REGION Network 56: Paregg. Testa - [Sollevatore] - Movimento operazione a lavoro / a riposo
   // Sollevatore del Centraggio - Scende quando è in posizione e sta attendendo il pezzo
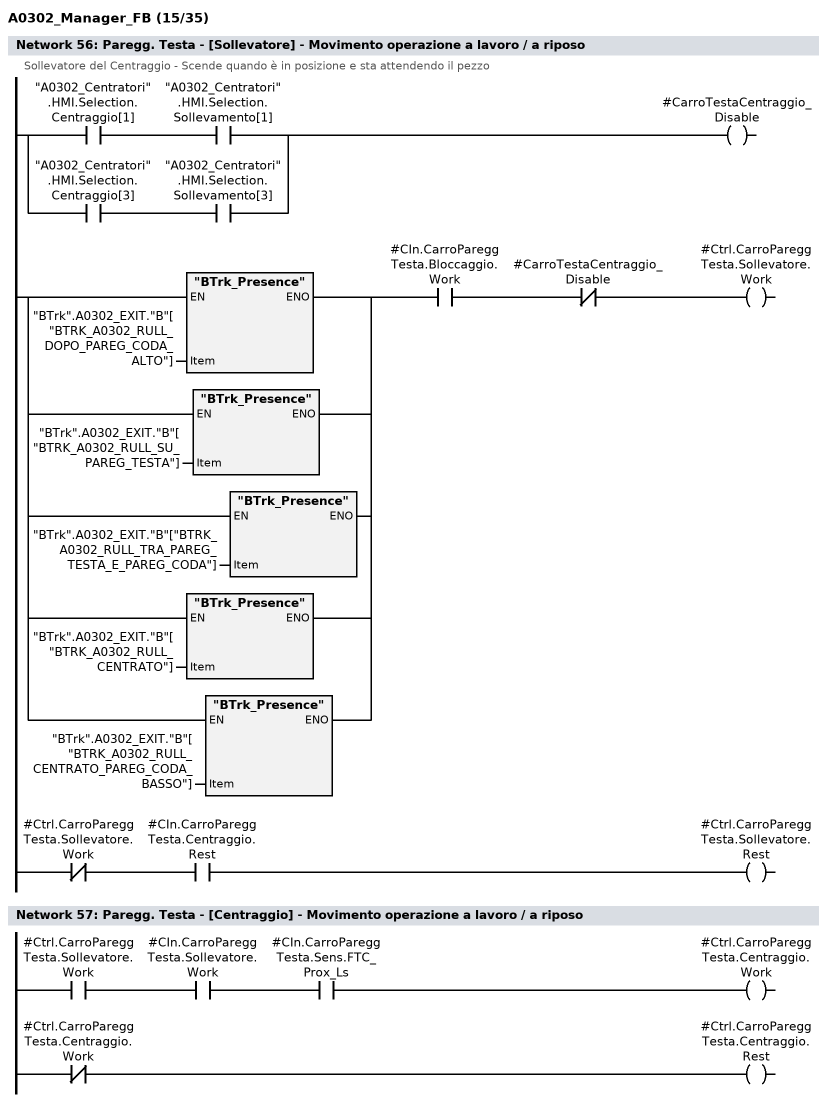
   RUNG wire#powerrail
      Contact( "A0302_Centratori".HMI.Selection.Centraggio[1] )
      Contact( "A0302_Centratori".HMI.Selection.Sollevamento[1] )
      wire#w1
      Coil( #CarroTestaCentraggio_Disable )
   END_RUNG
   RUNG wire#powerrail
      Contact( "A0302_Centratori".HMI.Selection.Centraggio[3] )
      Contact( "A0302_Centratori".HMI.Selection.Sollevamento[3] )
   END_RUNG wire#w1
   RUNG wire#powerrail
      "BTrk_Presence"(Item := "BTrk".A0302_EXIT."B"["BTRK_A0302_RULL_DOPO_PAREG_CODA_ALTO"])
      wire#w2
      Contact( #CIn.CarroPareggTesta.Bloccaggio.Work )
      I_Contact( #CarroTestaCentraggio_Disable )
      Coil( #Ctrl.CarroPareggTesta.Sollevatore.Work )
   END_RUNG
   RUNG wire#powerrail
      "BTrk_Presence"(Item := "BTrk".A0302_EXIT."B"["BTRK_A0302_RULL_SU_PAREG_TESTA"])
   END_RUNG wire#w2
   RUNG wire#powerrail
      "BTrk_Presence"(Item := "BTrk".A0302_EXIT."B"["BTRK_A0302_RULL_TRA_PAREG_TESTA_E_PAREG_CODA"])
   END_RUNG wire#w2
   RUNG wire#powerrail
      "BTrk_Presence"(Item := "BTrk".A0302_EXIT."B"["BTRK_A0302_RULL_CENTRATO"])
   END_RUNG wire#w2
   RUNG wire#powerrail
      "BTrk_Presence"(Item := "BTrk".A0302_EXIT."B"["BTRK_A0302_RULL_CENTRATO_PAREG_CODA_BASSO"])
   END_RUNG wire#w2
   RUNG wire#powerrail
      I_Contact( #Ctrl.CarroPareggTesta.Sollevatore.Work )
      Contact( #CIn.CarroPareggTesta.Centraggio.Rest )
      Coil( #Ctrl.CarroPareggTesta.Sollevatore.Rest )
   END_RUNG
   // the same network as SCL:
   #CarroTestaCentraggio_Disable := ("A0302_Centratori".HMI.Selection.Centraggio[1] AND "A0302_Centratori".HMI.Selection.Sollevamento[1]) OR ("A0302_Centratori".HMI.Selection.Centraggio[3] AND "A0302_Centratori".HMI.Selection.Sollevamento[3]);
   "BTrk_Presence"(Item := "BTrk".A0302_EXIT."B"["BTRK_A0302_RULL_DOPO_PAREG_CODA_ALTO"], ENO => #_w1);
   "BTrk_Presence"(Item := "BTrk".A0302_EXIT."B"["BTRK_A0302_RULL_SU_PAREG_TESTA"], ENO => #_w2);
   "BTrk_Presence"(Item := "BTrk".A0302_EXIT."B"["BTRK_A0302_RULL_TRA_PAREG_TESTA_E_PAREG_CODA"], ENO => #_w3);
   "BTrk_Presence"(Item := "BTrk".A0302_EXIT."B"["BTRK_A0302_RULL_CENTRATO"], ENO => #_w4);
   "BTrk_Presence"(Item := "BTrk".A0302_EXIT."B"["BTRK_A0302_RULL_CENTRATO_PAREG_CODA_BASSO"], ENO => #_w5);
   #Ctrl.CarroPareggTesta.Sollevatore.Work := (#_w1 OR #_w2 OR #_w3 OR #_w4 OR #_w5) AND #CIn.CarroPareggTesta.Bloccaggio.Work AND NOT #CarroTestaCentraggio_Disable;
   #Ctrl.CarroPareggTesta.Sollevatore.Rest := NOT #Ctrl.CarroPareggTesta.Sollevatore.Work AND #CIn.CarroPareggTesta.Centraggio.Rest;
END_REGION

REGION Network 57: Paregg. Testa - [Centraggio] - Movimento operazione a lavoro / a riposo
   RUNG wire#powerrail
      Contact( #Ctrl.CarroPareggTesta.Sollevatore.Work )
      Contact( #CIn.CarroPareggTesta.Sollevatore.Work )
      Contact( #CIn.CarroPareggTesta.Sens.FTC_Prox_Ls )
      Coil( #Ctrl.CarroPareggTesta.Centraggio.Work )
   END_RUNG
   RUNG wire#powerrail
      I_Contact( #Ctrl.CarroPareggTesta.Centraggio.Work )
      Coil( #Ctrl.CarroPareggTesta.Centraggio.Rest )
   END_RUNG
   // the same network as SCL:
   #Ctrl.CarroPareggTesta.Centraggio.Work := #Ctrl.CarroPareggTesta.Sollevatore.Work AND #CIn.CarroPareggTesta.Sollevatore.Work AND #CIn.CarroPareggTesta.Sens.FTC_Prox_Ls;
   #Ctrl.CarroPareggTesta.Centraggio.Rest := NOT #Ctrl.CarroPareggTesta.Centraggio.Work;
END_REGION

REGION Network 58: <+>
END_REGION

REGION Network 59: Paregg. Testa - [Ax - Sollevatore + Centraggio] - COut Manager
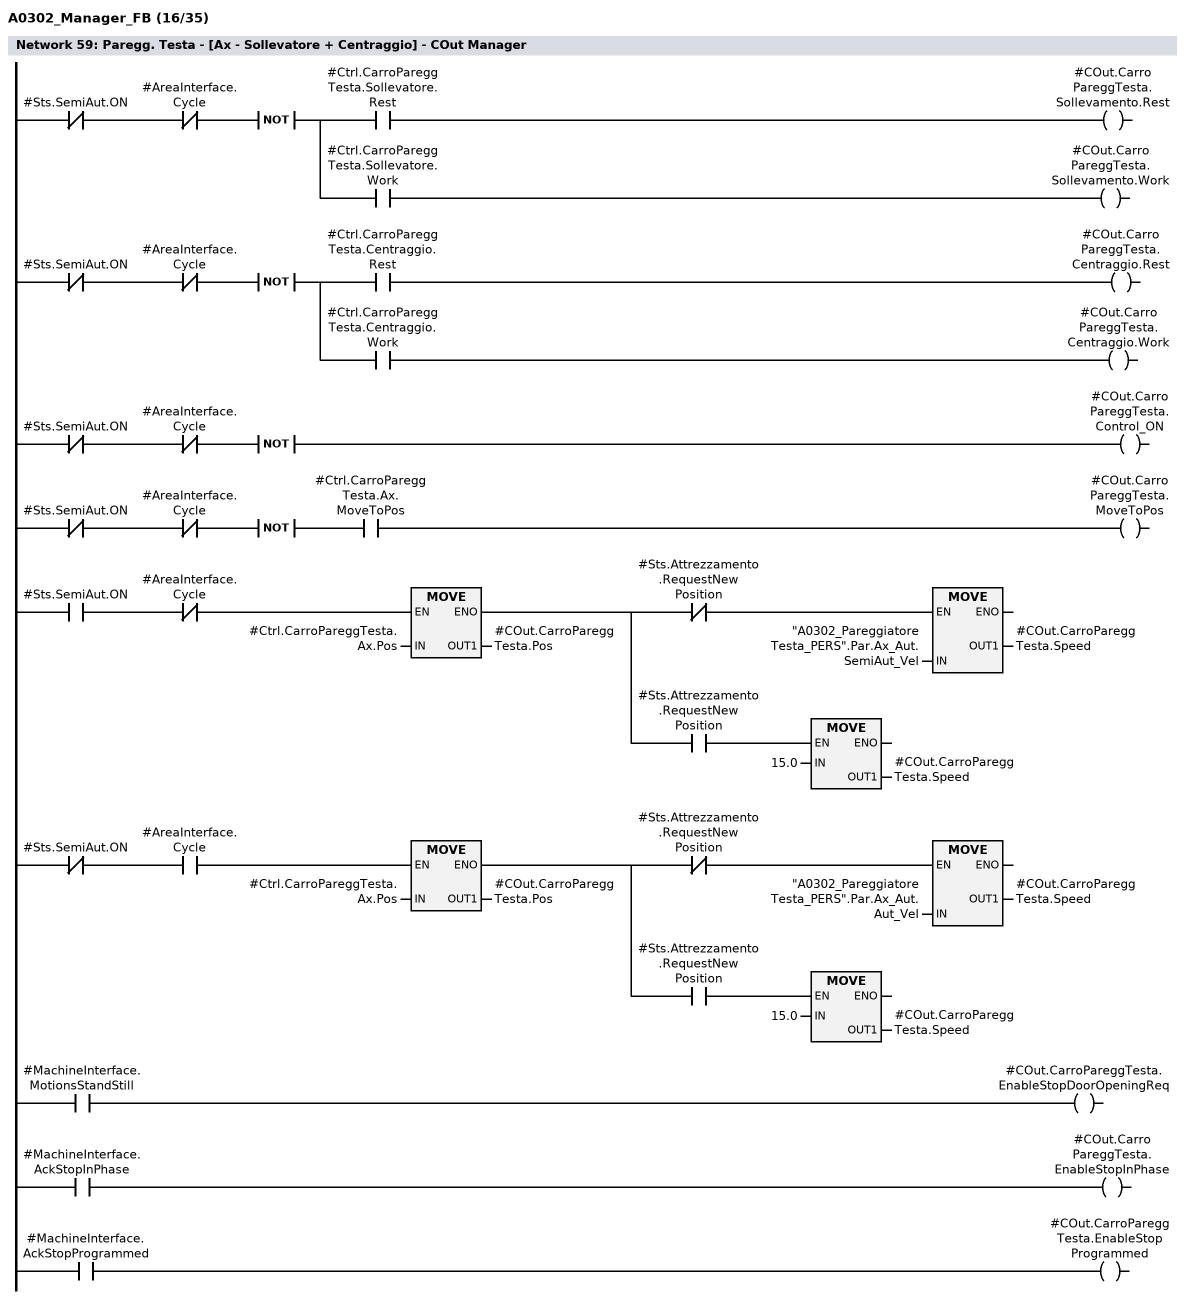
   RUNG wire#powerrail
      I_Contact( #Sts.SemiAut.ON )
      I_Contact( #AreaInterface.Cycle )
      Not()
      wire#w1
      Contact( #Ctrl.CarroPareggTesta.Sollevatore.Rest )
      Coil( #COut.CarroPareggTesta.Sollevamento.Rest )
   END_RUNG
   RUNG wire#w1
      Contact( #Ctrl.CarroPareggTesta.Sollevatore.Work )
      Coil( #COut.CarroPareggTesta.Sollevamento.Work )
   END_RUNG
   RUNG wire#powerrail
      I_Contact( #Sts.SemiAut.ON )
      I_Contact( #AreaInterface.Cycle )
      Not()
      wire#w2
      Contact( #Ctrl.CarroPareggTesta.Centraggio.Rest )
      Coil( #COut.CarroPareggTesta.Centraggio.Rest )
   END_RUNG
   RUNG wire#w2
      Contact( #Ctrl.CarroPareggTesta.Centraggio.Work )
      Coil( #COut.CarroPareggTesta.Centraggio.Work )
   END_RUNG
   RUNG wire#powerrail
      I_Contact( #Sts.SemiAut.ON )
      I_Contact( #AreaInterface.Cycle )
      Not()
      Coil( #COut.CarroPareggTesta.Control_ON )
   END_RUNG
   RUNG wire#powerrail
      I_Contact( #Sts.SemiAut.ON )
      I_Contact( #AreaInterface.Cycle )
      Not()
      Contact( #Ctrl.CarroPareggTesta.Ax.MoveToPos )
      Coil( #COut.CarroPareggTesta.MoveToPos )
   END_RUNG
   RUNG wire#powerrail
      Contact( #Sts.SemiAut.ON )
      I_Contact( #AreaInterface.Cycle )
      Move(in := #Ctrl.CarroPareggTesta.Ax.Pos, out1 => #COut.CarroPareggTesta.Pos)
      wire#w3
      I_Contact( #Sts.Attrezzamento.RequestNewPosition )
      Move(in := "A0302_PareggiatoreTesta_PERS".Par.Ax_Aut.SemiAut_Vel, out1 => #COut.CarroPareggTesta.Speed)
   END_RUNG
   RUNG wire#w3
      Contact( #Sts.Attrezzamento.RequestNewPosition )
      Move(in := 15.0, out1 => #COut.CarroPareggTesta.Speed)
   END_RUNG
   RUNG wire#powerrail
      I_Contact( #Sts.SemiAut.ON )
      Contact( #AreaInterface.Cycle )
      Move(in := #Ctrl.CarroPareggTesta.Ax.Pos, out1 => #COut.CarroPareggTesta.Pos)
      wire#w4
      I_Contact( #Sts.Attrezzamento.RequestNewPosition )
      Move(in := "A0302_PareggiatoreTesta_PERS".Par.Ax_Aut.Aut_Vel, out1 => #COut.CarroPareggTesta.Speed)
   END_RUNG
   RUNG wire#w4
      Contact( #Sts.Attrezzamento.RequestNewPosition )
      Move(in := 15.0, out1 => #COut.CarroPareggTesta.Speed)
   END_RUNG
   RUNG wire#powerrail
      Contact( #MachineInterface.MotionsStandStill )
      Coil( #COut.CarroPareggTesta.EnableStopDoorOpeningReq )
   END_RUNG
   RUNG wire#powerrail
      Contact( #MachineInterface.AckStopInPhase )
      Coil( #COut.CarroPareggTesta.EnableStopInPhase )
   END_RUNG
   RUNG wire#powerrail
      Contact( #MachineInterface.AckStopProgrammed )
      Coil( #COut.CarroPareggTesta.EnableStopProgrammed )
   END_RUNG
   // the same network as SCL:
   #_w1 := NOT (NOT #Sts.SemiAut.ON AND NOT #AreaInterface.Cycle);
   #COut.CarroPareggTesta.Sollevamento.Rest := #_w1 AND #Ctrl.CarroPareggTesta.Sollevatore.Rest;
   #COut.CarroPareggTesta.Sollevamento.Work := #_w1 AND #Ctrl.CarroPareggTesta.Sollevatore.Work;
   #_w2 := NOT (NOT #Sts.SemiAut.ON AND NOT #AreaInterface.Cycle);
   #COut.CarroPareggTesta.Centraggio.Rest := #_w2 AND #Ctrl.CarroPareggTesta.Centraggio.Rest;
   #COut.CarroPareggTesta.Centraggio.Work := #_w2 AND #Ctrl.CarroPareggTesta.Centraggio.Work;
   #COut.CarroPareggTesta.Control_ON := NOT (NOT #Sts.SemiAut.ON AND NOT #AreaInterface.Cycle);
   #COut.CarroPareggTesta.MoveToPos := NOT (NOT #Sts.SemiAut.ON AND NOT #AreaInterface.Cycle) AND #Ctrl.CarroPareggTesta.Ax.MoveToPos;
   #_w3 := #Sts.SemiAut.ON AND NOT #AreaInterface.Cycle;
   IF #_w3 THEN #COut.CarroPareggTesta.Pos := #Ctrl.CarroPareggTesta.Ax.Pos; END_IF;
   IF #_w3 AND NOT #Sts.Attrezzamento.RequestNewPosition THEN
       #COut.CarroPareggTesta.Speed := "A0302_PareggiatoreTesta_PERS".Par.Ax_Aut.SemiAut_Vel;
   END_IF;
   IF #_w3 AND #Sts.Attrezzamento.RequestNewPosition THEN #COut.CarroPareggTesta.Speed := 15.0; END_IF;
   #_w4 := NOT #Sts.SemiAut.ON AND #AreaInterface.Cycle;
   IF #_w4 THEN #COut.CarroPareggTesta.Pos := #Ctrl.CarroPareggTesta.Ax.Pos; END_IF;
   IF #_w4 AND NOT #Sts.Attrezzamento.RequestNewPosition THEN
       #COut.CarroPareggTesta.Speed := "A0302_PareggiatoreTesta_PERS".Par.Ax_Aut.Aut_Vel;
   END_IF;
   IF #_w4 AND #Sts.Attrezzamento.RequestNewPosition THEN #COut.CarroPareggTesta.Speed := 15.0; END_IF;
   #COut.CarroPareggTesta.EnableStopDoorOpeningReq := #MachineInterface.MotionsStandStill;
   #COut.CarroPareggTesta.EnableStopInPhase := #MachineInterface.AckStopInPhase;
   #COut.CarroPareggTesta.EnableStopProgrammed := #MachineInterface.AckStopProgrammed;
END_REGION

REGION Network 60: Paregg. Testa [Bloccaggio] - Movimento operazione a lavoro / a riposo
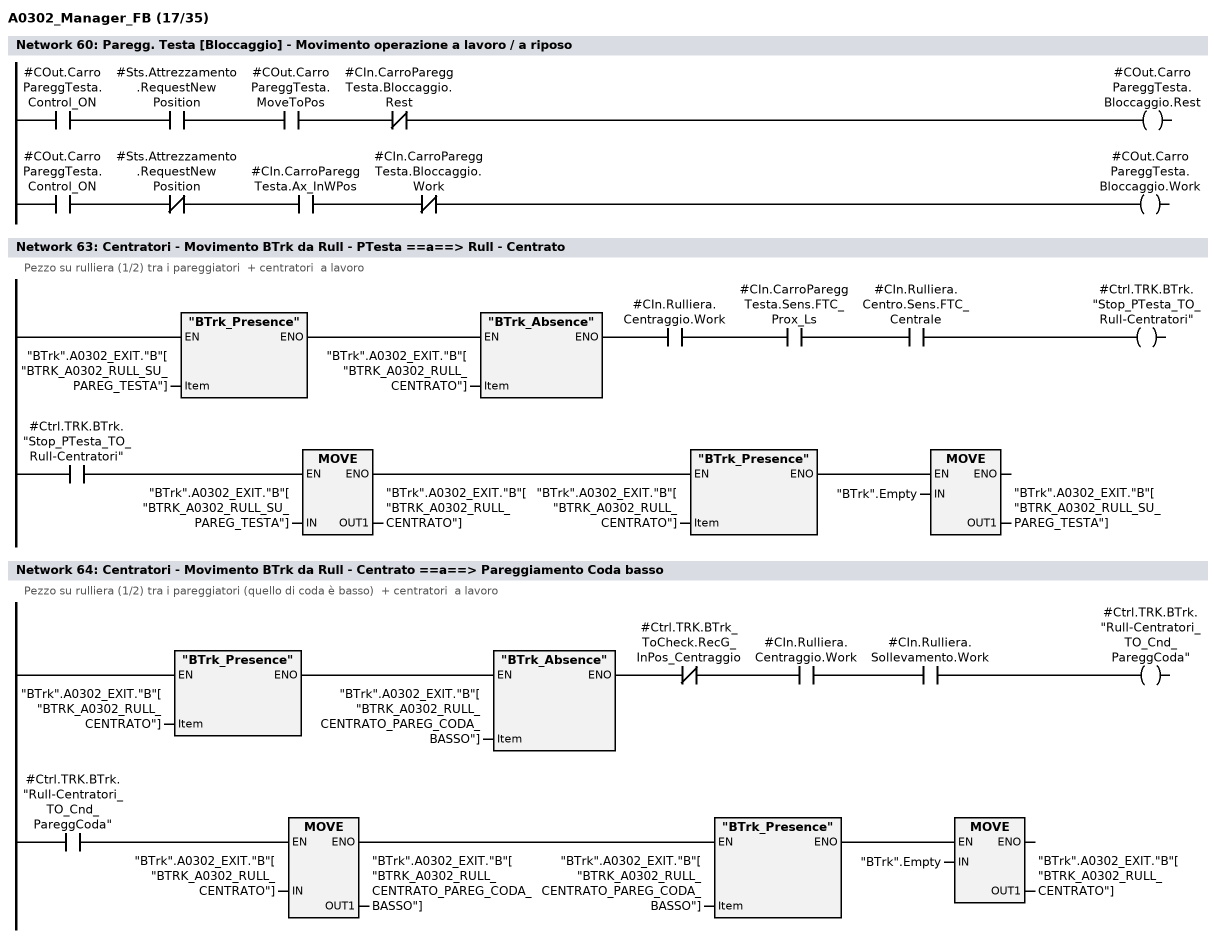
   RUNG wire#powerrail
      Contact( #COut.CarroPareggTesta.Control_ON )
      Contact( #Sts.Attrezzamento.RequestNewPosition )
      Contact( #COut.CarroPareggTesta.MoveToPos )
      I_Contact( #CIn.CarroPareggTesta.Bloccaggio.Rest )
      Coil( #COut.CarroPareggTesta.Bloccaggio.Rest )
   END_RUNG
   RUNG wire#powerrail
      Contact( #COut.CarroPareggTesta.Control_ON )
      I_Contact( #Sts.Attrezzamento.RequestNewPosition )
      Contact( #CIn.CarroPareggTesta.Ax_InWPos )
      I_Contact( #CIn.CarroPareggTesta.Bloccaggio.Work )
      Coil( #COut.CarroPareggTesta.Bloccaggio.Work )
   END_RUNG
   // the same network as SCL:
   #COut.CarroPareggTesta.Bloccaggio.Rest := #COut.CarroPareggTesta.Control_ON AND #Sts.Attrezzamento.RequestNewPosition AND #COut.CarroPareggTesta.MoveToPos AND NOT #CIn.CarroPareggTesta.Bloccaggio.Rest;
   #COut.CarroPareggTesta.Bloccaggio.Work := #COut.CarroPareggTesta.Control_ON AND NOT #Sts.Attrezzamento.RequestNewPosition AND #CIn.CarroPareggTesta.Ax_InWPos AND NOT #CIn.CarroPareggTesta.Bloccaggio.Work;
END_REGION

REGION Network 61: <<<< CENTRATORI >>>>
END_REGION

REGION Network 62: <+>
END_REGION

REGION Network 63: Centratori - Movimento BTrk da Rull - PTesta ==a==> Rull - Centrato
   // Pezzo su rulliera (1/2) tra i pareggiatori  + centratori  a lavoro
   RUNG wire#powerrail
      "BTrk_Presence"(Item := "BTrk".A0302_EXIT."B"["BTRK_A0302_RULL_SU_PAREG_TESTA"])
      "BTrk_Absence"(Item := "BTrk".A0302_EXIT."B"["BTRK_A0302_RULL_CENTRATO"])
      Contact( #CIn.Rulliera.Centraggio.Work )
      Contact( #CIn.CarroPareggTesta.Sens.FTC_Prox_Ls )
      Contact( #CIn.Rulliera.Centro.Sens.FTC_Centrale )
      Coil( #Ctrl.TRK.BTrk."Stop_PTesta_TO_Rull-Centratori" )
   END_RUNG
   RUNG wire#powerrail
      Contact( #Ctrl.TRK.BTrk."Stop_PTesta_TO_Rull-Centratori" )
      Move(in := "BTrk".A0302_EXIT."B"["BTRK_A0302_RULL_SU_PAREG_TESTA"], out1 => "BTrk".A0302_EXIT."B"["BTRK_A0302_RULL_CENTRATO"])
      "BTrk_Presence"(Item := "BTrk".A0302_EXIT."B"["BTRK_A0302_RULL_CENTRATO"])
      Move(in := "BTrk".Empty, out1 => "BTrk".A0302_EXIT."B"["BTRK_A0302_RULL_SU_PAREG_TESTA"])
   END_RUNG
   // the same network as SCL:
   "BTrk_Presence"(Item := "BTrk".A0302_EXIT."B"["BTRK_A0302_RULL_SU_PAREG_TESTA"], ENO => #_w1);
   "BTrk_Absence"(EN := #_w1, Item := "BTrk".A0302_EXIT."B"["BTRK_A0302_RULL_CENTRATO"], ENO => #_w2);
   #Ctrl.TRK.BTrk."Stop_PTesta_TO_Rull-Centratori" := #_w2 AND #CIn.Rulliera.Centraggio.Work AND #CIn.CarroPareggTesta.Sens.FTC_Prox_Ls AND #CIn.Rulliera.Centro.Sens.FTC_Centrale;
   IF #Ctrl.TRK.BTrk."Stop_PTesta_TO_Rull-Centratori" THEN
       "BTrk".A0302_EXIT."B"["BTRK_A0302_RULL_CENTRATO"] := "BTrk".A0302_EXIT."B"["BTRK_A0302_RULL_SU_PAREG_TESTA"];
   END_IF;
   "BTrk_Presence"(EN := #Ctrl.TRK.BTrk."Stop_PTesta_TO_Rull-Centratori",
                   Item := "BTrk".A0302_EXIT."B"["BTRK_A0302_RULL_CENTRATO"],
                   ENO => #_w3);
   IF #_w3 THEN "BTrk".A0302_EXIT."B"["BTRK_A0302_RULL_SU_PAREG_TESTA"] := "BTrk".Empty; END_IF;
END_REGION

REGION Network 64: Centratori - Movimento BTrk da Rull - Centrato ==a==> Pareggiamento Coda basso
   // Pezzo su rulliera (1/2) tra i pareggiatori (quello di coda è basso)  + centratori  a lavoro
   RUNG wire#powerrail
      "BTrk_Presence"(Item := "BTrk".A0302_EXIT."B"["BTRK_A0302_RULL_CENTRATO"])
      "BTrk_Absence"(Item := "BTrk".A0302_EXIT."B"["BTRK_A0302_RULL_CENTRATO_PAREG_CODA_BASSO"])
      I_Contact( #Ctrl.TRK.BTrk_ToCheck.RecG_InPos_Centraggio )
      Contact( #CIn.Rulliera.Centraggio.Work )
      Contact( #CIn.Rulliera.Sollevamento.Work )
      Coil( #Ctrl.TRK.BTrk."Rull-Centratori_TO_Cnd_PareggCoda" )
   END_RUNG
   RUNG wire#powerrail
      Contact( #Ctrl.TRK.BTrk."Rull-Centratori_TO_Cnd_PareggCoda" )
      Move(in := "BTrk".A0302_EXIT."B"["BTRK_A0302_RULL_CENTRATO"], out1 => "BTrk".A0302_EXIT."B"["BTRK_A0302_RULL_CENTRATO_PAREG_CODA_BASSO"])
      "BTrk_Presence"(Item := "BTrk".A0302_EXIT."B"["BTRK_A0302_RULL_CENTRATO_PAREG_CODA_BASSO"])
      Move(in := "BTrk".Empty, out1 => "BTrk".A0302_EXIT."B"["BTRK_A0302_RULL_CENTRATO"])
   END_RUNG
   // the same network as SCL:
   "BTrk_Presence"(Item := "BTrk".A0302_EXIT."B"["BTRK_A0302_RULL_CENTRATO"], ENO => #_w1);
   "BTrk_Absence"(EN := #_w1,
                  Item := "BTrk".A0302_EXIT."B"["BTRK_A0302_RULL_CENTRATO_PAREG_CODA_BASSO"],
                  ENO => #_w2);
   #Ctrl.TRK.BTrk."Rull-Centratori_TO_Cnd_PareggCoda" := #_w2 AND NOT #Ctrl.TRK.BTrk_ToCheck.RecG_InPos_Centraggio AND #CIn.Rulliera.Centraggio.Work AND #CIn.Rulliera.Sollevamento.Work;
   IF #Ctrl.TRK.BTrk."Rull-Centratori_TO_Cnd_PareggCoda" THEN
       "BTrk".A0302_EXIT."B"["BTRK_A0302_RULL_CENTRATO_PAREG_CODA_BASSO"] := "BTrk".A0302_EXIT."B"["BTRK_A0302_RULL_CENTRATO"];
   END_IF;
   "BTrk_Presence"(EN := #Ctrl.TRK.BTrk."Rull-Centratori_TO_Cnd_PareggCoda",
                   Item := "BTrk".A0302_EXIT."B"["BTRK_A0302_RULL_CENTRATO_PAREG_CODA_BASSO"],
                   ENO => #_w3);
   IF #_w3 THEN "BTrk".A0302_EXIT."B"["BTRK_A0302_RULL_CENTRATO"] := "BTrk".Empty; END_IF;
END_REGION

REGION Network 65: Centratori - Movimento BTrk da Pareggiamento Coda basso ==a==> Pareggiato
   // Pezzo su rulliera (1/2) tra i pareggiatori e paregiatura di coda eseguito lavoro cilindro idraulico (ora si sa la misura del pezzo, si può mettere utenze in attesa del prossimo pezzo)
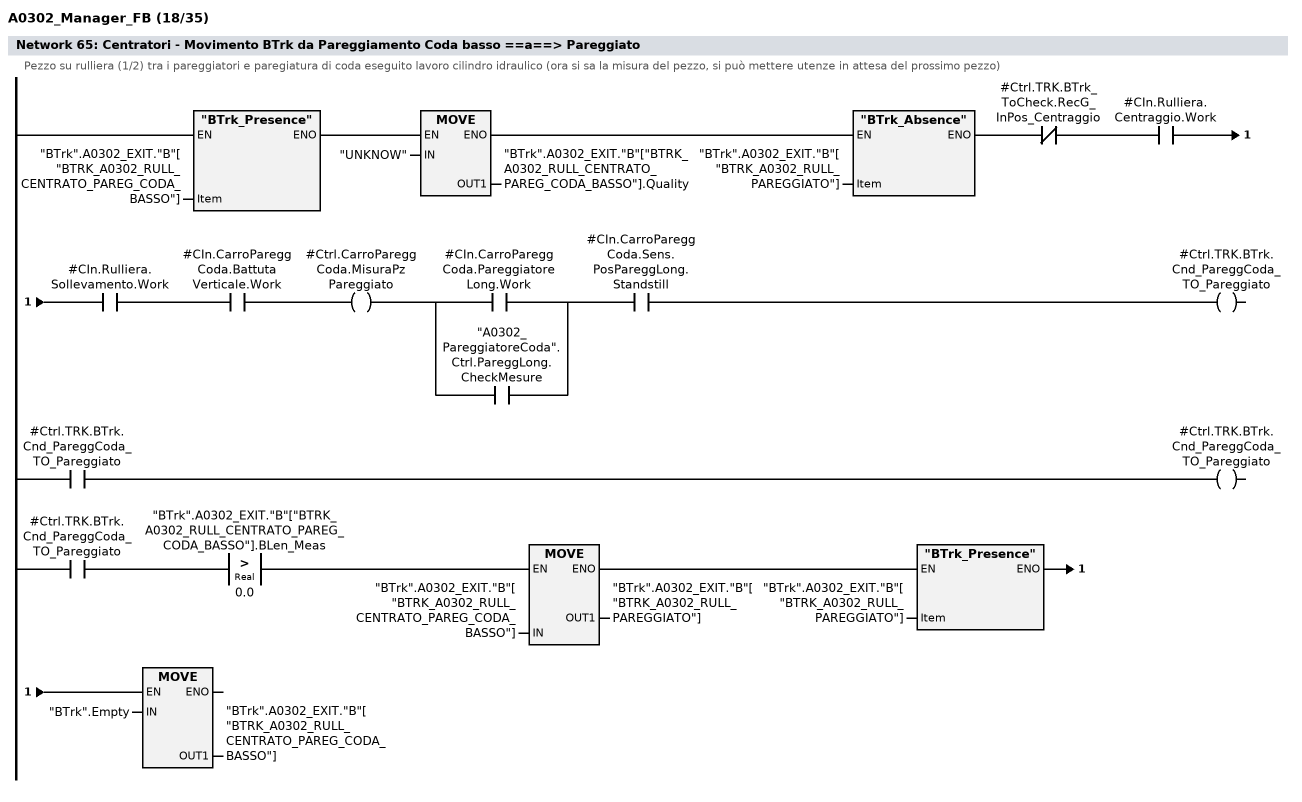
   RUNG wire#powerrail
      "BTrk_Presence"(Item := "BTrk".A0302_EXIT."B"["BTRK_A0302_RULL_CENTRATO_PAREG_CODA_BASSO"])
      Move(in := "UNKNOW", out1 => "BTrk".A0302_EXIT."B"["BTRK_A0302_RULL_CENTRATO_PAREG_CODA_BASSO"].Quality)
      "BTrk_Absence"(Item := "BTrk".A0302_EXIT."B"["BTRK_A0302_RULL_PAREGGIATO"])
      I_Contact( #Ctrl.TRK.BTrk_ToCheck.RecG_InPos_Centraggio )
      Contact( #CIn.Rulliera.Centraggio.Work )
      Contact( #CIn.Rulliera.Sollevamento.Work )
      Contact( #CIn.CarroPareggCoda.BattutaVerticale.Work )
      Coil( #Ctrl.CarroPareggCoda.MisuraPzPareggiato )
      wire#w1
      Contact( #CIn.CarroPareggCoda.PareggiatoreLong.Work )
      wire#w2
      Contact( #CIn.CarroPareggCoda.Sens.PosPareggLong.Standstill )
      Coil( #Ctrl.TRK.BTrk.Cnd_PareggCoda_TO_Pareggiato )
   END_RUNG
   RUNG wire#w1
      Contact( "A0302_PareggiatoreCoda".Ctrl.PareggLong.CheckMesure )
   END_RUNG wire#w2
   RUNG wire#powerrail
      Contact( #Ctrl.TRK.BTrk.Cnd_PareggCoda_TO_Pareggiato )
      Coil( #Ctrl.TRK.BTrk.Cnd_PareggCoda_TO_Pareggiato )
   END_RUNG
   RUNG wire#powerrail
      Contact( #Ctrl.TRK.BTrk.Cnd_PareggCoda_TO_Pareggiato )
      { S7_Templates := "SrcType := Real" } GT_Contact(in1 := "BTrk".A0302_EXIT."B"["BTRK_A0302_RULL_CENTRATO_PAREG_CODA_BASSO"].BLen_Meas, in2 := 0.0)
      Move(in := "BTrk".A0302_EXIT."B"["BTRK_A0302_RULL_CENTRATO_PAREG_CODA_BASSO"], out1 => "BTrk".A0302_EXIT."B"["BTRK_A0302_RULL_PAREGGIATO"])
      "BTrk_Presence"(Item := "BTrk".A0302_EXIT."B"["BTRK_A0302_RULL_PAREGGIATO"])
      Move(in := "BTrk".Empty, out1 => "BTrk".A0302_EXIT."B"["BTRK_A0302_RULL_CENTRATO_PAREG_CODA_BASSO"])
   END_RUNG
   // the same network as SCL:
   "BTrk_Presence"(Item := "BTrk".A0302_EXIT."B"["BTRK_A0302_RULL_CENTRATO_PAREG_CODA_BASSO"], ENO => #_w1);
   IF #_w1 THEN
       "BTrk".A0302_EXIT."B"["BTRK_A0302_RULL_CENTRATO_PAREG_CODA_BASSO"].Quality := "UNKNOW";
   END_IF;
   "BTrk_Absence"(EN := #_w1, Item := "BTrk".A0302_EXIT."B"["BTRK_A0302_RULL_PAREGGIATO"], ENO => #_w2);
   #Ctrl.CarroPareggCoda.MisuraPzPareggiato := #_w2 AND NOT #Ctrl.TRK.BTrk_ToCheck.RecG_InPos_Centraggio AND #CIn.Rulliera.Centraggio.Work AND #CIn.Rulliera.Sollevamento.Work AND #CIn.CarroPareggCoda.BattutaVerticale.Work;
   #Ctrl.TRK.BTrk.Cnd_PareggCoda_TO_Pareggiato := #Ctrl.CarroPareggCoda.MisuraPzPareggiato AND (#CIn.CarroPareggCoda.PareggiatoreLong.Work OR "A0302_PareggiatoreCoda".Ctrl.PareggLong.CheckMesure) AND #CIn.CarroPareggCoda.Sens.PosPareggLong.Standstill;
   #Ctrl.TRK.BTrk.Cnd_PareggCoda_TO_Pareggiato := #Ctrl.TRK.BTrk.Cnd_PareggCoda_TO_Pareggiato;
   #_w3 := #Ctrl.TRK.BTrk.Cnd_PareggCoda_TO_Pareggiato AND ("BTrk".A0302_EXIT."B"["BTRK_A0302_RULL_CENTRATO_PAREG_CODA_BASSO"].BLen_Meas > 0.0);
   IF #_w3 THEN
       "BTrk".A0302_EXIT."B"["BTRK_A0302_RULL_PAREGGIATO"] := "BTrk".A0302_EXIT."B"["BTRK_A0302_RULL_CENTRATO_PAREG_CODA_BASSO"];
   END_IF;
   "BTrk_Presence"(EN := #_w3, Item := "BTrk".A0302_EXIT."B"["BTRK_A0302_RULL_PAREGGIATO"], ENO => #_w4);
   IF #_w4 THEN "BTrk".A0302_EXIT."B"["BTRK_A0302_RULL_CENTRATO_PAREG_CODA_BASSO"] := "BTrk".Empty; END_IF;
END_REGION

REGION Network 66: <+>
END_REGION

REGION Network 67: [Sollevamento] - Rulliera - Movimento operazione a lavoro / a riposo
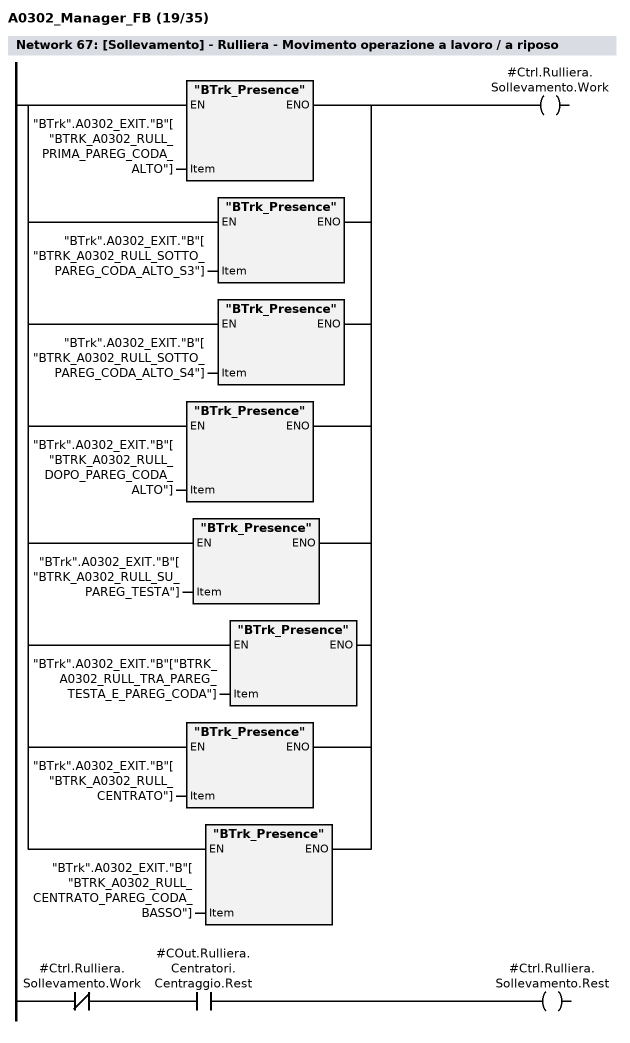
   RUNG wire#powerrail
      "BTrk_Presence"(Item := "BTrk".A0302_EXIT."B"["BTRK_A0302_RULL_PRIMA_PAREG_CODA_ALTO"])
      wire#w1
      Coil( #Ctrl.Rulliera.Sollevamento.Work )
   END_RUNG
   RUNG wire#powerrail
      "BTrk_Presence"(Item := "BTrk".A0302_EXIT."B"["BTRK_A0302_RULL_SOTTO_PAREG_CODA_ALTO_S3"])
   END_RUNG wire#w1
   RUNG wire#powerrail
      "BTrk_Presence"(Item := "BTrk".A0302_EXIT."B"["BTRK_A0302_RULL_SOTTO_PAREG_CODA_ALTO_S4"])
   END_RUNG wire#w1
   RUNG wire#powerrail
      "BTrk_Presence"(Item := "BTrk".A0302_EXIT."B"["BTRK_A0302_RULL_DOPO_PAREG_CODA_ALTO"])
   END_RUNG wire#w1
   RUNG wire#powerrail
      "BTrk_Presence"(Item := "BTrk".A0302_EXIT."B"["BTRK_A0302_RULL_SU_PAREG_TESTA"])
   END_RUNG wire#w1
   RUNG wire#powerrail
      "BTrk_Presence"(Item := "BTrk".A0302_EXIT."B"["BTRK_A0302_RULL_TRA_PAREG_TESTA_E_PAREG_CODA"])
   END_RUNG wire#w1
   RUNG wire#powerrail
      "BTrk_Presence"(Item := "BTrk".A0302_EXIT."B"["BTRK_A0302_RULL_CENTRATO"])
   END_RUNG wire#w1
   RUNG wire#powerrail
      "BTrk_Presence"(Item := "BTrk".A0302_EXIT."B"["BTRK_A0302_RULL_CENTRATO_PAREG_CODA_BASSO"])
   END_RUNG wire#w1
   RUNG wire#powerrail
      I_Contact( #Ctrl.Rulliera.Sollevamento.Work )
      Contact( #COut.Rulliera.Centratori.Centraggio.Rest )
      Coil( #Ctrl.Rulliera.Sollevamento.Rest )
   END_RUNG
   // the same network as SCL:
   "BTrk_Presence"(Item := "BTrk".A0302_EXIT."B"["BTRK_A0302_RULL_PRIMA_PAREG_CODA_ALTO"], ENO => #_w1);
   "BTrk_Presence"(Item := "BTrk".A0302_EXIT."B"["BTRK_A0302_RULL_SOTTO_PAREG_CODA_ALTO_S3"], ENO => #_w2);
   "BTrk_Presence"(Item := "BTrk".A0302_EXIT."B"["BTRK_A0302_RULL_SOTTO_PAREG_CODA_ALTO_S4"], ENO => #_w3);
   "BTrk_Presence"(Item := "BTrk".A0302_EXIT."B"["BTRK_A0302_RULL_DOPO_PAREG_CODA_ALTO"], ENO => #_w4);
   "BTrk_Presence"(Item := "BTrk".A0302_EXIT."B"["BTRK_A0302_RULL_SU_PAREG_TESTA"], ENO => #_w5);
   "BTrk_Presence"(Item := "BTrk".A0302_EXIT."B"["BTRK_A0302_RULL_TRA_PAREG_TESTA_E_PAREG_CODA"], ENO => #_w6);
   "BTrk_Presence"(Item := "BTrk".A0302_EXIT."B"["BTRK_A0302_RULL_CENTRATO"], ENO => #_w7);
   "BTrk_Presence"(Item := "BTrk".A0302_EXIT."B"["BTRK_A0302_RULL_CENTRATO_PAREG_CODA_BASSO"], ENO => #_w8);
   #Ctrl.Rulliera.Sollevamento.Work := #_w1 OR #_w2 OR #_w3 OR #_w4 OR #_w5 OR #_w6 OR #_w7 OR #_w8;
   #Ctrl.Rulliera.Sollevamento.Rest := NOT #Ctrl.Rulliera.Sollevamento.Work AND #COut.Rulliera.Centratori.Centraggio.Rest;
END_REGION

REGION Network 68: [Centraggio] - Rulliera - Movimento operazione a lavoro / a riposo
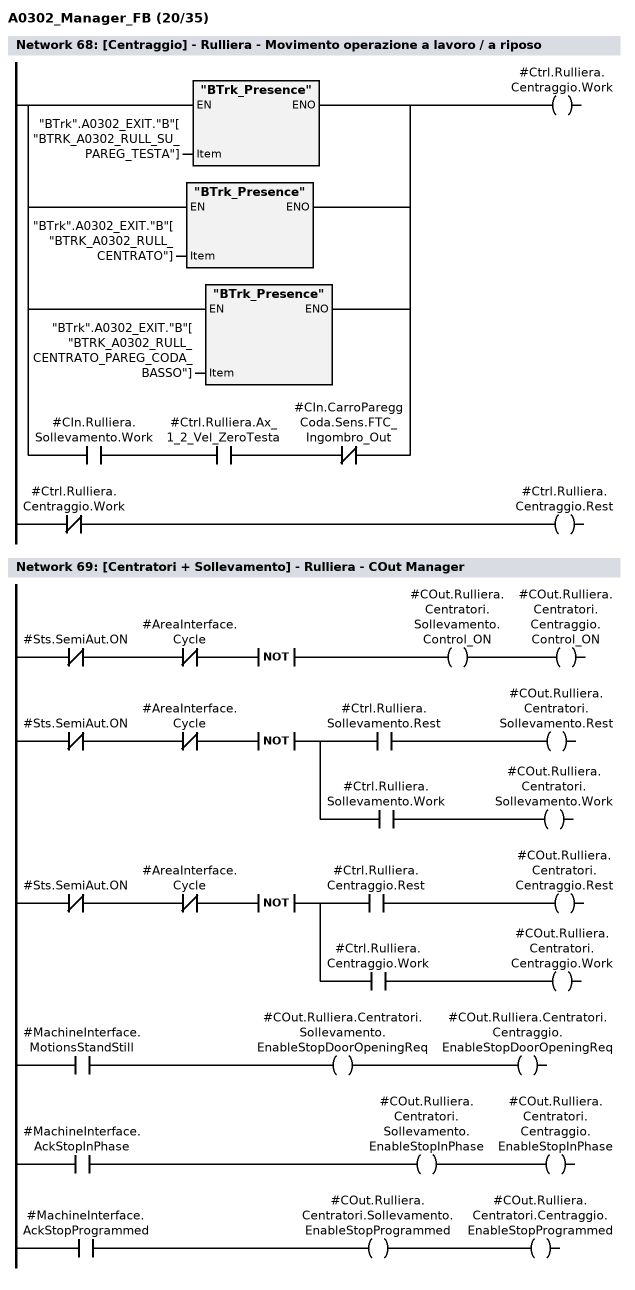
   RUNG wire#powerrail
      "BTrk_Presence"(Item := "BTrk".A0302_EXIT."B"["BTRK_A0302_RULL_SU_PAREG_TESTA"])
      wire#w1
      Coil( #Ctrl.Rulliera.Centraggio.Work )
   END_RUNG
   RUNG wire#powerrail
      "BTrk_Presence"(Item := "BTrk".A0302_EXIT."B"["BTRK_A0302_RULL_CENTRATO"])
   END_RUNG wire#w1
   RUNG wire#powerrail
      "BTrk_Presence"(Item := "BTrk".A0302_EXIT."B"["BTRK_A0302_RULL_CENTRATO_PAREG_CODA_BASSO"])
   END_RUNG wire#w1
   RUNG wire#powerrail
      Contact( #CIn.Rulliera.Sollevamento.Work )
      Contact( #Ctrl.Rulliera.Ax_1_2_Vel_ZeroTesta )
      I_Contact( #CIn.CarroPareggCoda.Sens.FTC_Ingombro_Out )
   END_RUNG wire#w1
   RUNG wire#powerrail
      I_Contact( #Ctrl.Rulliera.Centraggio.Work )
      Coil( #Ctrl.Rulliera.Centraggio.Rest )
   END_RUNG
   // the same network as SCL:
   "BTrk_Presence"(Item := "BTrk".A0302_EXIT."B"["BTRK_A0302_RULL_SU_PAREG_TESTA"], ENO => #_w1);
   "BTrk_Presence"(Item := "BTrk".A0302_EXIT."B"["BTRK_A0302_RULL_CENTRATO"], ENO => #_w2);
   "BTrk_Presence"(Item := "BTrk".A0302_EXIT."B"["BTRK_A0302_RULL_CENTRATO_PAREG_CODA_BASSO"], ENO => #_w3);
   #Ctrl.Rulliera.Centraggio.Work := #_w1 OR #_w2 OR #_w3 OR (#CIn.Rulliera.Sollevamento.Work AND #Ctrl.Rulliera.Ax_1_2_Vel_ZeroTesta AND NOT #CIn.CarroPareggCoda.Sens.FTC_Ingombro_Out);
   #Ctrl.Rulliera.Centraggio.Rest := NOT #Ctrl.Rulliera.Centraggio.Work;
END_REGION

REGION Network 69: [Centratori + Sollevamento] - Rulliera - COut Manager
   RUNG wire#powerrail
      I_Contact( #Sts.SemiAut.ON )
      I_Contact( #AreaInterface.Cycle )
      Not()
      Coil( #COut.Rulliera.Centratori.Sollevamento.Control_ON )
      Coil( #COut.Rulliera.Centratori.Centraggio.Control_ON )
   END_RUNG
   RUNG wire#powerrail
      I_Contact( #Sts.SemiAut.ON )
      I_Contact( #AreaInterface.Cycle )
      Not()
      wire#w1
      Contact( #Ctrl.Rulliera.Sollevamento.Rest )
      Coil( #COut.Rulliera.Centratori.Sollevamento.Rest )
   END_RUNG
   RUNG wire#w1
      Contact( #Ctrl.Rulliera.Sollevamento.Work )
      Coil( #COut.Rulliera.Centratori.Sollevamento.Work )
   END_RUNG
   RUNG wire#powerrail
      I_Contact( #Sts.SemiAut.ON )
      I_Contact( #AreaInterface.Cycle )
      Not()
      wire#w2
      Contact( #Ctrl.Rulliera.Centraggio.Rest )
      Coil( #COut.Rulliera.Centratori.Centraggio.Rest )
   END_RUNG
   RUNG wire#w2
      Contact( #Ctrl.Rulliera.Centraggio.Work )
      Coil( #COut.Rulliera.Centratori.Centraggio.Work )
   END_RUNG
   RUNG wire#powerrail
      Contact( #MachineInterface.MotionsStandStill )
      Coil( #COut.Rulliera.Centratori.Sollevamento.EnableStopDoorOpeningReq )
      Coil( #COut.Rulliera.Centratori.Centraggio.EnableStopDoorOpeningReq )
   END_RUNG
   RUNG wire#powerrail
      Contact( #MachineInterface.AckStopInPhase )
      Coil( #COut.Rulliera.Centratori.Sollevamento.EnableStopInPhase )
      Coil( #COut.Rulliera.Centratori.Centraggio.EnableStopInPhase )
   END_RUNG
   RUNG wire#powerrail
      Contact( #MachineInterface.AckStopProgrammed )
      Coil( #COut.Rulliera.Centratori.Sollevamento.EnableStopProgrammed )
      Coil( #COut.Rulliera.Centratori.Centraggio.EnableStopProgrammed )
   END_RUNG
   // the same network as SCL:
   #COut.Rulliera.Centratori.Sollevamento.Control_ON := NOT (NOT #Sts.SemiAut.ON AND NOT #AreaInterface.Cycle);
   #COut.Rulliera.Centratori.Centraggio.Control_ON := #COut.Rulliera.Centratori.Sollevamento.Control_ON;
   #_w1 := NOT (NOT #Sts.SemiAut.ON AND NOT #AreaInterface.Cycle);
   #COut.Rulliera.Centratori.Sollevamento.Rest := #_w1 AND #Ctrl.Rulliera.Sollevamento.Rest;
   #COut.Rulliera.Centratori.Sollevamento.Work := #_w1 AND #Ctrl.Rulliera.Sollevamento.Work;
   #_w2 := NOT (NOT #Sts.SemiAut.ON AND NOT #AreaInterface.Cycle);
   #COut.Rulliera.Centratori.Centraggio.Rest := #_w2 AND #Ctrl.Rulliera.Centraggio.Rest;
   #COut.Rulliera.Centratori.Centraggio.Work := #_w2 AND #Ctrl.Rulliera.Centraggio.Work;
   #COut.Rulliera.Centratori.Sollevamento.EnableStopDoorOpeningReq := #MachineInterface.MotionsStandStill;
   #COut.Rulliera.Centratori.Centraggio.EnableStopDoorOpeningReq := #MachineInterface.MotionsStandStill;
   #COut.Rulliera.Centratori.Sollevamento.EnableStopInPhase := #MachineInterface.AckStopInPhase;
   #COut.Rulliera.Centratori.Centraggio.EnableStopInPhase := #MachineInterface.AckStopInPhase;
   #COut.Rulliera.Centratori.Sollevamento.EnableStopProgrammed := #MachineInterface.AckStopProgrammed;
   #COut.Rulliera.Centratori.Centraggio.EnableStopProgrammed := #MachineInterface.AckStopProgrammed;
END_REGION

REGION Network 72: ************************************************************************************
END_REGION

REGION Network 73: <<<< PAREGGIATORE CODA >>>>
END_REGION

REGION Network 74: <+>
END_REGION

REGION Network 75: Paregg. Coda - Movimento BTrk da STOP Rull Paregg Coda Basso ==a==> Paregg Coda Alto
   // Pezzo su rulliera (1) + pareggiatore coda alto quindi può muoversi liberamente
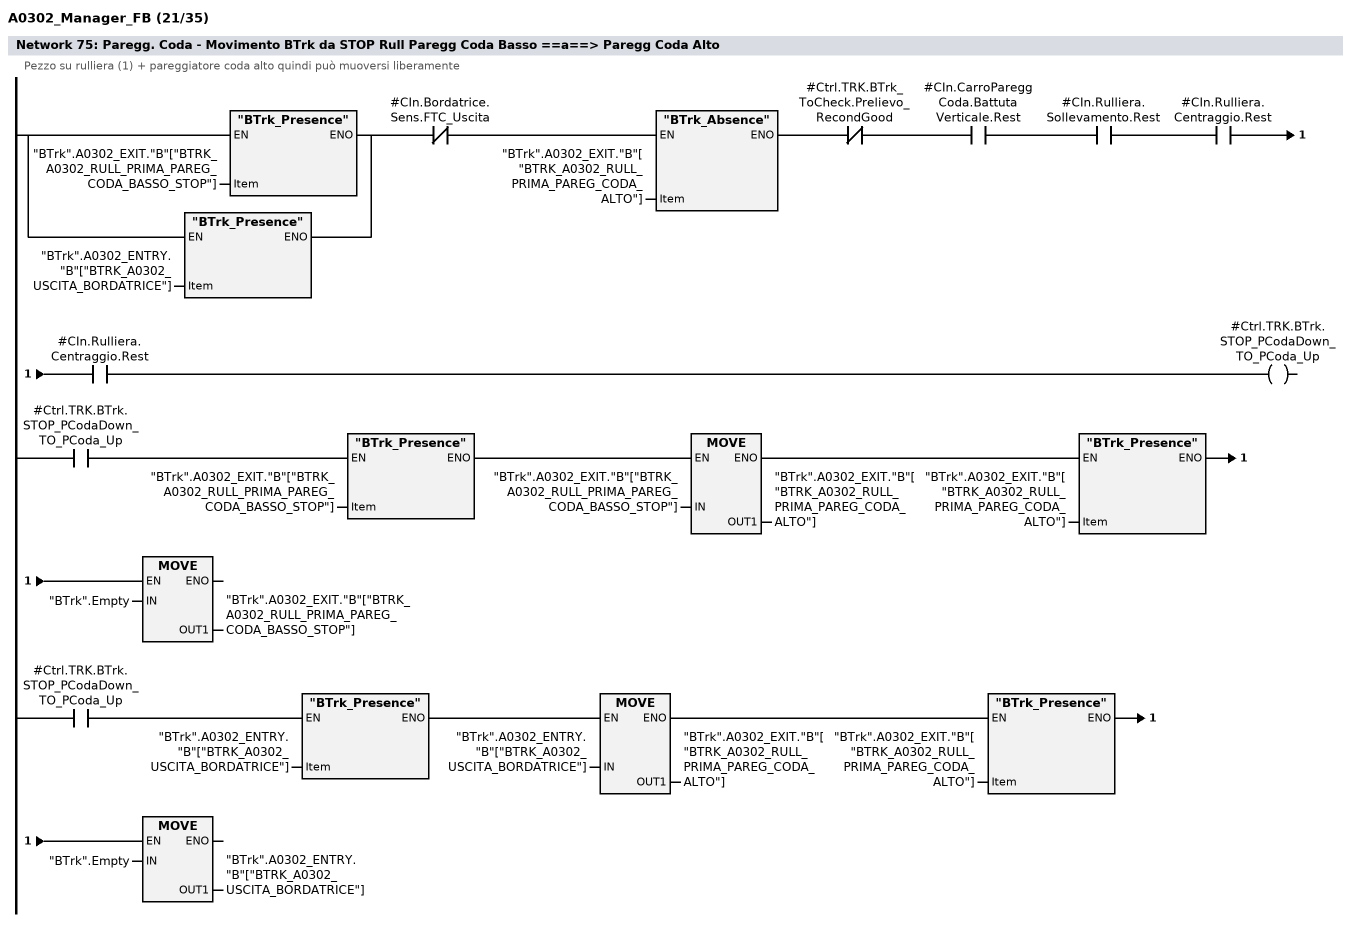
   RUNG wire#powerrail
      "BTrk_Presence"(Item := "BTrk".A0302_EXIT."B"["BTRK_A0302_RULL_PRIMA_PAREG_CODA_BASSO_STOP"])
      wire#w1
      I_Contact( #CIn.Bordatrice.Sens.FTC_Uscita )
      "BTrk_Absence"(Item := "BTrk".A0302_EXIT."B"["BTRK_A0302_RULL_PRIMA_PAREG_CODA_ALTO"])
      I_Contact( #Ctrl.TRK.BTrk_ToCheck.Prelievo_RecondGood )
      Contact( #CIn.CarroPareggCoda.BattutaVerticale.Rest )
      Contact( #CIn.Rulliera.Sollevamento.Rest )
      Contact( #CIn.Rulliera.Centraggio.Rest )
      Contact( #CIn.Rulliera.Centraggio.Rest )
      Coil( #Ctrl.TRK.BTrk.STOP_PCodaDown_TO_PCoda_Up )
   END_RUNG
   RUNG wire#powerrail
      "BTrk_Presence"(Item := "BTrk".A0302_ENTRY."B"["BTRK_A0302_USCITA_BORDATRICE"])
   END_RUNG wire#w1
   RUNG wire#powerrail
      Contact( #Ctrl.TRK.BTrk.STOP_PCodaDown_TO_PCoda_Up )
      "BTrk_Presence"(Item := "BTrk".A0302_EXIT."B"["BTRK_A0302_RULL_PRIMA_PAREG_CODA_BASSO_STOP"])
      Move(in := "BTrk".A0302_EXIT."B"["BTRK_A0302_RULL_PRIMA_PAREG_CODA_BASSO_STOP"], out1 => "BTrk".A0302_EXIT."B"["BTRK_A0302_RULL_PRIMA_PAREG_CODA_ALTO"])
      "BTrk_Presence"(Item := "BTrk".A0302_EXIT."B"["BTRK_A0302_RULL_PRIMA_PAREG_CODA_ALTO"])
      Move(in := "BTrk".Empty, out1 => "BTrk".A0302_EXIT."B"["BTRK_A0302_RULL_PRIMA_PAREG_CODA_BASSO_STOP"])
   END_RUNG
   RUNG wire#powerrail
      Contact( #Ctrl.TRK.BTrk.STOP_PCodaDown_TO_PCoda_Up )
      "BTrk_Presence"(Item := "BTrk".A0302_ENTRY."B"["BTRK_A0302_USCITA_BORDATRICE"])
      Move(in := "BTrk".A0302_ENTRY."B"["BTRK_A0302_USCITA_BORDATRICE"], out1 => "BTrk".A0302_EXIT."B"["BTRK_A0302_RULL_PRIMA_PAREG_CODA_ALTO"])
      "BTrk_Presence"(Item := "BTrk".A0302_EXIT."B"["BTRK_A0302_RULL_PRIMA_PAREG_CODA_ALTO"])
      Move(in := "BTrk".Empty, out1 => "BTrk".A0302_ENTRY."B"["BTRK_A0302_USCITA_BORDATRICE"])
   END_RUNG
   // the same network as SCL:
   "BTrk_Presence"(Item := "BTrk".A0302_EXIT."B"["BTRK_A0302_RULL_PRIMA_PAREG_CODA_BASSO_STOP"], ENO => #_w1);
   "BTrk_Presence"(Item := "BTrk".A0302_ENTRY."B"["BTRK_A0302_USCITA_BORDATRICE"], ENO => #_w2);
   "BTrk_Absence"(EN := (#_w1 OR #_w2) AND NOT #CIn.Bordatrice.Sens.FTC_Uscita,
                  Item := "BTrk".A0302_EXIT."B"["BTRK_A0302_RULL_PRIMA_PAREG_CODA_ALTO"],
                  ENO => #_w3);
   #Ctrl.TRK.BTrk.STOP_PCodaDown_TO_PCoda_Up := #_w3 AND NOT #Ctrl.TRK.BTrk_ToCheck.Prelievo_RecondGood AND #CIn.CarroPareggCoda.BattutaVerticale.Rest AND #CIn.Rulliera.Sollevamento.Rest AND #CIn.Rulliera.Centraggio.Rest AND #CIn.Rulliera.Centraggio.Rest;
   "BTrk_Presence"(EN := #Ctrl.TRK.BTrk.STOP_PCodaDown_TO_PCoda_Up,
                   Item := "BTrk".A0302_EXIT."B"["BTRK_A0302_RULL_PRIMA_PAREG_CODA_BASSO_STOP"],
                   ENO => #_w4);
   IF #_w4 THEN
       "BTrk".A0302_EXIT."B"["BTRK_A0302_RULL_PRIMA_PAREG_CODA_ALTO"] := "BTrk".A0302_EXIT."B"["BTRK_A0302_RULL_PRIMA_PAREG_CODA_BASSO_STOP"];
   END_IF;
   "BTrk_Presence"(EN := #_w4,
                   Item := "BTrk".A0302_EXIT."B"["BTRK_A0302_RULL_PRIMA_PAREG_CODA_ALTO"],
                   ENO => #_w5);
   IF #_w5 THEN "BTrk".A0302_EXIT."B"["BTRK_A0302_RULL_PRIMA_PAREG_CODA_BASSO_STOP"] := "BTrk".Empty; END_IF;
   "BTrk_Presence"(EN := #Ctrl.TRK.BTrk.STOP_PCodaDown_TO_PCoda_Up,
                   Item := "BTrk".A0302_ENTRY."B"["BTRK_A0302_USCITA_BORDATRICE"],
                   ENO => #_w6);
   IF #_w6 THEN
       "BTrk".A0302_EXIT."B"["BTRK_A0302_RULL_PRIMA_PAREG_CODA_ALTO"] := "BTrk".A0302_ENTRY."B"["BTRK_A0302_USCITA_BORDATRICE"];
   END_IF;
   "BTrk_Presence"(EN := #_w6,
                   Item := "BTrk".A0302_EXIT."B"["BTRK_A0302_RULL_PRIMA_PAREG_CODA_ALTO"],
                   ENO => #_w7);
   IF #_w7 THEN "BTrk".A0302_ENTRY."B"["BTRK_A0302_USCITA_BORDATRICE"] := "BTrk".Empty; END_IF;
END_REGION

REGION Network 76: Paregg. Coda - Movimento BTrk Rull prima P Coda Alto ==a==> Paregg Coda Alto e Beams in Sens S3
   // Pezzo su rulliera (1) + pareggiatore coda alto ed ha incontrato il sensore 3 (in ingresso al pareg.)
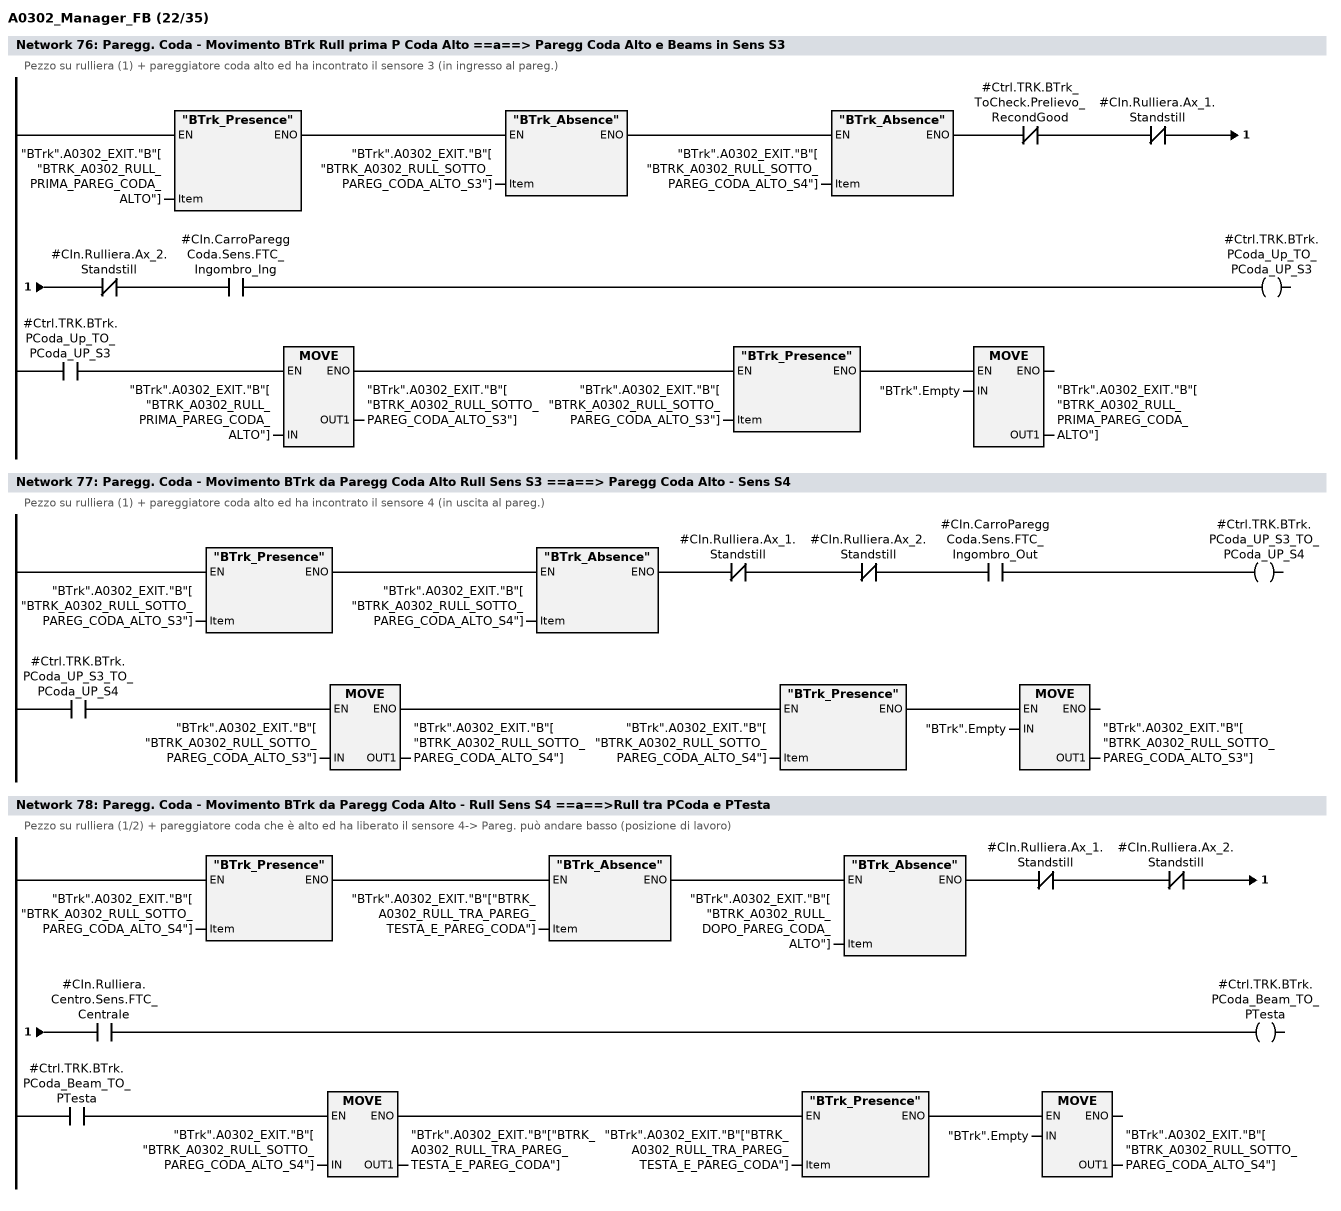
   RUNG wire#powerrail
      "BTrk_Presence"(Item := "BTrk".A0302_EXIT."B"["BTRK_A0302_RULL_PRIMA_PAREG_CODA_ALTO"])
      "BTrk_Absence"(Item := "BTrk".A0302_EXIT."B"["BTRK_A0302_RULL_SOTTO_PAREG_CODA_ALTO_S3"])
      "BTrk_Absence"(Item := "BTrk".A0302_EXIT."B"["BTRK_A0302_RULL_SOTTO_PAREG_CODA_ALTO_S4"])
      I_Contact( #Ctrl.TRK.BTrk_ToCheck.Prelievo_RecondGood )
      I_Contact( #CIn.Rulliera.Ax_1.Standstill )
      I_Contact( #CIn.Rulliera.Ax_2.Standstill )
      Contact( #CIn.CarroPareggCoda.Sens.FTC_Ingombro_Ing )
      Coil( #Ctrl.TRK.BTrk.PCoda_Up_TO_PCoda_UP_S3 )
   END_RUNG
   RUNG wire#powerrail
      Contact( #Ctrl.TRK.BTrk.PCoda_Up_TO_PCoda_UP_S3 )
      Move(in := "BTrk".A0302_EXIT."B"["BTRK_A0302_RULL_PRIMA_PAREG_CODA_ALTO"], out1 => "BTrk".A0302_EXIT."B"["BTRK_A0302_RULL_SOTTO_PAREG_CODA_ALTO_S3"])
      "BTrk_Presence"(Item := "BTrk".A0302_EXIT."B"["BTRK_A0302_RULL_SOTTO_PAREG_CODA_ALTO_S3"])
      Move(in := "BTrk".Empty, out1 => "BTrk".A0302_EXIT."B"["BTRK_A0302_RULL_PRIMA_PAREG_CODA_ALTO"])
   END_RUNG
   // the same network as SCL:
   "BTrk_Presence"(Item := "BTrk".A0302_EXIT."B"["BTRK_A0302_RULL_PRIMA_PAREG_CODA_ALTO"], ENO => #_w1);
   "BTrk_Absence"(EN := #_w1,
                  Item := "BTrk".A0302_EXIT."B"["BTRK_A0302_RULL_SOTTO_PAREG_CODA_ALTO_S3"],
                  ENO => #_w2);
   "BTrk_Absence"(EN := #_w2,
                  Item := "BTrk".A0302_EXIT."B"["BTRK_A0302_RULL_SOTTO_PAREG_CODA_ALTO_S4"],
                  ENO => #_w3);
   #Ctrl.TRK.BTrk.PCoda_Up_TO_PCoda_UP_S3 := #_w3 AND NOT #Ctrl.TRK.BTrk_ToCheck.Prelievo_RecondGood AND NOT #CIn.Rulliera.Ax_1.Standstill AND NOT #CIn.Rulliera.Ax_2.Standstill AND #CIn.CarroPareggCoda.Sens.FTC_Ingombro_Ing;
   IF #Ctrl.TRK.BTrk.PCoda_Up_TO_PCoda_UP_S3 THEN
       "BTrk".A0302_EXIT."B"["BTRK_A0302_RULL_SOTTO_PAREG_CODA_ALTO_S3"] := "BTrk".A0302_EXIT."B"["BTRK_A0302_RULL_PRIMA_PAREG_CODA_ALTO"];
   END_IF;
   "BTrk_Presence"(EN := #Ctrl.TRK.BTrk.PCoda_Up_TO_PCoda_UP_S3,
                   Item := "BTrk".A0302_EXIT."B"["BTRK_A0302_RULL_SOTTO_PAREG_CODA_ALTO_S3"],
                   ENO => #_w4);
   IF #_w4 THEN "BTrk".A0302_EXIT."B"["BTRK_A0302_RULL_PRIMA_PAREG_CODA_ALTO"] := "BTrk".Empty; END_IF;
END_REGION

REGION Network 77: Paregg. Coda - Movimento BTrk da Paregg Coda Alto Rull Sens S3 ==a==> Paregg Coda Alto - Sens S4
   // Pezzo su rulliera (1) + pareggiatore coda alto ed ha incontrato il sensore 4 (in uscita al pareg.)
   RUNG wire#powerrail
      "BTrk_Presence"(Item := "BTrk".A0302_EXIT."B"["BTRK_A0302_RULL_SOTTO_PAREG_CODA_ALTO_S3"])
      "BTrk_Absence"(Item := "BTrk".A0302_EXIT."B"["BTRK_A0302_RULL_SOTTO_PAREG_CODA_ALTO_S4"])
      I_Contact( #CIn.Rulliera.Ax_1.Standstill )
      I_Contact( #CIn.Rulliera.Ax_2.Standstill )
      Contact( #CIn.CarroPareggCoda.Sens.FTC_Ingombro_Out )
      Coil( #Ctrl.TRK.BTrk.PCoda_UP_S3_TO_PCoda_UP_S4 )
   END_RUNG
   RUNG wire#powerrail
      Contact( #Ctrl.TRK.BTrk.PCoda_UP_S3_TO_PCoda_UP_S4 )
      Move(in := "BTrk".A0302_EXIT."B"["BTRK_A0302_RULL_SOTTO_PAREG_CODA_ALTO_S3"], out1 => "BTrk".A0302_EXIT."B"["BTRK_A0302_RULL_SOTTO_PAREG_CODA_ALTO_S4"])
      "BTrk_Presence"(Item := "BTrk".A0302_EXIT."B"["BTRK_A0302_RULL_SOTTO_PAREG_CODA_ALTO_S4"])
      Move(in := "BTrk".Empty, out1 => "BTrk".A0302_EXIT."B"["BTRK_A0302_RULL_SOTTO_PAREG_CODA_ALTO_S3"])
   END_RUNG
   // the same network as SCL:
   "BTrk_Presence"(Item := "BTrk".A0302_EXIT."B"["BTRK_A0302_RULL_SOTTO_PAREG_CODA_ALTO_S3"], ENO => #_w1);
   "BTrk_Absence"(EN := #_w1,
                  Item := "BTrk".A0302_EXIT."B"["BTRK_A0302_RULL_SOTTO_PAREG_CODA_ALTO_S4"],
                  ENO => #_w2);
   #Ctrl.TRK.BTrk.PCoda_UP_S3_TO_PCoda_UP_S4 := #_w2 AND NOT #CIn.Rulliera.Ax_1.Standstill AND NOT #CIn.Rulliera.Ax_2.Standstill AND #CIn.CarroPareggCoda.Sens.FTC_Ingombro_Out;
   IF #Ctrl.TRK.BTrk.PCoda_UP_S3_TO_PCoda_UP_S4 THEN
       "BTrk".A0302_EXIT."B"["BTRK_A0302_RULL_SOTTO_PAREG_CODA_ALTO_S4"] := "BTrk".A0302_EXIT."B"["BTRK_A0302_RULL_SOTTO_PAREG_CODA_ALTO_S3"];
   END_IF;
   "BTrk_Presence"(EN := #Ctrl.TRK.BTrk.PCoda_UP_S3_TO_PCoda_UP_S4,
                   Item := "BTrk".A0302_EXIT."B"["BTRK_A0302_RULL_SOTTO_PAREG_CODA_ALTO_S4"],
                   ENO => #_w3);
   IF #_w3 THEN "BTrk".A0302_EXIT."B"["BTRK_A0302_RULL_SOTTO_PAREG_CODA_ALTO_S3"] := "BTrk".Empty; END_IF;
END_REGION

REGION Network 78: Paregg. Coda - Movimento BTrk da Paregg Coda Alto - Rull Sens S4 ==a==>Rull tra PCoda e PTesta
   // Pezzo su rulliera (1/2) + pareggiatore coda che è alto ed ha liberato il sensore 4-> Pareg. può andare basso (posizione di lavoro)
   RUNG wire#powerrail
      "BTrk_Presence"(Item := "BTrk".A0302_EXIT."B"["BTRK_A0302_RULL_SOTTO_PAREG_CODA_ALTO_S4"])
      "BTrk_Absence"(Item := "BTrk".A0302_EXIT."B"["BTRK_A0302_RULL_TRA_PAREG_TESTA_E_PAREG_CODA"])
      "BTrk_Absence"(Item := "BTrk".A0302_EXIT."B"["BTRK_A0302_RULL_DOPO_PAREG_CODA_ALTO"])
      I_Contact( #CIn.Rulliera.Ax_1.Standstill )
      I_Contact( #CIn.Rulliera.Ax_2.Standstill )
      Contact( #CIn.Rulliera.Centro.Sens.FTC_Centrale )
      Coil( #Ctrl.TRK.BTrk.PCoda_Beam_TO_PTesta )
   END_RUNG
   RUNG wire#powerrail
      Contact( #Ctrl.TRK.BTrk.PCoda_Beam_TO_PTesta )
      Move(in := "BTrk".A0302_EXIT."B"["BTRK_A0302_RULL_SOTTO_PAREG_CODA_ALTO_S4"], out1 => "BTrk".A0302_EXIT."B"["BTRK_A0302_RULL_TRA_PAREG_TESTA_E_PAREG_CODA"])
      "BTrk_Presence"(Item := "BTrk".A0302_EXIT."B"["BTRK_A0302_RULL_TRA_PAREG_TESTA_E_PAREG_CODA"])
      Move(in := "BTrk".Empty, out1 => "BTrk".A0302_EXIT."B"["BTRK_A0302_RULL_SOTTO_PAREG_CODA_ALTO_S4"])
   END_RUNG
   // the same network as SCL:
   "BTrk_Presence"(Item := "BTrk".A0302_EXIT."B"["BTRK_A0302_RULL_SOTTO_PAREG_CODA_ALTO_S4"], ENO => #_w1);
   "BTrk_Absence"(EN := #_w1,
                  Item := "BTrk".A0302_EXIT."B"["BTRK_A0302_RULL_TRA_PAREG_TESTA_E_PAREG_CODA"],
                  ENO => #_w2);
   "BTrk_Absence"(EN := #_w2,
                  Item := "BTrk".A0302_EXIT."B"["BTRK_A0302_RULL_DOPO_PAREG_CODA_ALTO"],
                  ENO => #_w3);
   #Ctrl.TRK.BTrk.PCoda_Beam_TO_PTesta := #_w3 AND NOT #CIn.Rulliera.Ax_1.Standstill AND NOT #CIn.Rulliera.Ax_2.Standstill AND #CIn.Rulliera.Centro.Sens.FTC_Centrale;
   IF #Ctrl.TRK.BTrk.PCoda_Beam_TO_PTesta THEN
       "BTrk".A0302_EXIT."B"["BTRK_A0302_RULL_TRA_PAREG_TESTA_E_PAREG_CODA"] := "BTrk".A0302_EXIT."B"["BTRK_A0302_RULL_SOTTO_PAREG_CODA_ALTO_S4"];
   END_IF;
   "BTrk_Presence"(EN := #Ctrl.TRK.BTrk.PCoda_Beam_TO_PTesta,
                   Item := "BTrk".A0302_EXIT."B"["BTRK_A0302_RULL_TRA_PAREG_TESTA_E_PAREG_CODA"],
                   ENO => #_w4);
   IF #_w4 THEN "BTrk".A0302_EXIT."B"["BTRK_A0302_RULL_SOTTO_PAREG_CODA_ALTO_S4"] := "BTrk".Empty; END_IF;
END_REGION

REGION Network 79: Paregg. Coda - Movimento BTrk tra Rull PCoda e PTesta => Rull dopo PCoda alto
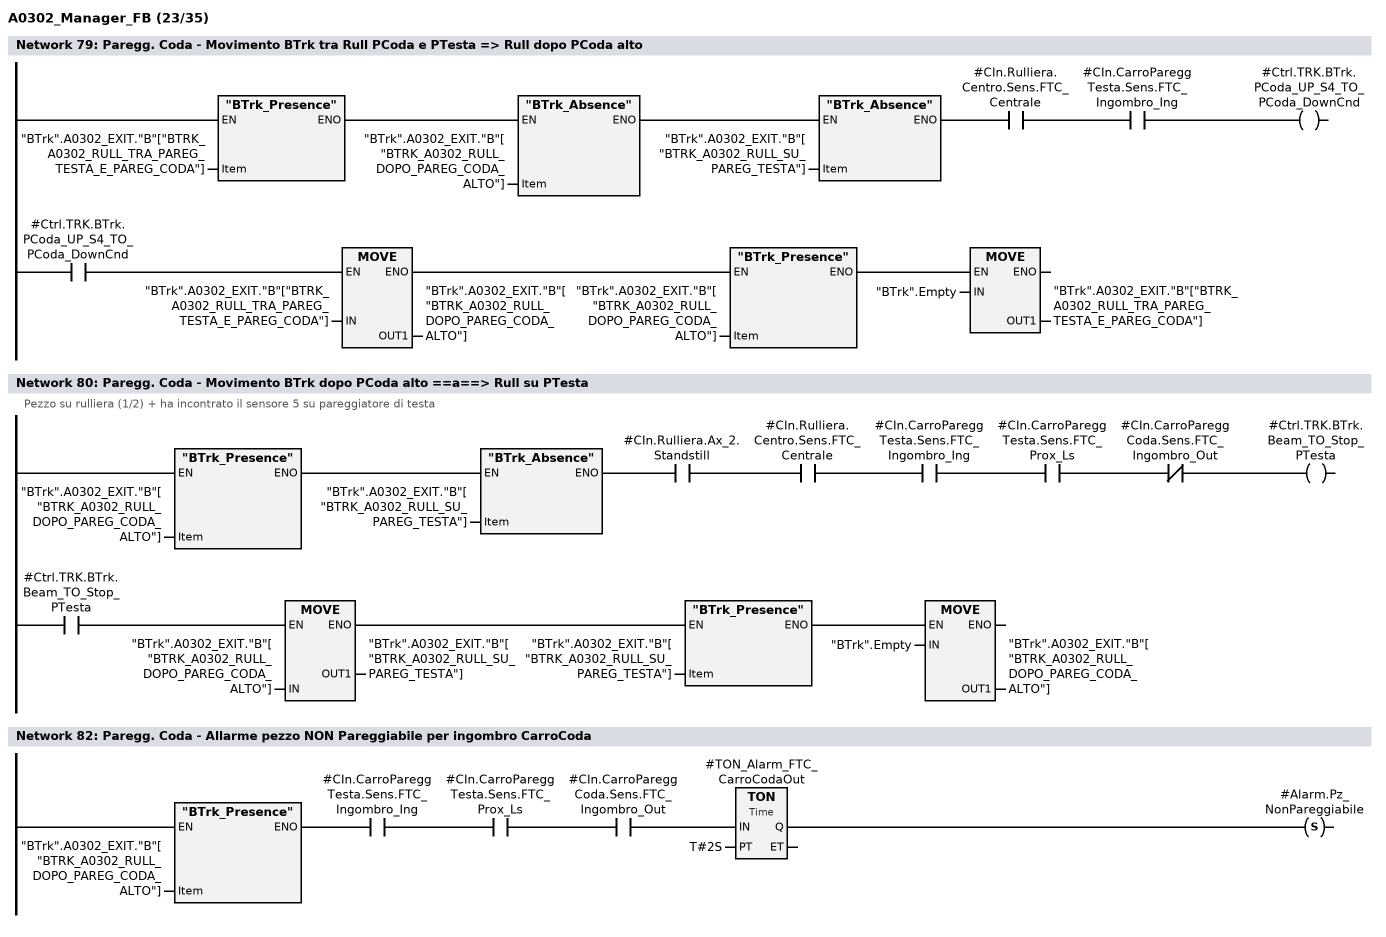
   RUNG wire#powerrail
      "BTrk_Presence"(Item := "BTrk".A0302_EXIT."B"["BTRK_A0302_RULL_TRA_PAREG_TESTA_E_PAREG_CODA"])
      "BTrk_Absence"(Item := "BTrk".A0302_EXIT."B"["BTRK_A0302_RULL_DOPO_PAREG_CODA_ALTO"])
      "BTrk_Absence"(Item := "BTrk".A0302_EXIT."B"["BTRK_A0302_RULL_SU_PAREG_TESTA"])
      Contact( #CIn.Rulliera.Centro.Sens.FTC_Centrale )
      Contact( #CIn.CarroPareggTesta.Sens.FTC_Ingombro_Ing )
      Coil( #Ctrl.TRK.BTrk.PCoda_UP_S4_TO_PCoda_DownCnd )
   END_RUNG
   RUNG wire#powerrail
      Contact( #Ctrl.TRK.BTrk.PCoda_UP_S4_TO_PCoda_DownCnd )
      Move(in := "BTrk".A0302_EXIT."B"["BTRK_A0302_RULL_TRA_PAREG_TESTA_E_PAREG_CODA"], out1 => "BTrk".A0302_EXIT."B"["BTRK_A0302_RULL_DOPO_PAREG_CODA_ALTO"])
      "BTrk_Presence"(Item := "BTrk".A0302_EXIT."B"["BTRK_A0302_RULL_DOPO_PAREG_CODA_ALTO"])
      Move(in := "BTrk".Empty, out1 => "BTrk".A0302_EXIT."B"["BTRK_A0302_RULL_TRA_PAREG_TESTA_E_PAREG_CODA"])
   END_RUNG
   // the same network as SCL:
   "BTrk_Presence"(Item := "BTrk".A0302_EXIT."B"["BTRK_A0302_RULL_TRA_PAREG_TESTA_E_PAREG_CODA"], ENO => #_w1);
   "BTrk_Absence"(EN := #_w1,
                  Item := "BTrk".A0302_EXIT."B"["BTRK_A0302_RULL_DOPO_PAREG_CODA_ALTO"],
                  ENO => #_w2);
   "BTrk_Absence"(EN := #_w2, Item := "BTrk".A0302_EXIT."B"["BTRK_A0302_RULL_SU_PAREG_TESTA"], ENO => #_w3);
   #Ctrl.TRK.BTrk.PCoda_UP_S4_TO_PCoda_DownCnd := #_w3 AND #CIn.Rulliera.Centro.Sens.FTC_Centrale AND #CIn.CarroPareggTesta.Sens.FTC_Ingombro_Ing;
   IF #Ctrl.TRK.BTrk.PCoda_UP_S4_TO_PCoda_DownCnd THEN
       "BTrk".A0302_EXIT."B"["BTRK_A0302_RULL_DOPO_PAREG_CODA_ALTO"] := "BTrk".A0302_EXIT."B"["BTRK_A0302_RULL_TRA_PAREG_TESTA_E_PAREG_CODA"];
   END_IF;
   "BTrk_Presence"(EN := #Ctrl.TRK.BTrk.PCoda_UP_S4_TO_PCoda_DownCnd,
                   Item := "BTrk".A0302_EXIT."B"["BTRK_A0302_RULL_DOPO_PAREG_CODA_ALTO"],
                   ENO => #_w4);
   IF #_w4 THEN
       "BTrk".A0302_EXIT."B"["BTRK_A0302_RULL_TRA_PAREG_TESTA_E_PAREG_CODA"] := "BTrk".Empty;
   END_IF;
END_REGION

REGION Network 80: Paregg. Coda - Movimento BTrk dopo PCoda alto ==a==> Rull su PTesta
   // Pezzo su rulliera (1/2) + ha incontrato il sensore 5 su pareggiatore di testa
   RUNG wire#powerrail
      "BTrk_Presence"(Item := "BTrk".A0302_EXIT."B"["BTRK_A0302_RULL_DOPO_PAREG_CODA_ALTO"])
      "BTrk_Absence"(Item := "BTrk".A0302_EXIT."B"["BTRK_A0302_RULL_SU_PAREG_TESTA"])
      Contact( #CIn.Rulliera.Ax_2.Standstill )
      Contact( #CIn.Rulliera.Centro.Sens.FTC_Centrale )
      Contact( #CIn.CarroPareggTesta.Sens.FTC_Ingombro_Ing )
      Contact( #CIn.CarroPareggTesta.Sens.FTC_Prox_Ls )
      I_Contact( #CIn.CarroPareggCoda.Sens.FTC_Ingombro_Out )
      Coil( #Ctrl.TRK.BTrk.Beam_TO_Stop_PTesta )
   END_RUNG
   RUNG wire#powerrail
      Contact( #Ctrl.TRK.BTrk.Beam_TO_Stop_PTesta )
      Move(in := "BTrk".A0302_EXIT."B"["BTRK_A0302_RULL_DOPO_PAREG_CODA_ALTO"], out1 => "BTrk".A0302_EXIT."B"["BTRK_A0302_RULL_SU_PAREG_TESTA"])
      "BTrk_Presence"(Item := "BTrk".A0302_EXIT."B"["BTRK_A0302_RULL_SU_PAREG_TESTA"])
      Move(in := "BTrk".Empty, out1 => "BTrk".A0302_EXIT."B"["BTRK_A0302_RULL_DOPO_PAREG_CODA_ALTO"])
   END_RUNG
   // the same network as SCL:
   "BTrk_Presence"(Item := "BTrk".A0302_EXIT."B"["BTRK_A0302_RULL_DOPO_PAREG_CODA_ALTO"], ENO => #_w1);
   "BTrk_Absence"(EN := #_w1, Item := "BTrk".A0302_EXIT."B"["BTRK_A0302_RULL_SU_PAREG_TESTA"], ENO => #_w2);
   #Ctrl.TRK.BTrk.Beam_TO_Stop_PTesta := #_w2 AND #CIn.Rulliera.Ax_2.Standstill AND #CIn.Rulliera.Centro.Sens.FTC_Centrale AND #CIn.CarroPareggTesta.Sens.FTC_Ingombro_Ing AND #CIn.CarroPareggTesta.Sens.FTC_Prox_Ls AND NOT #CIn.CarroPareggCoda.Sens.FTC_Ingombro_Out;
   IF #Ctrl.TRK.BTrk.Beam_TO_Stop_PTesta THEN
       "BTrk".A0302_EXIT."B"["BTRK_A0302_RULL_SU_PAREG_TESTA"] := "BTrk".A0302_EXIT."B"["BTRK_A0302_RULL_DOPO_PAREG_CODA_ALTO"];
   END_IF;
   "BTrk_Presence"(EN := #Ctrl.TRK.BTrk.Beam_TO_Stop_PTesta,
                   Item := "BTrk".A0302_EXIT."B"["BTRK_A0302_RULL_SU_PAREG_TESTA"],
                   ENO => #_w3);
   IF #_w3 THEN "BTrk".A0302_EXIT."B"["BTRK_A0302_RULL_DOPO_PAREG_CODA_ALTO"] := "BTrk".Empty; END_IF;
END_REGION

REGION Network 81: <+>
END_REGION

REGION Network 82: Paregg. Coda - Allarme pezzo NON Pareggiabile per ingombro CarroCoda
   RUNG wire#powerrail
      "BTrk_Presence"(Item := "BTrk".A0302_EXIT."B"["BTRK_A0302_RULL_DOPO_PAREG_CODA_ALTO"])
      Contact( #CIn.CarroPareggTesta.Sens.FTC_Ingombro_Ing )
      Contact( #CIn.CarroPareggTesta.Sens.FTC_Prox_Ls )
      Contact( #CIn.CarroPareggCoda.Sens.FTC_Ingombro_Out )
      { S7_Templates := "time_type := Time" } #TON_Alarm_FTC_CarroCodaOut.TON(pt := T#2S, et =>)
      S_Coil( #Alarm.Pz_NonPareggiabile )
   END_RUNG
   // the same network as SCL:
   "BTrk_Presence"(Item := "BTrk".A0302_EXIT."B"["BTRK_A0302_RULL_DOPO_PAREG_CODA_ALTO"], ENO => #_w1);
   #TON_Alarm_FTC_CarroCodaOut.TON(IN := #_w1 AND #CIn.CarroPareggTesta.Sens.FTC_Ingombro_Ing AND #CIn.CarroPareggTesta.Sens.FTC_Prox_Ls AND #CIn.CarroPareggCoda.Sens.FTC_Ingombro_Out,
                           PT := T#2S);
   IF #TON_Alarm_FTC_CarroCodaOut.Q THEN #Alarm.Pz_NonPareggiabile := TRUE; END_IF;
END_REGION

REGION Network 83: <+>
END_REGION

REGION Network 84: Paregg. Coda [Battuta Vrt] - Movimento operazione a lavoro / a riposo
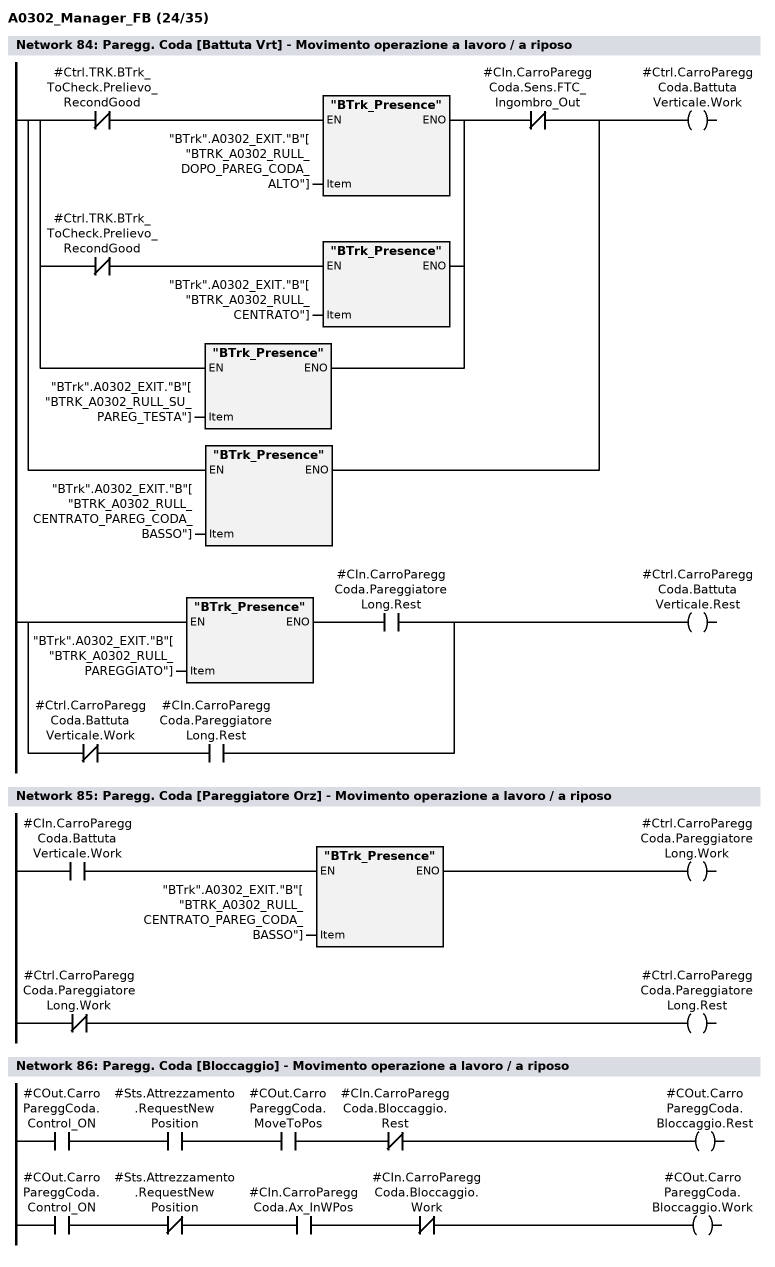
   RUNG wire#powerrail
      I_Contact( #Ctrl.TRK.BTrk_ToCheck.Prelievo_RecondGood )
      "BTrk_Presence"(Item := "BTrk".A0302_EXIT."B"["BTRK_A0302_RULL_DOPO_PAREG_CODA_ALTO"])
      wire#w1
      I_Contact( #CIn.CarroPareggCoda.Sens.FTC_Ingombro_Out )
      wire#w2
      Coil( #Ctrl.CarroPareggCoda.BattutaVerticale.Work )
   END_RUNG
   RUNG wire#powerrail
      I_Contact( #Ctrl.TRK.BTrk_ToCheck.Prelievo_RecondGood )
      "BTrk_Presence"(Item := "BTrk".A0302_EXIT."B"["BTRK_A0302_RULL_CENTRATO"])
   END_RUNG wire#w1
   RUNG wire#powerrail
      "BTrk_Presence"(Item := "BTrk".A0302_EXIT."B"["BTRK_A0302_RULL_SU_PAREG_TESTA"])
   END_RUNG wire#w1
   RUNG wire#powerrail
      "BTrk_Presence"(Item := "BTrk".A0302_EXIT."B"["BTRK_A0302_RULL_CENTRATO_PAREG_CODA_BASSO"])
   END_RUNG wire#w2
   RUNG wire#powerrail
      "BTrk_Presence"(Item := "BTrk".A0302_EXIT."B"["BTRK_A0302_RULL_PAREGGIATO"])
      Contact( #CIn.CarroPareggCoda.PareggiatoreLong.Rest )
      wire#w3
      Coil( #Ctrl.CarroPareggCoda.BattutaVerticale.Rest )
   END_RUNG
   RUNG wire#powerrail
      I_Contact( #Ctrl.CarroPareggCoda.BattutaVerticale.Work )
      Contact( #CIn.CarroPareggCoda.PareggiatoreLong.Rest )
   END_RUNG wire#w3
   // the same network as SCL:
   "BTrk_Presence"(EN := NOT #Ctrl.TRK.BTrk_ToCheck.Prelievo_RecondGood,
                   Item := "BTrk".A0302_EXIT."B"["BTRK_A0302_RULL_DOPO_PAREG_CODA_ALTO"],
                   ENO => #_w1);
   "BTrk_Presence"(EN := NOT #Ctrl.TRK.BTrk_ToCheck.Prelievo_RecondGood,
                   Item := "BTrk".A0302_EXIT."B"["BTRK_A0302_RULL_CENTRATO"],
                   ENO => #_w2);
   "BTrk_Presence"(Item := "BTrk".A0302_EXIT."B"["BTRK_A0302_RULL_SU_PAREG_TESTA"], ENO => #_w3);
   "BTrk_Presence"(Item := "BTrk".A0302_EXIT."B"["BTRK_A0302_RULL_CENTRATO_PAREG_CODA_BASSO"], ENO => #_w4);
   #Ctrl.CarroPareggCoda.BattutaVerticale.Work := ((#_w1 OR #_w2 OR #_w3) AND NOT #CIn.CarroPareggCoda.Sens.FTC_Ingombro_Out) OR #_w4;
   "BTrk_Presence"(Item := "BTrk".A0302_EXIT."B"["BTRK_A0302_RULL_PAREGGIATO"], ENO => #_w5);
   #Ctrl.CarroPareggCoda.BattutaVerticale.Rest := (#_w5 AND #CIn.CarroPareggCoda.PareggiatoreLong.Rest) OR (NOT #Ctrl.CarroPareggCoda.BattutaVerticale.Work AND #CIn.CarroPareggCoda.PareggiatoreLong.Rest);
END_REGION

REGION Network 85: Paregg. Coda [Pareggiatore Orz] - Movimento operazione a lavoro / a riposo
   RUNG wire#powerrail
      Contact( #CIn.CarroPareggCoda.BattutaVerticale.Work )
      "BTrk_Presence"(Item := "BTrk".A0302_EXIT."B"["BTRK_A0302_RULL_CENTRATO_PAREG_CODA_BASSO"])
      Coil( #Ctrl.CarroPareggCoda.PareggiatoreLong.Work )
   END_RUNG
   RUNG wire#powerrail
      I_Contact( #Ctrl.CarroPareggCoda.PareggiatoreLong.Work )
      Coil( #Ctrl.CarroPareggCoda.PareggiatoreLong.Rest )
   END_RUNG
   // the same network as SCL:
   "BTrk_Presence"(EN := #CIn.CarroPareggCoda.BattutaVerticale.Work,
                   Item := "BTrk".A0302_EXIT."B"["BTRK_A0302_RULL_CENTRATO_PAREG_CODA_BASSO"],
                   ENO => #_w1);
   #Ctrl.CarroPareggCoda.PareggiatoreLong.Work := #_w1;
   #Ctrl.CarroPareggCoda.PareggiatoreLong.Rest := NOT #Ctrl.CarroPareggCoda.PareggiatoreLong.Work;
END_REGION

REGION Network 86: Paregg. Coda [Bloccaggio] - Movimento operazione a lavoro / a riposo
   RUNG wire#powerrail
      Contact( #COut.CarroPareggCoda.Control_ON )
      Contact( #Sts.Attrezzamento.RequestNewPosition )
      Contact( #COut.CarroPareggCoda.MoveToPos )
      I_Contact( #CIn.CarroPareggCoda.Bloccaggio.Rest )
      Coil( #COut.CarroPareggCoda.Bloccaggio.Rest )
   END_RUNG
   RUNG wire#powerrail
      Contact( #COut.CarroPareggCoda.Control_ON )
      I_Contact( #Sts.Attrezzamento.RequestNewPosition )
      Contact( #CIn.CarroPareggCoda.Ax_InWPos )
      I_Contact( #CIn.CarroPareggCoda.Bloccaggio.Work )
      Coil( #COut.CarroPareggCoda.Bloccaggio.Work )
   END_RUNG
   // the same network as SCL:
   #COut.CarroPareggCoda.Bloccaggio.Rest := #COut.CarroPareggCoda.Control_ON AND #Sts.Attrezzamento.RequestNewPosition AND #COut.CarroPareggCoda.MoveToPos AND NOT #CIn.CarroPareggCoda.Bloccaggio.Rest;
   #COut.CarroPareggCoda.Bloccaggio.Work := #COut.CarroPareggCoda.Control_ON AND NOT #Sts.Attrezzamento.RequestNewPosition AND #CIn.CarroPareggCoda.Ax_InWPos AND NOT #CIn.CarroPareggCoda.Bloccaggio.Work;
END_REGION

REGION Network 87: <+>
END_REGION

REGION Network 88: Carro Pareggiatore Coda - COut Manager
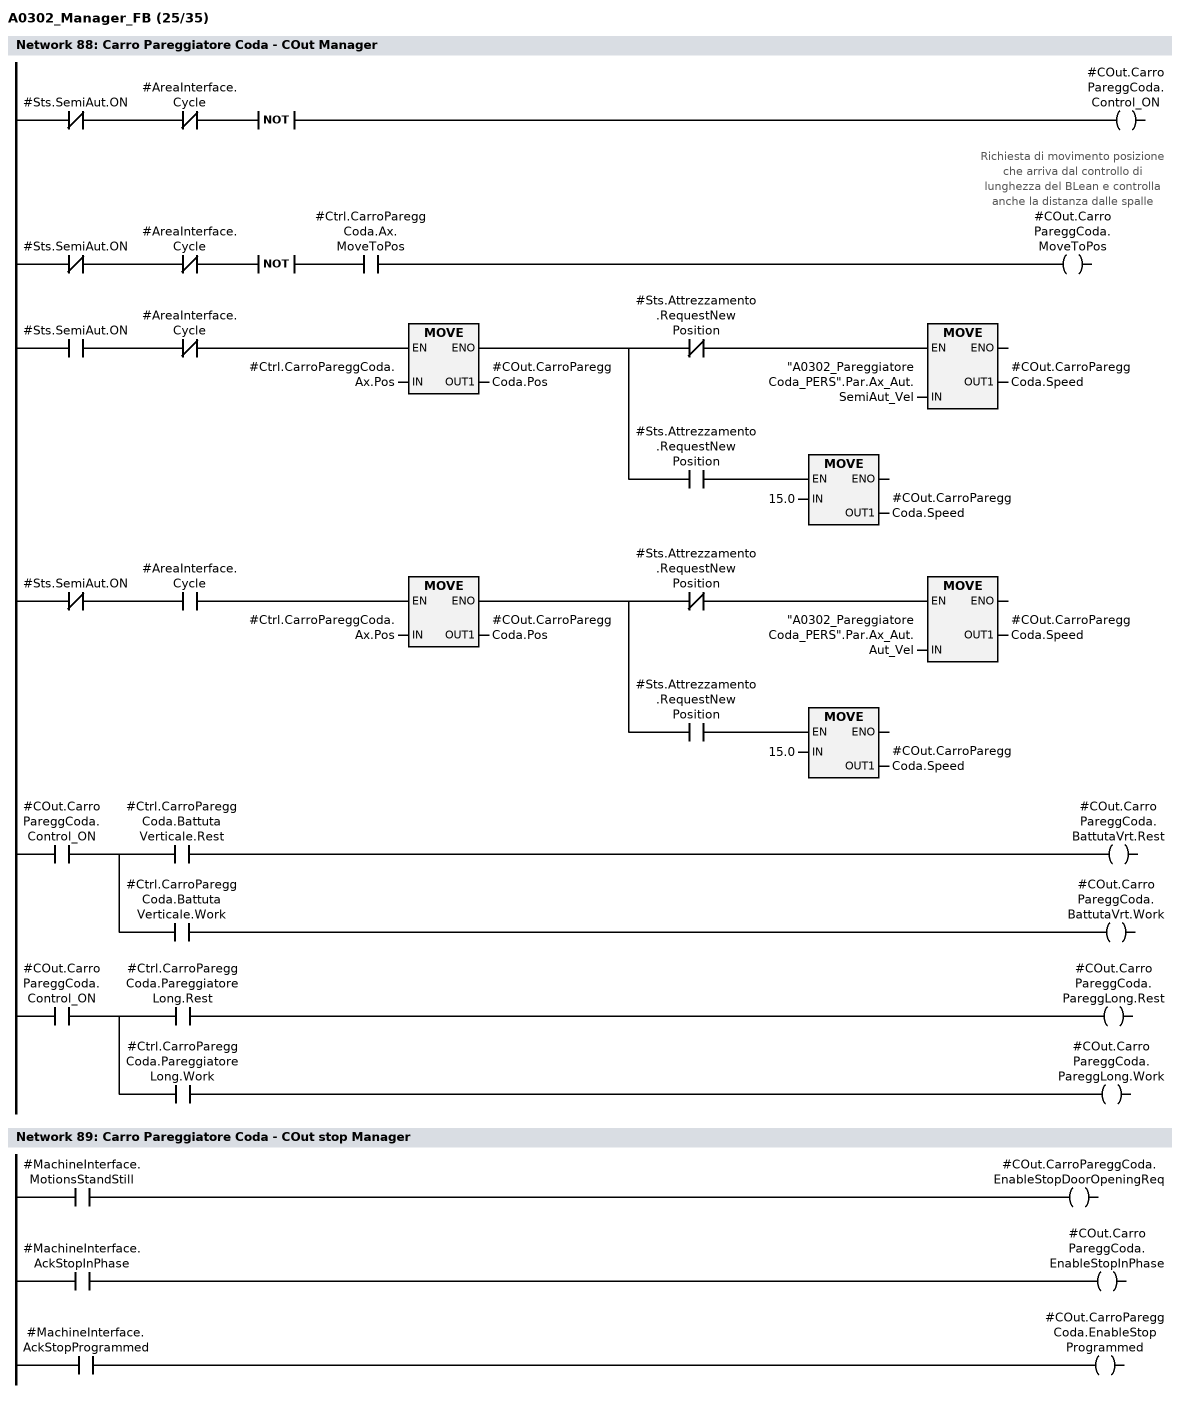
   RUNG wire#powerrail
      I_Contact( #Sts.SemiAut.ON )
      I_Contact( #AreaInterface.Cycle )
      Not()
      Coil( #COut.CarroPareggCoda.Control_ON )
   END_RUNG
   RUNG wire#powerrail
      I_Contact( #Sts.SemiAut.ON )
      I_Contact( #AreaInterface.Cycle )
      Not()
      Contact( #Ctrl.CarroPareggCoda.Ax.MoveToPos )
      Coil( #COut.CarroPareggCoda.MoveToPos )   // Richiesta di movimento posizione che arriva dal controllo di lunghezza del BLean e controlla anche la distanza dalle spalle
   END_RUNG
   RUNG wire#powerrail
      Contact( #Sts.SemiAut.ON )
      I_Contact( #AreaInterface.Cycle )
      Move(in := #Ctrl.CarroPareggCoda.Ax.Pos, out1 => #COut.CarroPareggCoda.Pos)
      wire#w1
      I_Contact( #Sts.Attrezzamento.RequestNewPosition )
      Move(in := "A0302_PareggiatoreCoda_PERS".Par.Ax_Aut.SemiAut_Vel, out1 => #COut.CarroPareggCoda.Speed)
   END_RUNG
   RUNG wire#w1
      Contact( #Sts.Attrezzamento.RequestNewPosition )
      Move(in := 15.0, out1 => #COut.CarroPareggCoda.Speed)
   END_RUNG
   RUNG wire#powerrail
      I_Contact( #Sts.SemiAut.ON )
      Contact( #AreaInterface.Cycle )
      Move(in := #Ctrl.CarroPareggCoda.Ax.Pos, out1 => #COut.CarroPareggCoda.Pos)
      wire#w2
      I_Contact( #Sts.Attrezzamento.RequestNewPosition )
      Move(in := "A0302_PareggiatoreCoda_PERS".Par.Ax_Aut.Aut_Vel, out1 => #COut.CarroPareggCoda.Speed)
   END_RUNG
   RUNG wire#w2
      Contact( #Sts.Attrezzamento.RequestNewPosition )
      Move(in := 15.0, out1 => #COut.CarroPareggCoda.Speed)
   END_RUNG
   RUNG wire#powerrail
      Contact( #COut.CarroPareggCoda.Control_ON )
      wire#w3
      Contact( #Ctrl.CarroPareggCoda.BattutaVerticale.Rest )
      Coil( #COut.CarroPareggCoda.BattutaVrt.Rest )
   END_RUNG
   RUNG wire#w3
      Contact( #Ctrl.CarroPareggCoda.BattutaVerticale.Work )
      Coil( #COut.CarroPareggCoda.BattutaVrt.Work )
   END_RUNG
   RUNG wire#powerrail
      Contact( #COut.CarroPareggCoda.Control_ON )
      wire#w4
      Contact( #Ctrl.CarroPareggCoda.PareggiatoreLong.Rest )
      Coil( #COut.CarroPareggCoda.PareggLong.Rest )
   END_RUNG
   RUNG wire#w4
      Contact( #Ctrl.CarroPareggCoda.PareggiatoreLong.Work )
      Coil( #COut.CarroPareggCoda.PareggLong.Work )
   END_RUNG
   // the same network as SCL:
   #COut.CarroPareggCoda.Control_ON := NOT (NOT #Sts.SemiAut.ON AND NOT #AreaInterface.Cycle);
   #COut.CarroPareggCoda.MoveToPos := NOT (NOT #Sts.SemiAut.ON AND NOT #AreaInterface.Cycle) AND #Ctrl.CarroPareggCoda.Ax.MoveToPos;   // Richiesta di movimento posizione che arriva dal controllo di lunghezza del BLean e controlla anche la distanza dalle spalle
   #_w1 := #Sts.SemiAut.ON AND NOT #AreaInterface.Cycle;
   IF #_w1 THEN #COut.CarroPareggCoda.Pos := #Ctrl.CarroPareggCoda.Ax.Pos; END_IF;
   IF #_w1 AND NOT #Sts.Attrezzamento.RequestNewPosition THEN
       #COut.CarroPareggCoda.Speed := "A0302_PareggiatoreCoda_PERS".Par.Ax_Aut.SemiAut_Vel;
   END_IF;
   IF #_w1 AND #Sts.Attrezzamento.RequestNewPosition THEN #COut.CarroPareggCoda.Speed := 15.0; END_IF;
   #_w2 := NOT #Sts.SemiAut.ON AND #AreaInterface.Cycle;
   IF #_w2 THEN #COut.CarroPareggCoda.Pos := #Ctrl.CarroPareggCoda.Ax.Pos; END_IF;
   IF #_w2 AND NOT #Sts.Attrezzamento.RequestNewPosition THEN
       #COut.CarroPareggCoda.Speed := "A0302_PareggiatoreCoda_PERS".Par.Ax_Aut.Aut_Vel;
   END_IF;
   IF #_w2 AND #Sts.Attrezzamento.RequestNewPosition THEN #COut.CarroPareggCoda.Speed := 15.0; END_IF;
   #COut.CarroPareggCoda.BattutaVrt.Rest := #COut.CarroPareggCoda.Control_ON AND #Ctrl.CarroPareggCoda.BattutaVerticale.Rest;
   #COut.CarroPareggCoda.BattutaVrt.Work := #COut.CarroPareggCoda.Control_ON AND #Ctrl.CarroPareggCoda.BattutaVerticale.Work;
   #COut.CarroPareggCoda.PareggLong.Rest := #COut.CarroPareggCoda.Control_ON AND #Ctrl.CarroPareggCoda.PareggiatoreLong.Rest;
   #COut.CarroPareggCoda.PareggLong.Work := #COut.CarroPareggCoda.Control_ON AND #Ctrl.CarroPareggCoda.PareggiatoreLong.Work;
END_REGION

REGION Network 89: Carro Pareggiatore Coda - COut stop Manager
   RUNG wire#powerrail
      Contact( #MachineInterface.MotionsStandStill )
      Coil( #COut.CarroPareggCoda.EnableStopDoorOpeningReq )
   END_RUNG
   RUNG wire#powerrail
      Contact( #MachineInterface.AckStopInPhase )
      Coil( #COut.CarroPareggCoda.EnableStopInPhase )
   END_RUNG
   RUNG wire#powerrail
      Contact( #MachineInterface.AckStopProgrammed )
      Coil( #COut.CarroPareggCoda.EnableStopProgrammed )
   END_RUNG
   // the same network as SCL:
   #COut.CarroPareggCoda.EnableStopDoorOpeningReq := #MachineInterface.MotionsStandStill;
   #COut.CarroPareggCoda.EnableStopInPhase := #MachineInterface.AckStopInPhase;
   #COut.CarroPareggCoda.EnableStopProgrammed := #MachineInterface.AckStopProgrammed;
END_REGION

REGION Network 90: ************************************************************************************
END_REGION

REGION Network 91: HU Cytropack - COut Manager
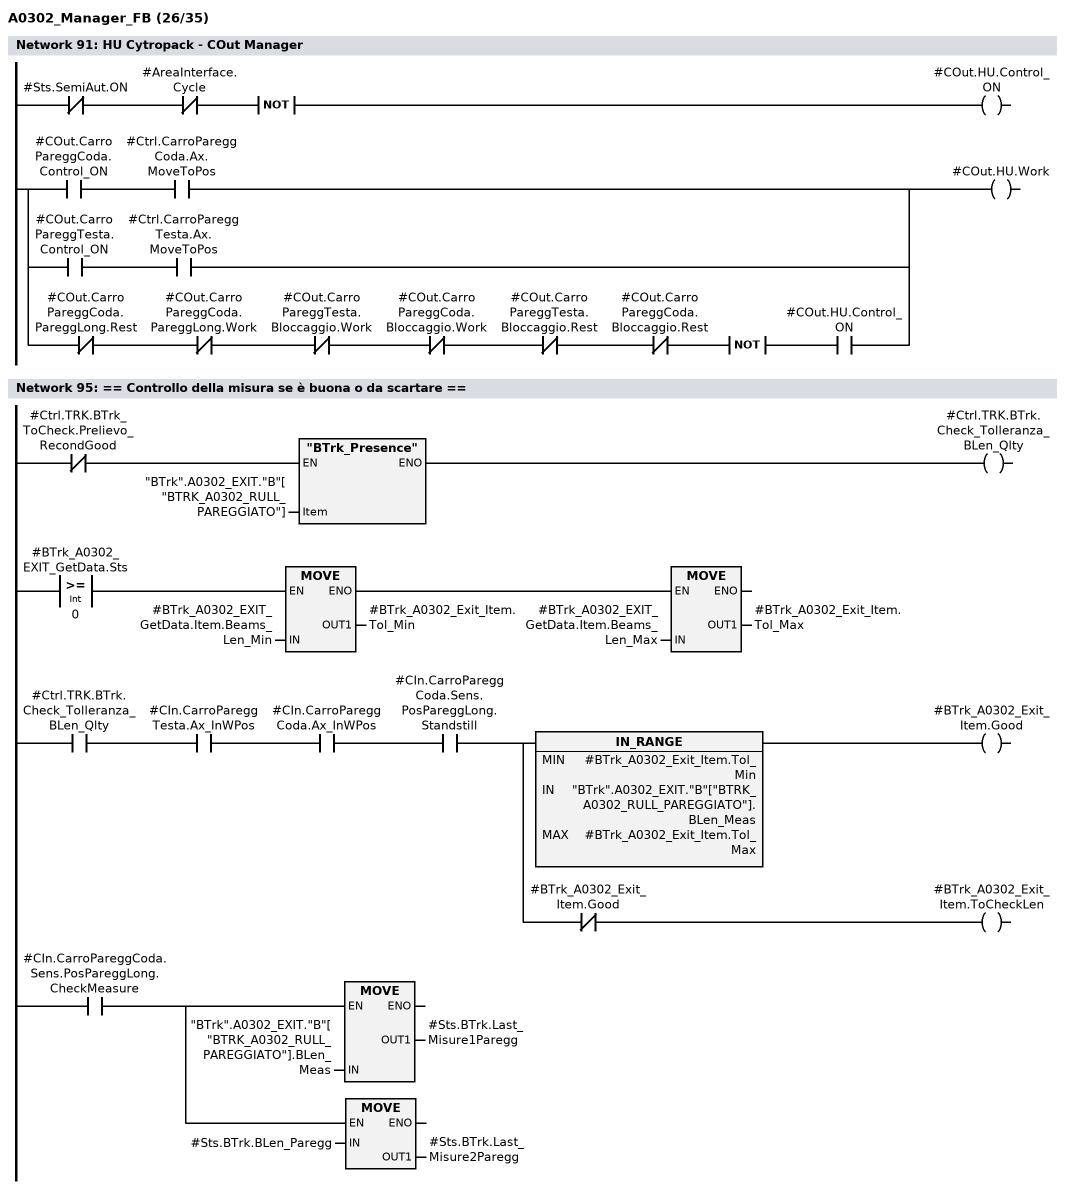
   RUNG wire#powerrail
      I_Contact( #Sts.SemiAut.ON )
      I_Contact( #AreaInterface.Cycle )
      Not()
      Coil( #COut.HU.Control_ON )
   END_RUNG
   RUNG wire#powerrail
      Contact( #COut.CarroPareggCoda.Control_ON )
      Contact( #Ctrl.CarroPareggCoda.Ax.MoveToPos )
      wire#w1
      Coil( #COut.HU.Work )
   END_RUNG
   RUNG wire#powerrail
      Contact( #COut.CarroPareggTesta.Control_ON )
      Contact( #Ctrl.CarroPareggTesta.Ax.MoveToPos )
   END_RUNG wire#w1
   RUNG wire#powerrail
      I_Contact( #COut.CarroPareggCoda.PareggLong.Rest )
      I_Contact( #COut.CarroPareggCoda.PareggLong.Work )
      I_Contact( #COut.CarroPareggTesta.Bloccaggio.Work )
      I_Contact( #COut.CarroPareggCoda.Bloccaggio.Work )
      I_Contact( #COut.CarroPareggTesta.Bloccaggio.Rest )
      I_Contact( #COut.CarroPareggCoda.Bloccaggio.Rest )
      Not()
      Contact( #COut.HU.Control_ON )
   END_RUNG wire#w1
   // the same network as SCL:
   #COut.HU.Control_ON := NOT (NOT #Sts.SemiAut.ON AND NOT #AreaInterface.Cycle);
   #COut.HU.Work := (#COut.CarroPareggCoda.Control_ON AND #Ctrl.CarroPareggCoda.Ax.MoveToPos) OR (#COut.CarroPareggTesta.Control_ON AND #Ctrl.CarroPareggTesta.Ax.MoveToPos) OR (NOT (NOT #COut.CarroPareggCoda.PareggLong.Rest AND NOT #COut.CarroPareggCoda.PareggLong.Work AND NOT #COut.CarroPareggTesta.Bloccaggio.Work AND NOT #COut.CarroPareggCoda.Bloccaggio.Work AND NOT #COut.CarroPareggTesta.Bloccaggio.Rest AND NOT #COut.CarroPareggCoda.Bloccaggio.Rest) AND #COut.HU.Control_ON);
END_REGION

REGION Network 92: **********************************************************************************
END_REGION

REGION Network 93: <<<<< CONTROLLO MISURA DEL BEAMS >>>>>>
END_REGION

REGION Network 94 (SCL): == Lettura del Beam pareggiato ==
   // Controllo della misura del beam misurata


   IF NOT #Ctrl.TRK.BTrk_ToCheck.Prelievo_RecondGood THEN

       // Salvo misura con Offset gioco
       IF #CIn.CarroPareggTesta.Ax_InWPos AND #CIn.CarroPareggCoda.Ax_InWPos
           AND (#Ctrl.TRK.BTrk.Cnd_PareggCoda_TO_Pareggiato OR "A03_DEBUG".A0302_Manager.PareggiaRead) THEN
           "BTrk".A0302_EXIT.B[BTRK_A0302_RULL_CENTRATO_PAREG_CODA_BASSO].BLen_Meas :=
           LREAL_TO_REAL(IN := (#CIn.CarroPareggCoda.Ax.ActualPosition + #CIn.CarroPareggTesta.Ax.ActualPosition) - #CIn.CarroPareggCoda.Sens.PosPareggLong.Value) - #OffsetGioco;
       END_IF;

       // Salvo misura senza Offset gioco
       IF #CIn.CarroPareggTesta.Ax_InWPos AND #CIn.CarroPareggCoda.Ax_InWPos
           AND (#Ctrl.TRK.BTrk.Cnd_PareggCoda_TO_Pareggiato OR "A03_DEBUG".A0302_Manager.PareggiaRead) THEN
           #Sts.BTrk.BLen_Paregg :=LREAL_TO_REAL(IN := (#CIn.CarroPareggCoda.Ax.ActualPosition + #CIn.CarroPareggTesta.Ax.ActualPosition) - #CIn.CarroPareggCoda.Sens.PosPareggLong.Value);
       END_IF;
   END_IF;
END_REGION

REGION Network 95: == Controllo della misura se è buona o da scartare ==
   RUNG wire#powerrail
      I_Contact( #Ctrl.TRK.BTrk_ToCheck.Prelievo_RecondGood )
      "BTrk_Presence"(Item := "BTrk".A0302_EXIT."B"["BTRK_A0302_RULL_PAREGGIATO"])
      Coil( #Ctrl.TRK.BTrk.Check_Tolleranza_BLen_Qlty )
   END_RUNG
   RUNG wire#powerrail
      { S7_Templates := "SrcType := Int" } GE_Contact(in1 := #BTrk_A0302_EXIT_GetData.Sts, in2 := 0)
      Move(in := #BTrk_A0302_EXIT_GetData.Item.Beams_Len_Min, out1 => #BTrk_A0302_Exit_Item.Tol_Min)
      Move(in := #BTrk_A0302_EXIT_GetData.Item.Beams_Len_Max, out1 => #BTrk_A0302_Exit_Item.Tol_Max)
   END_RUNG
   RUNG wire#powerrail
      Contact( #Ctrl.TRK.BTrk.Check_Tolleranza_BLen_Qlty )
      Contact( #CIn.CarroPareggTesta.Ax_InWPos )
      Contact( #CIn.CarroPareggCoda.Ax_InWPos )
      Contact( #CIn.CarroPareggCoda.Sens.PosPareggLong.Standstill )
      wire#w1
      { S7_Templates := "SrcType := Real" } InRange(min := #BTrk_A0302_Exit_Item.Tol_Min, in := "BTrk".A0302_EXIT."B"["BTRK_A0302_RULL_PAREGGIATO"].BLen_Meas, max := #BTrk_A0302_Exit_Item.Tol_Max)
      Coil( #BTrk_A0302_Exit_Item.Good )
   END_RUNG
   RUNG wire#w1
      I_Contact( #BTrk_A0302_Exit_Item.Good )
      Coil( #BTrk_A0302_Exit_Item.ToCheckLen )
   END_RUNG
   RUNG wire#powerrail
      Contact( #CIn.CarroPareggCoda.Sens.PosPareggLong.CheckMeasure )
      wire#w2
      Move(in := "BTrk".A0302_EXIT."B"["BTRK_A0302_RULL_PAREGGIATO"].BLen_Meas, out1 => #Sts.BTrk.Last_Misure1Paregg)
   END_RUNG
   RUNG wire#w2
      Move(in := #Sts.BTrk.BLen_Paregg, out1 => #Sts.BTrk.Last_Misure2Paregg)
   END_RUNG
   // the same network as SCL:
   "BTrk_Presence"(EN := NOT #Ctrl.TRK.BTrk_ToCheck.Prelievo_RecondGood,
                   Item := "BTrk".A0302_EXIT."B"["BTRK_A0302_RULL_PAREGGIATO"],
                   ENO => #_w1);
   #Ctrl.TRK.BTrk.Check_Tolleranza_BLen_Qlty := #_w1;
   IF #BTrk_A0302_EXIT_GetData.Sts >= 0 THEN
       #BTrk_A0302_Exit_Item.Tol_Min := #BTrk_A0302_EXIT_GetData.Item.Beams_Len_Min;
       #BTrk_A0302_Exit_Item.Tol_Max := #BTrk_A0302_EXIT_GetData.Item.Beams_Len_Max;
   END_IF;
   #_w2 := #Ctrl.TRK.BTrk.Check_Tolleranza_BLen_Qlty AND #CIn.CarroPareggTesta.Ax_InWPos AND #CIn.CarroPareggCoda.Ax_InWPos AND #CIn.CarroPareggCoda.Sens.PosPareggLong.Standstill;
   #BTrk_A0302_Exit_Item.Good := #_w2 AND (#BTrk_A0302_Exit_Item.Tol_Min <= "BTrk".A0302_EXIT."B"["BTRK_A0302_RULL_PAREGGIATO"].BLen_Meas) AND ("BTrk".A0302_EXIT."B"["BTRK_A0302_RULL_PAREGGIATO"].BLen_Meas <= #BTrk_A0302_Exit_Item.Tol_Max);
   #BTrk_A0302_Exit_Item.ToCheckLen := #_w2 AND NOT #BTrk_A0302_Exit_Item.Good;
   IF #CIn.CarroPareggCoda.Sens.PosPareggLong.CheckMeasure THEN
       #Sts.BTrk.Last_Misure1Paregg := "BTrk".A0302_EXIT."B"["BTRK_A0302_RULL_PAREGGIATO"].BLen_Meas;
       #Sts.BTrk.Last_Misure2Paregg := #Sts.BTrk.BLen_Paregg;
   END_IF;
END_REGION

REGION Network 96 (SCL): CONTROLLO QUALITA' - Determinazione della Qualità
   // In base alla misura del pezzo determino se il pezzo è buono o cattivo
   // 
   IF  "BTrk".A0302_EXIT.B[BTRK_A0302_RULL_PAREGGIATO].BLen_Meas > 0.0 AND "BTrk".A0302_EXIT.B[BTRK_A0302_RULL_PAREGGIATO].Quality = "UNKNOW" THEN
       // Pezzo misurato buono - In tolleranza
       IF #BTrk_A0302_Exit_Item.Good AND NOT #BTrk_A0302_Exit_Item.ToCheckLen THEN
           "BTrk".A0302_EXIT.B[BTRK_A0302_RULL_PAREGGIATO].Quality := "BEAM_GOOD_N";

       // Pezzo misurato da controllare - Fuori tolleranza 
       ELSIF NOT #BTrk_A0302_Exit_Item.Good AND #BTrk_A0302_Exit_Item.ToCheckLen THEN
           "BTrk".A0302_EXIT.B[BTRK_A0302_RULL_PAREGGIATO].Quality := "BEAM_TO_CHECK_N";

       END_IF;

   END_IF;
END_REGION

REGION Network 97: **********************************************************************************
END_REGION

REGION Network 98: <<<< MANIPOLATORI >>>>
END_REGION

REGION Network 99: <+>
END_REGION

REGION Network 100: Manipolatori - Movimento BTrk da Pareggiato ==a==> Presa in Basso
   // Pezzo su magneti del manipolatore basso in posizione di presa.
   // Quando faccio la presa
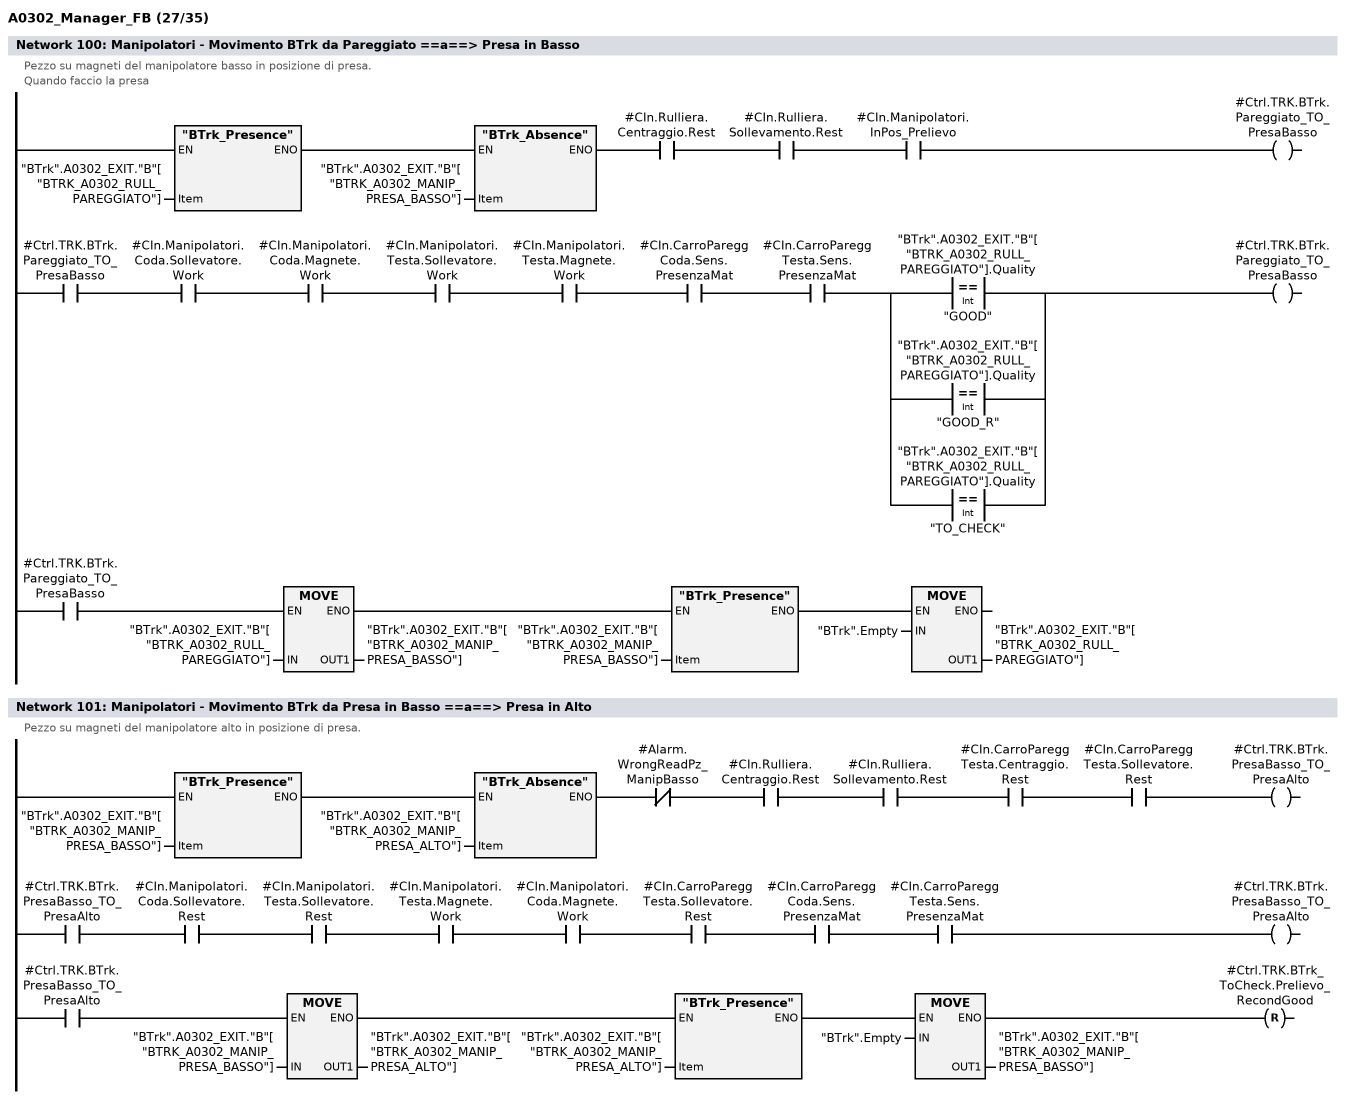
   RUNG wire#powerrail
      "BTrk_Presence"(Item := "BTrk".A0302_EXIT."B"["BTRK_A0302_RULL_PAREGGIATO"])
      "BTrk_Absence"(Item := "BTrk".A0302_EXIT."B"["BTRK_A0302_MANIP_PRESA_BASSO"])
      Contact( #CIn.Rulliera.Centraggio.Rest )
      Contact( #CIn.Rulliera.Sollevamento.Rest )
      Contact( #CIn.Manipolatori.InPos_Prelievo )
      Coil( #Ctrl.TRK.BTrk.Pareggiato_TO_PresaBasso )
   END_RUNG
   RUNG wire#powerrail
      Contact( #Ctrl.TRK.BTrk.Pareggiato_TO_PresaBasso )
      Contact( #CIn.Manipolatori.Coda.Sollevatore.Work )
      Contact( #CIn.Manipolatori.Coda.Magnete.Work )
      Contact( #CIn.Manipolatori.Testa.Sollevatore.Work )
      Contact( #CIn.Manipolatori.Testa.Magnete.Work )
      Contact( #CIn.CarroPareggCoda.Sens.PresenzaMat )
      Contact( #CIn.CarroPareggTesta.Sens.PresenzaMat )
      wire#w1
      { S7_Templates := "SrcType := Int" } EQ_Contact(in1 := "BTrk".A0302_EXIT."B"["BTRK_A0302_RULL_PAREGGIATO"].Quality, in2 := "GOOD")
      wire#w2
      Coil( #Ctrl.TRK.BTrk.Pareggiato_TO_PresaBasso )
   END_RUNG
   RUNG wire#w1
      { S7_Templates := "SrcType := Int" } EQ_Contact(in1 := "BTrk".A0302_EXIT."B"["BTRK_A0302_RULL_PAREGGIATO"].Quality, in2 := "GOOD_R")
   END_RUNG wire#w2
   RUNG wire#w1
      { S7_Templates := "SrcType := Int" } EQ_Contact(in1 := "BTrk".A0302_EXIT."B"["BTRK_A0302_RULL_PAREGGIATO"].Quality, in2 := "TO_CHECK")
   END_RUNG wire#w2
   RUNG wire#powerrail
      Contact( #Ctrl.TRK.BTrk.Pareggiato_TO_PresaBasso )
      Move(in := "BTrk".A0302_EXIT."B"["BTRK_A0302_RULL_PAREGGIATO"], out1 => "BTrk".A0302_EXIT."B"["BTRK_A0302_MANIP_PRESA_BASSO"])
      "BTrk_Presence"(Item := "BTrk".A0302_EXIT."B"["BTRK_A0302_MANIP_PRESA_BASSO"])
      Move(in := "BTrk".Empty, out1 => "BTrk".A0302_EXIT."B"["BTRK_A0302_RULL_PAREGGIATO"])
   END_RUNG
   // the same network as SCL:
   "BTrk_Presence"(Item := "BTrk".A0302_EXIT."B"["BTRK_A0302_RULL_PAREGGIATO"], ENO => #_w1);
   "BTrk_Absence"(EN := #_w1, Item := "BTrk".A0302_EXIT."B"["BTRK_A0302_MANIP_PRESA_BASSO"], ENO => #_w2);
   #Ctrl.TRK.BTrk.Pareggiato_TO_PresaBasso := #_w2 AND #CIn.Rulliera.Centraggio.Rest AND #CIn.Rulliera.Sollevamento.Rest AND #CIn.Manipolatori.InPos_Prelievo;
   #Ctrl.TRK.BTrk.Pareggiato_TO_PresaBasso := #Ctrl.TRK.BTrk.Pareggiato_TO_PresaBasso AND #CIn.Manipolatori.Coda.Sollevatore.Work AND #CIn.Manipolatori.Coda.Magnete.Work AND #CIn.Manipolatori.Testa.Sollevatore.Work AND #CIn.Manipolatori.Testa.Magnete.Work AND #CIn.CarroPareggCoda.Sens.PresenzaMat AND #CIn.CarroPareggTesta.Sens.PresenzaMat AND (("BTrk".A0302_EXIT."B"["BTRK_A0302_RULL_PAREGGIATO"].Quality = "GOOD") OR ("BTrk".A0302_EXIT."B"["BTRK_A0302_RULL_PAREGGIATO"].Quality = "GOOD_R") OR ("BTrk".A0302_EXIT."B"["BTRK_A0302_RULL_PAREGGIATO"].Quality = "TO_CHECK"));
   IF #Ctrl.TRK.BTrk.Pareggiato_TO_PresaBasso THEN
       "BTrk".A0302_EXIT."B"["BTRK_A0302_MANIP_PRESA_BASSO"] := "BTrk".A0302_EXIT."B"["BTRK_A0302_RULL_PAREGGIATO"];
   END_IF;
   "BTrk_Presence"(EN := #Ctrl.TRK.BTrk.Pareggiato_TO_PresaBasso,
                   Item := "BTrk".A0302_EXIT."B"["BTRK_A0302_MANIP_PRESA_BASSO"],
                   ENO => #_w3);
   IF #_w3 THEN "BTrk".A0302_EXIT."B"["BTRK_A0302_RULL_PAREGGIATO"] := "BTrk".Empty; END_IF;
END_REGION

REGION Network 101: Manipolatori - Movimento BTrk da Presa in Basso ==a==> Presa in Alto
   // Pezzo su magneti del manipolatore alto in posizione di presa.
   RUNG wire#powerrail
      "BTrk_Presence"(Item := "BTrk".A0302_EXIT."B"["BTRK_A0302_MANIP_PRESA_BASSO"])
      "BTrk_Absence"(Item := "BTrk".A0302_EXIT."B"["BTRK_A0302_MANIP_PRESA_ALTO"])
      I_Contact( #Alarm.WrongReadPz_ManipBasso )
      Contact( #CIn.Rulliera.Centraggio.Rest )
      Contact( #CIn.Rulliera.Sollevamento.Rest )
      Contact( #CIn.CarroPareggTesta.Centraggio.Rest )
      Contact( #CIn.CarroPareggTesta.Sollevatore.Rest )
      Coil( #Ctrl.TRK.BTrk.PresaBasso_TO_PresaAlto )
   END_RUNG
   RUNG wire#powerrail
      Contact( #Ctrl.TRK.BTrk.PresaBasso_TO_PresaAlto )
      Contact( #CIn.Manipolatori.Coda.Sollevatore.Rest )
      Contact( #CIn.Manipolatori.Testa.Sollevatore.Rest )
      Contact( #CIn.Manipolatori.Testa.Magnete.Work )
      Contact( #CIn.Manipolatori.Coda.Magnete.Work )
      Contact( #CIn.CarroPareggTesta.Sollevatore.Rest )
      Contact( #CIn.CarroPareggCoda.Sens.PresenzaMat )
      Contact( #CIn.CarroPareggTesta.Sens.PresenzaMat )
      Coil( #Ctrl.TRK.BTrk.PresaBasso_TO_PresaAlto )
   END_RUNG
   RUNG wire#powerrail
      Contact( #Ctrl.TRK.BTrk.PresaBasso_TO_PresaAlto )
      Move(in := "BTrk".A0302_EXIT."B"["BTRK_A0302_MANIP_PRESA_BASSO"], out1 => "BTrk".A0302_EXIT."B"["BTRK_A0302_MANIP_PRESA_ALTO"])
      "BTrk_Presence"(Item := "BTrk".A0302_EXIT."B"["BTRK_A0302_MANIP_PRESA_ALTO"])
      Move(in := "BTrk".Empty, out1 => "BTrk".A0302_EXIT."B"["BTRK_A0302_MANIP_PRESA_BASSO"])
      R_Coil( #Ctrl.TRK.BTrk_ToCheck.Prelievo_RecondGood )
   END_RUNG
   // the same network as SCL:
   "BTrk_Presence"(Item := "BTrk".A0302_EXIT."B"["BTRK_A0302_MANIP_PRESA_BASSO"], ENO => #_w1);
   "BTrk_Absence"(EN := #_w1, Item := "BTrk".A0302_EXIT."B"["BTRK_A0302_MANIP_PRESA_ALTO"], ENO => #_w2);
   #Ctrl.TRK.BTrk.PresaBasso_TO_PresaAlto := #_w2 AND NOT #Alarm.WrongReadPz_ManipBasso AND #CIn.Rulliera.Centraggio.Rest AND #CIn.Rulliera.Sollevamento.Rest AND #CIn.CarroPareggTesta.Centraggio.Rest AND #CIn.CarroPareggTesta.Sollevatore.Rest;
   #Ctrl.TRK.BTrk.PresaBasso_TO_PresaAlto := #Ctrl.TRK.BTrk.PresaBasso_TO_PresaAlto AND #CIn.Manipolatori.Coda.Sollevatore.Rest AND #CIn.Manipolatori.Testa.Sollevatore.Rest AND #CIn.Manipolatori.Testa.Magnete.Work AND #CIn.Manipolatori.Coda.Magnete.Work AND #CIn.CarroPareggTesta.Sollevatore.Rest AND #CIn.CarroPareggCoda.Sens.PresenzaMat AND #CIn.CarroPareggTesta.Sens.PresenzaMat;
   IF #Ctrl.TRK.BTrk.PresaBasso_TO_PresaAlto THEN
       "BTrk".A0302_EXIT."B"["BTRK_A0302_MANIP_PRESA_ALTO"] := "BTrk".A0302_EXIT."B"["BTRK_A0302_MANIP_PRESA_BASSO"];
   END_IF;
   "BTrk_Presence"(EN := #Ctrl.TRK.BTrk.PresaBasso_TO_PresaAlto,
                   Item := "BTrk".A0302_EXIT."B"["BTRK_A0302_MANIP_PRESA_ALTO"],
                   ENO => #_w3);
   IF #_w3 THEN
       "BTrk".A0302_EXIT."B"["BTRK_A0302_MANIP_PRESA_BASSO"] := "BTrk".Empty;
       #Ctrl.TRK.BTrk_ToCheck.Prelievo_RecondGood := FALSE;
   END_IF;
END_REGION

REGION Network 102: Manipolatori - Movimento BTrk da Presa in Alto Vs USCITA SCARTO alto
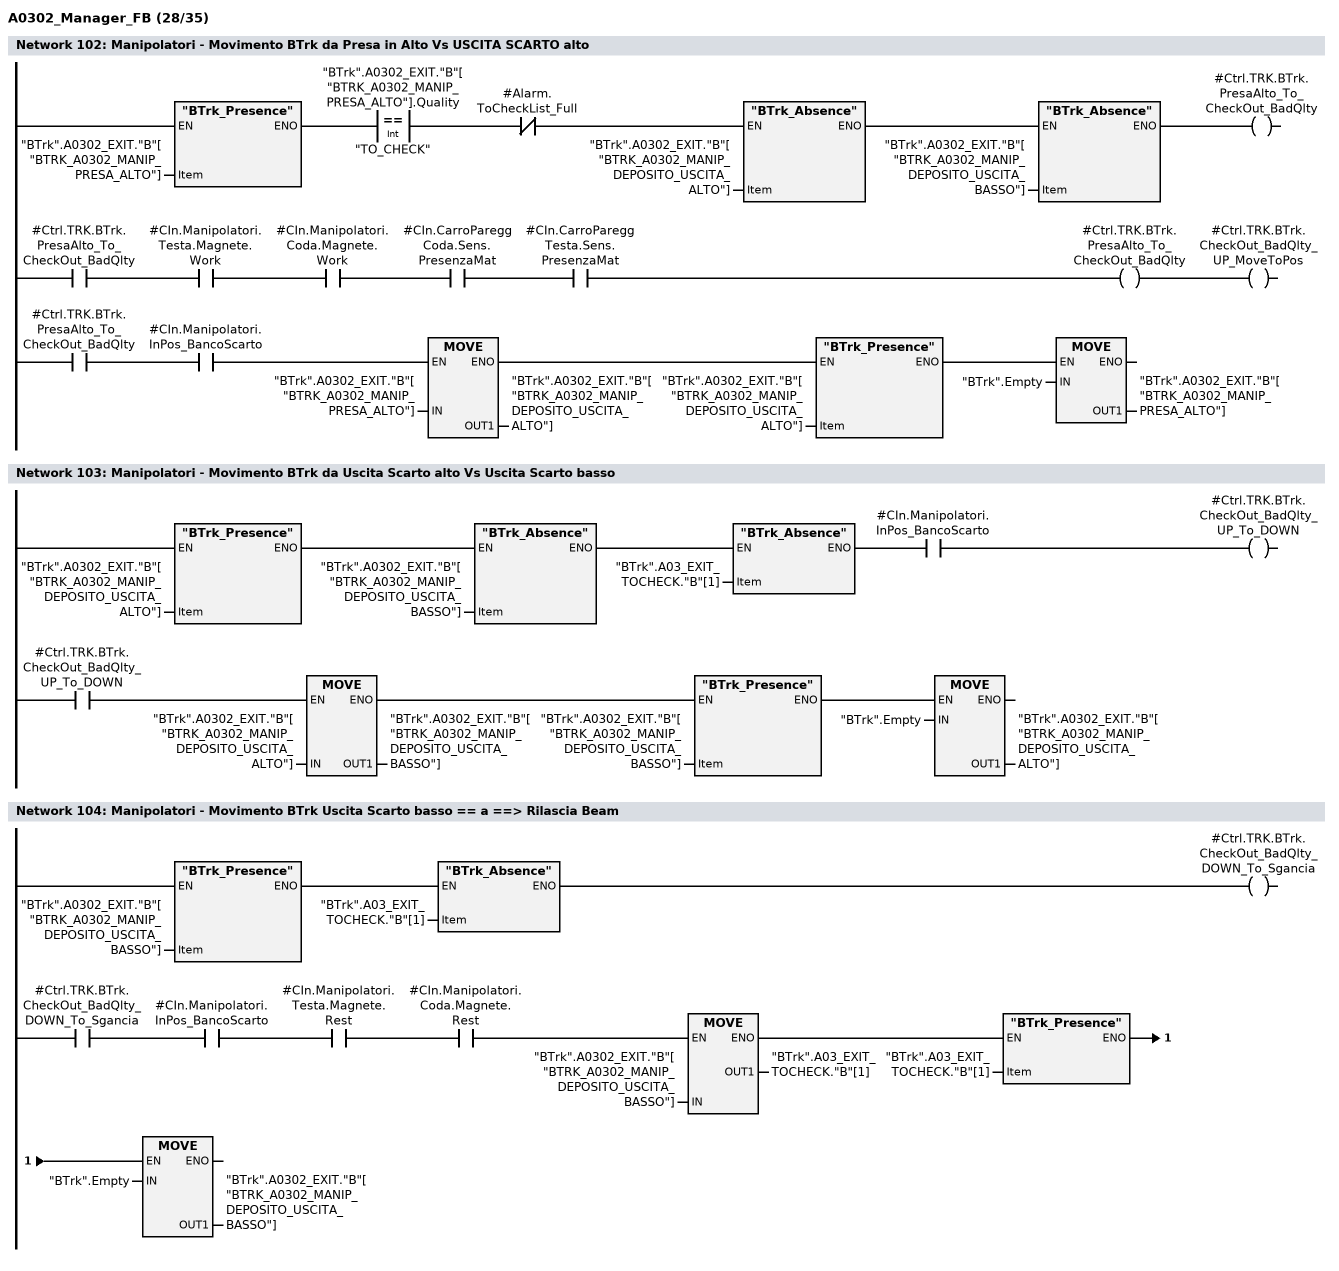
   RUNG wire#powerrail
      "BTrk_Presence"(Item := "BTrk".A0302_EXIT."B"["BTRK_A0302_MANIP_PRESA_ALTO"])
      { S7_Templates := "SrcType := Int" } EQ_Contact(in1 := "BTrk".A0302_EXIT."B"["BTRK_A0302_MANIP_PRESA_ALTO"].Quality, in2 := "TO_CHECK")
      I_Contact( #Alarm.ToCheckList_Full )
      "BTrk_Absence"(Item := "BTrk".A0302_EXIT."B"["BTRK_A0302_MANIP_DEPOSITO_USCITA_ALTO"])
      "BTrk_Absence"(Item := "BTrk".A0302_EXIT."B"["BTRK_A0302_MANIP_DEPOSITO_USCITA_BASSO"])
      Coil( #Ctrl.TRK.BTrk.PresaAlto_To_CheckOut_BadQlty )
   END_RUNG
   RUNG wire#powerrail
      Contact( #Ctrl.TRK.BTrk.PresaAlto_To_CheckOut_BadQlty )
      Contact( #CIn.Manipolatori.Testa.Magnete.Work )
      Contact( #CIn.Manipolatori.Coda.Magnete.Work )
      Contact( #CIn.CarroPareggCoda.Sens.PresenzaMat )
      Contact( #CIn.CarroPareggTesta.Sens.PresenzaMat )
      Coil( #Ctrl.TRK.BTrk.PresaAlto_To_CheckOut_BadQlty )
      Coil( #Ctrl.TRK.BTrk.CheckOut_BadQlty_UP_MoveToPos )
   END_RUNG
   RUNG wire#powerrail
      Contact( #Ctrl.TRK.BTrk.PresaAlto_To_CheckOut_BadQlty )
      Contact( #CIn.Manipolatori.InPos_BancoScarto )
      Move(in := "BTrk".A0302_EXIT."B"["BTRK_A0302_MANIP_PRESA_ALTO"], out1 => "BTrk".A0302_EXIT."B"["BTRK_A0302_MANIP_DEPOSITO_USCITA_ALTO"])
      "BTrk_Presence"(Item := "BTrk".A0302_EXIT."B"["BTRK_A0302_MANIP_DEPOSITO_USCITA_ALTO"])
      Move(in := "BTrk".Empty, out1 => "BTrk".A0302_EXIT."B"["BTRK_A0302_MANIP_PRESA_ALTO"])
   END_RUNG
   // the same network as SCL:
   "BTrk_Presence"(Item := "BTrk".A0302_EXIT."B"["BTRK_A0302_MANIP_PRESA_ALTO"], ENO => #_w1);
   "BTrk_Absence"(EN := #_w1 AND ("BTrk".A0302_EXIT."B"["BTRK_A0302_MANIP_PRESA_ALTO"].Quality = "TO_CHECK") AND NOT #Alarm.ToCheckList_Full,
                  Item := "BTrk".A0302_EXIT."B"["BTRK_A0302_MANIP_DEPOSITO_USCITA_ALTO"],
                  ENO => #_w2);
   "BTrk_Absence"(EN := #_w2,
                  Item := "BTrk".A0302_EXIT."B"["BTRK_A0302_MANIP_DEPOSITO_USCITA_BASSO"],
                  ENO => #_w3);
   #Ctrl.TRK.BTrk.PresaAlto_To_CheckOut_BadQlty := #_w3;
   #Ctrl.TRK.BTrk.PresaAlto_To_CheckOut_BadQlty := #Ctrl.TRK.BTrk.PresaAlto_To_CheckOut_BadQlty AND #CIn.Manipolatori.Testa.Magnete.Work AND #CIn.Manipolatori.Coda.Magnete.Work AND #CIn.CarroPareggCoda.Sens.PresenzaMat AND #CIn.CarroPareggTesta.Sens.PresenzaMat;
   #Ctrl.TRK.BTrk.CheckOut_BadQlty_UP_MoveToPos := #Ctrl.TRK.BTrk.PresaAlto_To_CheckOut_BadQlty;
   IF #Ctrl.TRK.BTrk.PresaAlto_To_CheckOut_BadQlty AND #CIn.Manipolatori.InPos_BancoScarto THEN
       "BTrk".A0302_EXIT."B"["BTRK_A0302_MANIP_DEPOSITO_USCITA_ALTO"] := "BTrk".A0302_EXIT."B"["BTRK_A0302_MANIP_PRESA_ALTO"];
   END_IF;
   "BTrk_Presence"(EN := #Ctrl.TRK.BTrk.PresaAlto_To_CheckOut_BadQlty AND #CIn.Manipolatori.InPos_BancoScarto,
                   Item := "BTrk".A0302_EXIT."B"["BTRK_A0302_MANIP_DEPOSITO_USCITA_ALTO"],
                   ENO => #_w4);
   IF #_w4 THEN "BTrk".A0302_EXIT."B"["BTRK_A0302_MANIP_PRESA_ALTO"] := "BTrk".Empty; END_IF;
END_REGION

REGION Network 103: Manipolatori - Movimento BTrk da Uscita Scarto alto Vs Uscita Scarto basso
   RUNG wire#powerrail
      "BTrk_Presence"(Item := "BTrk".A0302_EXIT."B"["BTRK_A0302_MANIP_DEPOSITO_USCITA_ALTO"])
      "BTrk_Absence"(Item := "BTrk".A0302_EXIT."B"["BTRK_A0302_MANIP_DEPOSITO_USCITA_BASSO"])
      "BTrk_Absence"(Item := "BTrk".A03_EXIT_TOCHECK."B"[1])
      Contact( #CIn.Manipolatori.InPos_BancoScarto )
      Coil( #Ctrl.TRK.BTrk.CheckOut_BadQlty_UP_To_DOWN )
   END_RUNG
   RUNG wire#powerrail
      Contact( #Ctrl.TRK.BTrk.CheckOut_BadQlty_UP_To_DOWN )
      Move(in := "BTrk".A0302_EXIT."B"["BTRK_A0302_MANIP_DEPOSITO_USCITA_ALTO"], out1 => "BTrk".A0302_EXIT."B"["BTRK_A0302_MANIP_DEPOSITO_USCITA_BASSO"])
      "BTrk_Presence"(Item := "BTrk".A0302_EXIT."B"["BTRK_A0302_MANIP_DEPOSITO_USCITA_BASSO"])
      Move(in := "BTrk".Empty, out1 => "BTrk".A0302_EXIT."B"["BTRK_A0302_MANIP_DEPOSITO_USCITA_ALTO"])
   END_RUNG
   // the same network as SCL:
   "BTrk_Presence"(Item := "BTrk".A0302_EXIT."B"["BTRK_A0302_MANIP_DEPOSITO_USCITA_ALTO"], ENO => #_w1);
   "BTrk_Absence"(EN := #_w1,
                  Item := "BTrk".A0302_EXIT."B"["BTRK_A0302_MANIP_DEPOSITO_USCITA_BASSO"],
                  ENO => #_w2);
   "BTrk_Absence"(EN := #_w2, Item := "BTrk".A03_EXIT_TOCHECK."B"[1], ENO => #_w3);
   #Ctrl.TRK.BTrk.CheckOut_BadQlty_UP_To_DOWN := #_w3 AND #CIn.Manipolatori.InPos_BancoScarto;
   IF #Ctrl.TRK.BTrk.CheckOut_BadQlty_UP_To_DOWN THEN
       "BTrk".A0302_EXIT."B"["BTRK_A0302_MANIP_DEPOSITO_USCITA_BASSO"] := "BTrk".A0302_EXIT."B"["BTRK_A0302_MANIP_DEPOSITO_USCITA_ALTO"];
   END_IF;
   "BTrk_Presence"(EN := #Ctrl.TRK.BTrk.CheckOut_BadQlty_UP_To_DOWN,
                   Item := "BTrk".A0302_EXIT."B"["BTRK_A0302_MANIP_DEPOSITO_USCITA_BASSO"],
                   ENO => #_w4);
   IF #_w4 THEN "BTrk".A0302_EXIT."B"["BTRK_A0302_MANIP_DEPOSITO_USCITA_ALTO"] := "BTrk".Empty; END_IF;
END_REGION

REGION Network 104: Manipolatori - Movimento BTrk Uscita Scarto basso == a ==> Rilascia Beam
   RUNG wire#powerrail
      "BTrk_Presence"(Item := "BTrk".A0302_EXIT."B"["BTRK_A0302_MANIP_DEPOSITO_USCITA_BASSO"])
      "BTrk_Absence"(Item := "BTrk".A03_EXIT_TOCHECK."B"[1])
      Coil( #Ctrl.TRK.BTrk.CheckOut_BadQlty_DOWN_To_Sgancia )
   END_RUNG
   RUNG wire#powerrail
      Contact( #Ctrl.TRK.BTrk.CheckOut_BadQlty_DOWN_To_Sgancia )
      Contact( #CIn.Manipolatori.InPos_BancoScarto )
      Contact( #CIn.Manipolatori.Testa.Magnete.Rest )
      Contact( #CIn.Manipolatori.Coda.Magnete.Rest )
      Move(in := "BTrk".A0302_EXIT."B"["BTRK_A0302_MANIP_DEPOSITO_USCITA_BASSO"], out1 => "BTrk".A03_EXIT_TOCHECK."B"[1])
      "BTrk_Presence"(Item := "BTrk".A03_EXIT_TOCHECK."B"[1])
      Move(in := "BTrk".Empty, out1 => "BTrk".A0302_EXIT."B"["BTRK_A0302_MANIP_DEPOSITO_USCITA_BASSO"])
   END_RUNG
   // the same network as SCL:
   "BTrk_Presence"(Item := "BTrk".A0302_EXIT."B"["BTRK_A0302_MANIP_DEPOSITO_USCITA_BASSO"], ENO => #_w1);
   "BTrk_Absence"(EN := #_w1, Item := "BTrk".A03_EXIT_TOCHECK."B"[1], ENO => #_w2);
   #Ctrl.TRK.BTrk.CheckOut_BadQlty_DOWN_To_Sgancia := #_w2;
   IF #Ctrl.TRK.BTrk.CheckOut_BadQlty_DOWN_To_Sgancia AND #CIn.Manipolatori.InPos_BancoScarto AND #CIn.Manipolatori.Testa.Magnete.Rest AND #CIn.Manipolatori.Coda.Magnete.Rest THEN
       "BTrk".A03_EXIT_TOCHECK."B"[1] := "BTrk".A0302_EXIT."B"["BTRK_A0302_MANIP_DEPOSITO_USCITA_BASSO"];
   END_IF;
   "BTrk_Presence"(EN := #Ctrl.TRK.BTrk.CheckOut_BadQlty_DOWN_To_Sgancia AND #CIn.Manipolatori.InPos_BancoScarto AND #CIn.Manipolatori.Testa.Magnete.Rest AND #CIn.Manipolatori.Coda.Magnete.Rest,
                   Item := "BTrk".A03_EXIT_TOCHECK."B"[1],
                   ENO => #_w3);
   IF #_w3 THEN "BTrk".A0302_EXIT."B"["BTRK_A0302_MANIP_DEPOSITO_USCITA_BASSO"] := "BTrk".Empty; END_IF;
END_REGION

REGION Network 105: ***********************************************************************************
END_REGION

REGION Network 106: == TRASFERISCI BTrk su elenco Tracking TO_CHECK ==
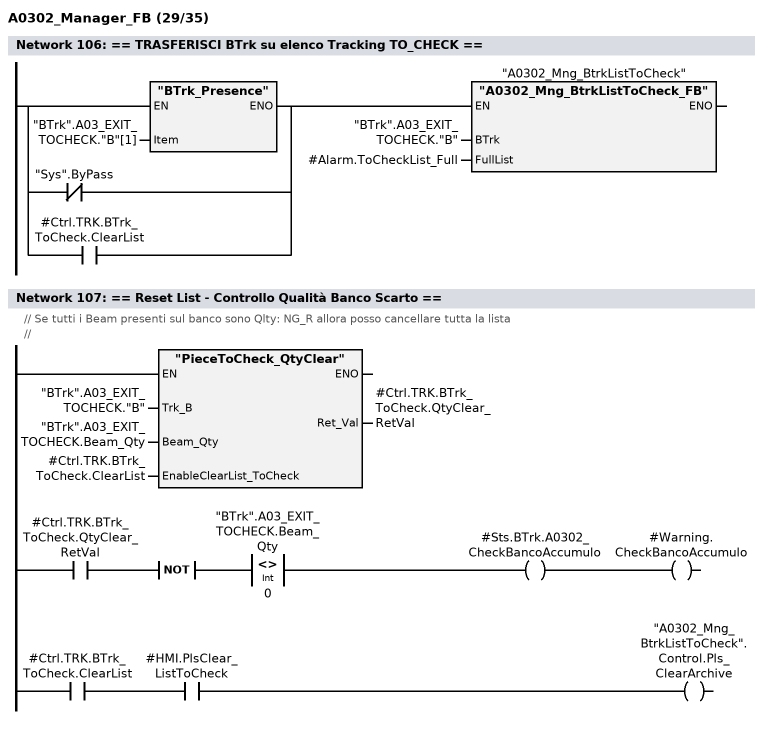
   RUNG wire#powerrail
      "BTrk_Presence"(Item := "BTrk".A03_EXIT_TOCHECK."B"[1])
      wire#w1
      "A0302_Mng_BtrkListToCheck"(BTrk := "BTrk".A03_EXIT_TOCHECK."B", FullList := #Alarm.ToCheckList_Full)
   END_RUNG
   RUNG wire#powerrail
      I_Contact( "Sys".ByPass )
   END_RUNG wire#w1
   RUNG wire#powerrail
      Contact( #Ctrl.TRK.BTrk_ToCheck.ClearList )
   END_RUNG wire#w1
   // the same network as SCL:
   "BTrk_Presence"(Item := "BTrk".A03_EXIT_TOCHECK."B"[1], ENO => #_w1);
   IF #_w1 OR NOT "Sys".ByPass OR #Ctrl.TRK.BTrk_ToCheck.ClearList THEN
       "A0302_Mng_BtrkListToCheck"(BTrk := "BTrk".A03_EXIT_TOCHECK."B", FullList := #Alarm.ToCheckList_Full);   // "A0302_Mng_BtrkListToCheck_FB"
   END_IF;
END_REGION

REGION Network 107: == Reset List - Controllo Qualità Banco Scarto ==
   // // Se tutti i Beam presenti sul banco sono Qlty: NG_R allora posso cancellare tutta la lista
   // //
   RUNG wire#powerrail
      "PieceToCheck_QtyClear"(Trk_B := "BTrk".A03_EXIT_TOCHECK."B", Beam_Qty := "BTrk".A03_EXIT_TOCHECK.Beam_Qty, EnableClearList_ToCheck := #Ctrl.TRK.BTrk_ToCheck.ClearList, Ret_Val => #Ctrl.TRK.BTrk_ToCheck.QtyClear_RetVal)
   END_RUNG
   RUNG wire#powerrail
      Contact( #Ctrl.TRK.BTrk_ToCheck.QtyClear_RetVal )
      Not()
      { S7_Templates := "SrcType := Int" } NE_Contact(in1 := "BTrk".A03_EXIT_TOCHECK.Beam_Qty, in2 := 0)
      Coil( #Sts.BTrk.A0302_CheckBancoAccumulo )
      Coil( #Warning.CheckBancoAccumulo )
   END_RUNG
   RUNG wire#powerrail
      Contact( #Ctrl.TRK.BTrk_ToCheck.ClearList )
      Contact( #HMI.PlsClear_ListToCheck )
      Coil( "A0302_Mng_BtrkListToCheck".Control.Pls_ClearArchive )
   END_RUNG
   // the same network as SCL:
   #Ctrl.TRK.BTrk_ToCheck.QtyClear_RetVal := "PieceToCheck_QtyClear"(Trk_B := "BTrk".A03_EXIT_TOCHECK."B",
                           Beam_Qty := "BTrk".A03_EXIT_TOCHECK.Beam_Qty,
                           EnableClearList_ToCheck := #Ctrl.TRK.BTrk_ToCheck.ClearList);
   #Sts.BTrk.A0302_CheckBancoAccumulo := NOT #Ctrl.TRK.BTrk_ToCheck.QtyClear_RetVal AND ("BTrk".A03_EXIT_TOCHECK.Beam_Qty <> 0);
   #Warning.CheckBancoAccumulo := #Sts.BTrk.A0302_CheckBancoAccumulo;
   "A0302_Mng_BtrkListToCheck".Control.Pls_ClearArchive := #Ctrl.TRK.BTrk_ToCheck.ClearList AND #HMI.PlsClear_ListToCheck;
END_REGION

REGION Network 108: = Movimento BTrk (RECOND_GOOD) Da banco accumulo ToChech == a ==> Centrori & Pareggiatori =
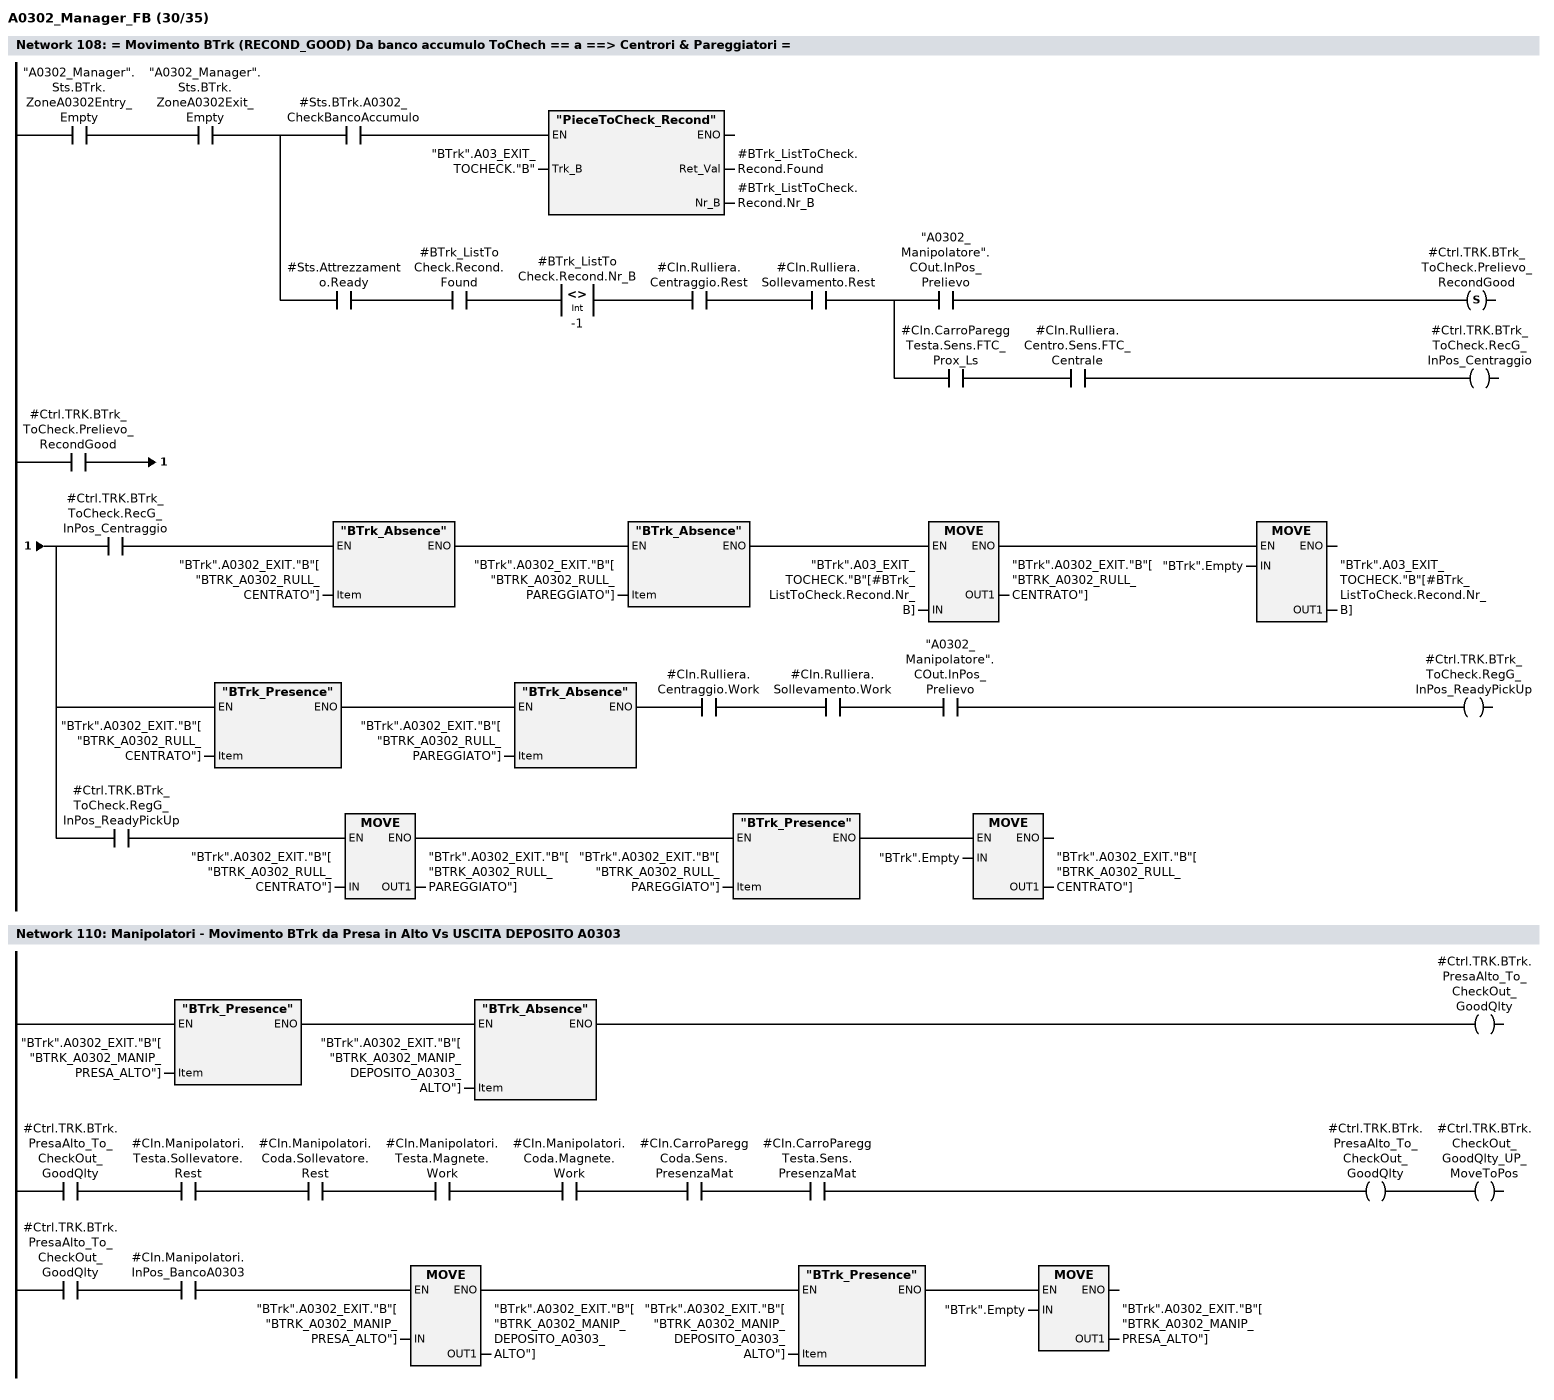
   RUNG wire#powerrail
      Contact( "A0302_Manager".Sts.BTrk.ZoneA0302Entry_Empty )
      Contact( "A0302_Manager".Sts.BTrk.ZoneA0302Exit_Empty )
      wire#w1
      Contact( #Sts.BTrk.A0302_CheckBancoAccumulo )
      "PieceToCheck_Recond"(Trk_B := "BTrk".A03_EXIT_TOCHECK."B", Ret_Val => #BTrk_ListToCheck.Recond.Found, Nr_B => #BTrk_ListToCheck.Recond.Nr_B)
   END_RUNG
   RUNG wire#w1
      Contact( #Sts.Attrezzamento.Ready )
      Contact( #BTrk_ListToCheck.Recond.Found )
      { S7_Templates := "SrcType := Int" } NE_Contact(in1 := #BTrk_ListToCheck.Recond.Nr_B, in2 := -1)
      Contact( #CIn.Rulliera.Centraggio.Rest )
      Contact( #CIn.Rulliera.Sollevamento.Rest )
      wire#w2
      Contact( "A0302_Manipolatore".COut.InPos_Prelievo )
      S_Coil( #Ctrl.TRK.BTrk_ToCheck.Prelievo_RecondGood )
   END_RUNG
   RUNG wire#w2
      Contact( #CIn.CarroPareggTesta.Sens.FTC_Prox_Ls )
      Contact( #CIn.Rulliera.Centro.Sens.FTC_Centrale )
      Coil( #Ctrl.TRK.BTrk_ToCheck.RecG_InPos_Centraggio )
   END_RUNG
   RUNG wire#powerrail
      Contact( #Ctrl.TRK.BTrk_ToCheck.Prelievo_RecondGood )
      wire#w3
      Contact( #Ctrl.TRK.BTrk_ToCheck.RecG_InPos_Centraggio )
      "BTrk_Absence"(Item := "BTrk".A0302_EXIT."B"["BTRK_A0302_RULL_CENTRATO"])
      "BTrk_Absence"(Item := "BTrk".A0302_EXIT."B"["BTRK_A0302_RULL_PAREGGIATO"])
      Move(in := "BTrk".A03_EXIT_TOCHECK."B"[#BTrk_ListToCheck.Recond.Nr_B], out1 => "BTrk".A0302_EXIT."B"["BTRK_A0302_RULL_CENTRATO"])
      Move(in := "BTrk".Empty, out1 => "BTrk".A03_EXIT_TOCHECK."B"[#BTrk_ListToCheck.Recond.Nr_B])
   END_RUNG
   RUNG wire#w3
      "BTrk_Presence"(Item := "BTrk".A0302_EXIT."B"["BTRK_A0302_RULL_CENTRATO"])
      "BTrk_Absence"(Item := "BTrk".A0302_EXIT."B"["BTRK_A0302_RULL_PAREGGIATO"])
      Contact( #CIn.Rulliera.Centraggio.Work )
      Contact( #CIn.Rulliera.Sollevamento.Work )
      Contact( "A0302_Manipolatore".COut.InPos_Prelievo )
      Coil( #Ctrl.TRK.BTrk_ToCheck.RegG_InPos_ReadyPickUp )
   END_RUNG
   RUNG wire#w3
      Contact( #Ctrl.TRK.BTrk_ToCheck.RegG_InPos_ReadyPickUp )
      Move(in := "BTrk".A0302_EXIT."B"["BTRK_A0302_RULL_CENTRATO"], out1 => "BTrk".A0302_EXIT."B"["BTRK_A0302_RULL_PAREGGIATO"])
      "BTrk_Presence"(Item := "BTrk".A0302_EXIT."B"["BTRK_A0302_RULL_PAREGGIATO"])
      Move(in := "BTrk".Empty, out1 => "BTrk".A0302_EXIT."B"["BTRK_A0302_RULL_CENTRATO"])
   END_RUNG
   // the same network as SCL:
   #_w1 := "A0302_Manager".Sts.BTrk.ZoneA0302Entry_Empty AND "A0302_Manager".Sts.BTrk.ZoneA0302Exit_Empty;
   IF #_w1 AND #Sts.BTrk.A0302_CheckBancoAccumulo THEN
       #BTrk_ListToCheck.Recond.Found := "PieceToCheck_Recond"(Trk_B := "BTrk".A03_EXIT_TOCHECK."B",
                               Nr_B => #BTrk_ListToCheck.Recond.Nr_B);
   END_IF;
   #_w2 := #_w1 AND #Sts.Attrezzamento.Ready AND #BTrk_ListToCheck.Recond.Found AND (#BTrk_ListToCheck.Recond.Nr_B <> (-1)) AND #CIn.Rulliera.Centraggio.Rest AND #CIn.Rulliera.Sollevamento.Rest;
   IF #_w2 AND "A0302_Manipolatore".COut.InPos_Prelievo THEN
       #Ctrl.TRK.BTrk_ToCheck.Prelievo_RecondGood := TRUE;
   END_IF;
   #Ctrl.TRK.BTrk_ToCheck.RecG_InPos_Centraggio := #_w2 AND #CIn.CarroPareggTesta.Sens.FTC_Prox_Ls AND #CIn.Rulliera.Centro.Sens.FTC_Centrale;
   "BTrk_Absence"(EN := #Ctrl.TRK.BTrk_ToCheck.Prelievo_RecondGood AND #Ctrl.TRK.BTrk_ToCheck.RecG_InPos_Centraggio,
                  Item := "BTrk".A0302_EXIT."B"["BTRK_A0302_RULL_CENTRATO"],
                  ENO => #_w3);
   "BTrk_Absence"(EN := #_w3, Item := "BTrk".A0302_EXIT."B"["BTRK_A0302_RULL_PAREGGIATO"], ENO => #_w4);
   IF #_w4 THEN
       "BTrk".A0302_EXIT."B"["BTRK_A0302_RULL_CENTRATO"] := "BTrk".A03_EXIT_TOCHECK."B"[#BTrk_ListToCheck.Recond.Nr_B];
       "BTrk".A03_EXIT_TOCHECK."B"[#BTrk_ListToCheck.Recond.Nr_B] := "BTrk".Empty;
   END_IF;
   "BTrk_Presence"(EN := #Ctrl.TRK.BTrk_ToCheck.Prelievo_RecondGood,
                   Item := "BTrk".A0302_EXIT."B"["BTRK_A0302_RULL_CENTRATO"],
                   ENO => #_w5);
   "BTrk_Absence"(EN := #_w5, Item := "BTrk".A0302_EXIT."B"["BTRK_A0302_RULL_PAREGGIATO"], ENO => #_w6);
   #Ctrl.TRK.BTrk_ToCheck.RegG_InPos_ReadyPickUp := #_w6 AND #CIn.Rulliera.Centraggio.Work AND #CIn.Rulliera.Sollevamento.Work AND "A0302_Manipolatore".COut.InPos_Prelievo;
   IF #Ctrl.TRK.BTrk_ToCheck.Prelievo_RecondGood AND #Ctrl.TRK.BTrk_ToCheck.RegG_InPos_ReadyPickUp THEN
       "BTrk".A0302_EXIT."B"["BTRK_A0302_RULL_PAREGGIATO"] := "BTrk".A0302_EXIT."B"["BTRK_A0302_RULL_CENTRATO"];
   END_IF;
   "BTrk_Presence"(EN := #Ctrl.TRK.BTrk_ToCheck.Prelievo_RecondGood AND #Ctrl.TRK.BTrk_ToCheck.RegG_InPos_ReadyPickUp,
                   Item := "BTrk".A0302_EXIT."B"["BTRK_A0302_RULL_PAREGGIATO"],
                   ENO => #_w7);
   IF #_w7 THEN "BTrk".A0302_EXIT."B"["BTRK_A0302_RULL_CENTRATO"] := "BTrk".Empty; END_IF;
END_REGION

REGION Network 109: ***********************************************************************************
END_REGION

REGION Network 110: Manipolatori - Movimento BTrk da Presa in Alto Vs USCITA DEPOSITO A0303
   RUNG wire#powerrail
      "BTrk_Presence"(Item := "BTrk".A0302_EXIT."B"["BTRK_A0302_MANIP_PRESA_ALTO"])
      "BTrk_Absence"(Item := "BTrk".A0302_EXIT."B"["BTRK_A0302_MANIP_DEPOSITO_A0303_ALTO"])
      Coil( #Ctrl.TRK.BTrk.PresaAlto_To_CheckOut_GoodQlty )
   END_RUNG
   RUNG wire#powerrail
      Contact( #Ctrl.TRK.BTrk.PresaAlto_To_CheckOut_GoodQlty )
      Contact( #CIn.Manipolatori.Testa.Sollevatore.Rest )
      Contact( #CIn.Manipolatori.Coda.Sollevatore.Rest )
      Contact( #CIn.Manipolatori.Testa.Magnete.Work )
      Contact( #CIn.Manipolatori.Coda.Magnete.Work )
      Contact( #CIn.CarroPareggCoda.Sens.PresenzaMat )
      Contact( #CIn.CarroPareggTesta.Sens.PresenzaMat )
      Coil( #Ctrl.TRK.BTrk.PresaAlto_To_CheckOut_GoodQlty )
      Coil( #Ctrl.TRK.BTrk.CheckOut_GoodQlty_UP_MoveToPos )
   END_RUNG
   RUNG wire#powerrail
      Contact( #Ctrl.TRK.BTrk.PresaAlto_To_CheckOut_GoodQlty )
      Contact( #CIn.Manipolatori.InPos_BancoA0303 )
      Move(in := "BTrk".A0302_EXIT."B"["BTRK_A0302_MANIP_PRESA_ALTO"], out1 => "BTrk".A0302_EXIT."B"["BTRK_A0302_MANIP_DEPOSITO_A0303_ALTO"])
      "BTrk_Presence"(Item := "BTrk".A0302_EXIT."B"["BTRK_A0302_MANIP_DEPOSITO_A0303_ALTO"])
      Move(in := "BTrk".Empty, out1 => "BTrk".A0302_EXIT."B"["BTRK_A0302_MANIP_PRESA_ALTO"])
   END_RUNG
   // the same network as SCL:
   "BTrk_Presence"(Item := "BTrk".A0302_EXIT."B"["BTRK_A0302_MANIP_PRESA_ALTO"], ENO => #_w1);
   "BTrk_Absence"(EN := #_w1,
                  Item := "BTrk".A0302_EXIT."B"["BTRK_A0302_MANIP_DEPOSITO_A0303_ALTO"],
                  ENO => #_w2);
   #Ctrl.TRK.BTrk.PresaAlto_To_CheckOut_GoodQlty := #_w2;
   #Ctrl.TRK.BTrk.PresaAlto_To_CheckOut_GoodQlty := #Ctrl.TRK.BTrk.PresaAlto_To_CheckOut_GoodQlty AND #CIn.Manipolatori.Testa.Sollevatore.Rest AND #CIn.Manipolatori.Coda.Sollevatore.Rest AND #CIn.Manipolatori.Testa.Magnete.Work AND #CIn.Manipolatori.Coda.Magnete.Work AND #CIn.CarroPareggCoda.Sens.PresenzaMat AND #CIn.CarroPareggTesta.Sens.PresenzaMat;
   #Ctrl.TRK.BTrk.CheckOut_GoodQlty_UP_MoveToPos := #Ctrl.TRK.BTrk.PresaAlto_To_CheckOut_GoodQlty;
   IF #Ctrl.TRK.BTrk.PresaAlto_To_CheckOut_GoodQlty AND #CIn.Manipolatori.InPos_BancoA0303 THEN
       "BTrk".A0302_EXIT."B"["BTRK_A0302_MANIP_DEPOSITO_A0303_ALTO"] := "BTrk".A0302_EXIT."B"["BTRK_A0302_MANIP_PRESA_ALTO"];
   END_IF;
   "BTrk_Presence"(EN := #Ctrl.TRK.BTrk.PresaAlto_To_CheckOut_GoodQlty AND #CIn.Manipolatori.InPos_BancoA0303,
                   Item := "BTrk".A0302_EXIT."B"["BTRK_A0302_MANIP_DEPOSITO_A0303_ALTO"],
                   ENO => #_w3);
   IF #_w3 THEN "BTrk".A0302_EXIT."B"["BTRK_A0302_MANIP_PRESA_ALTO"] := "BTrk".Empty; END_IF;
END_REGION

REGION Network 111: Manipolatori - Movimento BTrk da Uscita Deposito A0303 alto Vs Uscita deposito A0303 basso
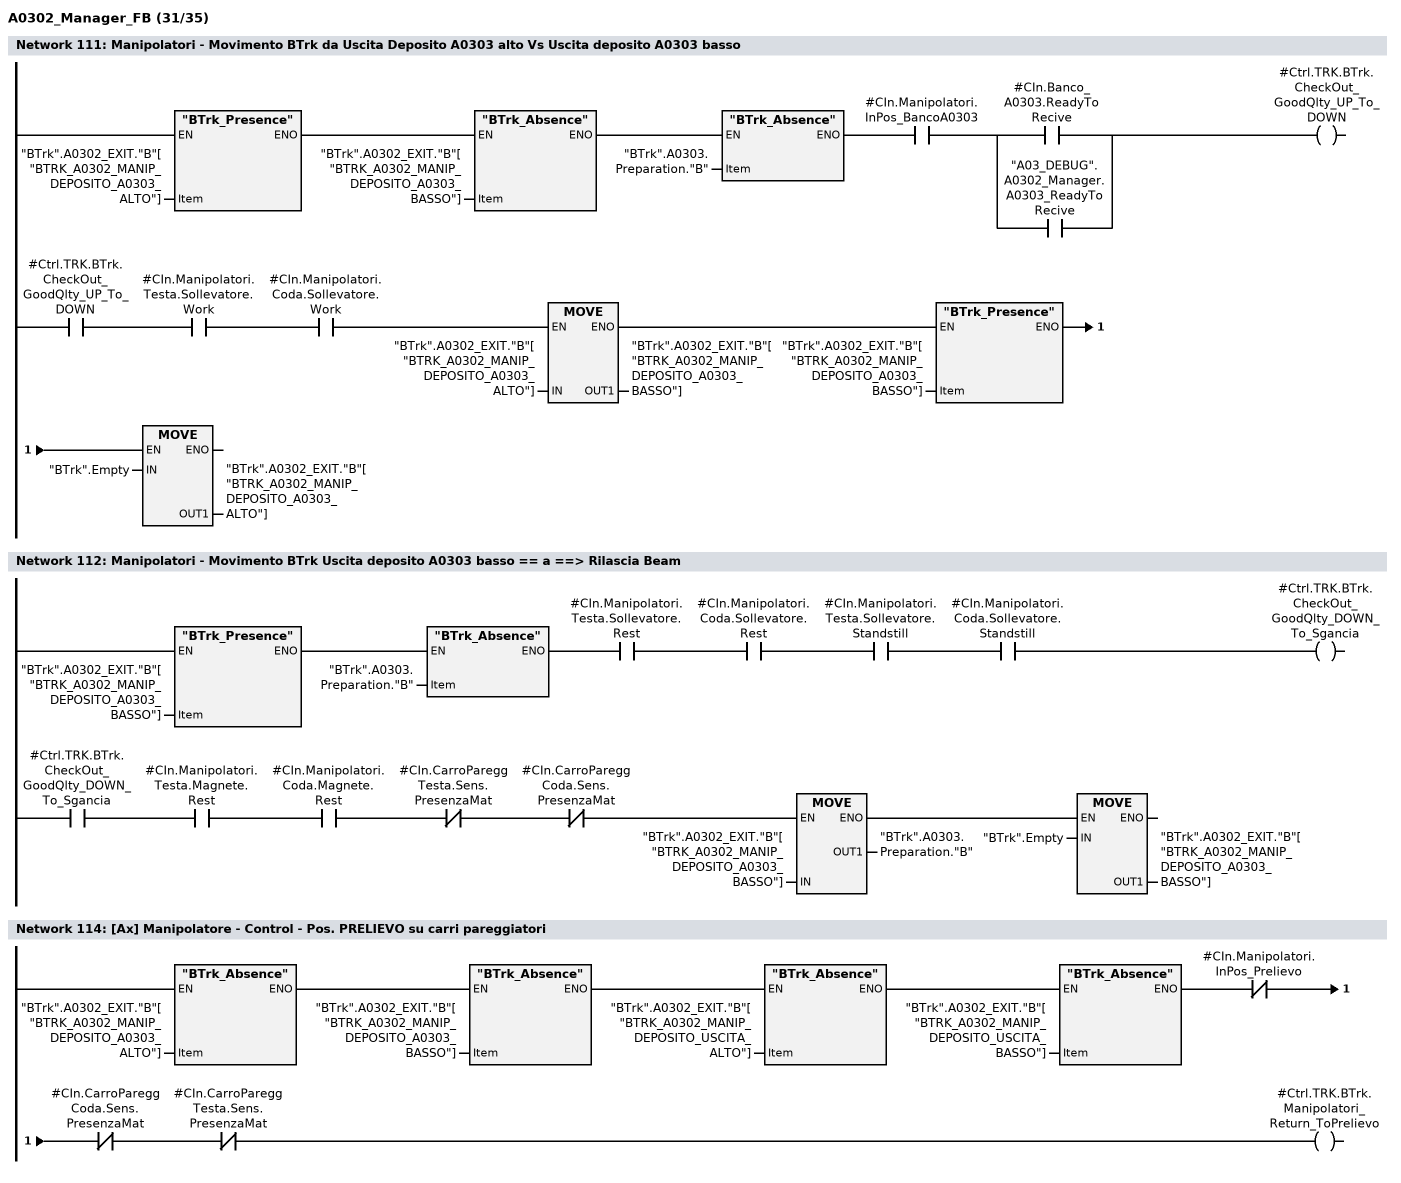
   RUNG wire#powerrail
      "BTrk_Presence"(Item := "BTrk".A0302_EXIT."B"["BTRK_A0302_MANIP_DEPOSITO_A0303_ALTO"])
      "BTrk_Absence"(Item := "BTrk".A0302_EXIT."B"["BTRK_A0302_MANIP_DEPOSITO_A0303_BASSO"])
      "BTrk_Absence"(Item := "BTrk".A0303.Preparation."B")
      Contact( #CIn.Manipolatori.InPos_BancoA0303 )
      wire#w1
      Contact( #CIn.Banco_A0303.ReadyToRecive )
      wire#w2
      Coil( #Ctrl.TRK.BTrk.CheckOut_GoodQlty_UP_To_DOWN )
   END_RUNG
   RUNG wire#w1
      Contact( "A03_DEBUG".A0302_Manager.A0303_ReadyToRecive )
   END_RUNG wire#w2
   RUNG wire#powerrail
      Contact( #Ctrl.TRK.BTrk.CheckOut_GoodQlty_UP_To_DOWN )
      Contact( #CIn.Manipolatori.Testa.Sollevatore.Work )
      Contact( #CIn.Manipolatori.Coda.Sollevatore.Work )
      Move(in := "BTrk".A0302_EXIT."B"["BTRK_A0302_MANIP_DEPOSITO_A0303_ALTO"], out1 => "BTrk".A0302_EXIT."B"["BTRK_A0302_MANIP_DEPOSITO_A0303_BASSO"])
      "BTrk_Presence"(Item := "BTrk".A0302_EXIT."B"["BTRK_A0302_MANIP_DEPOSITO_A0303_BASSO"])
      Move(in := "BTrk".Empty, out1 => "BTrk".A0302_EXIT."B"["BTRK_A0302_MANIP_DEPOSITO_A0303_ALTO"])
   END_RUNG
   // the same network as SCL:
   "BTrk_Presence"(Item := "BTrk".A0302_EXIT."B"["BTRK_A0302_MANIP_DEPOSITO_A0303_ALTO"], ENO => #_w1);
   "BTrk_Absence"(EN := #_w1,
                  Item := "BTrk".A0302_EXIT."B"["BTRK_A0302_MANIP_DEPOSITO_A0303_BASSO"],
                  ENO => #_w2);
   "BTrk_Absence"(EN := #_w2, Item := "BTrk".A0303.Preparation."B", ENO => #_w3);
   #Ctrl.TRK.BTrk.CheckOut_GoodQlty_UP_To_DOWN := #_w3 AND #CIn.Manipolatori.InPos_BancoA0303 AND (#CIn.Banco_A0303.ReadyToRecive OR "A03_DEBUG".A0302_Manager.A0303_ReadyToRecive);
   IF #Ctrl.TRK.BTrk.CheckOut_GoodQlty_UP_To_DOWN AND #CIn.Manipolatori.Testa.Sollevatore.Work AND #CIn.Manipolatori.Coda.Sollevatore.Work THEN
       "BTrk".A0302_EXIT."B"["BTRK_A0302_MANIP_DEPOSITO_A0303_BASSO"] := "BTrk".A0302_EXIT."B"["BTRK_A0302_MANIP_DEPOSITO_A0303_ALTO"];
   END_IF;
   "BTrk_Presence"(EN := #Ctrl.TRK.BTrk.CheckOut_GoodQlty_UP_To_DOWN AND #CIn.Manipolatori.Testa.Sollevatore.Work AND #CIn.Manipolatori.Coda.Sollevatore.Work,
                   Item := "BTrk".A0302_EXIT."B"["BTRK_A0302_MANIP_DEPOSITO_A0303_BASSO"],
                   ENO => #_w4);
   IF #_w4 THEN "BTrk".A0302_EXIT."B"["BTRK_A0302_MANIP_DEPOSITO_A0303_ALTO"] := "BTrk".Empty; END_IF;
END_REGION

REGION Network 112: Manipolatori - Movimento BTrk Uscita deposito A0303 basso == a ==> Rilascia Beam
   RUNG wire#powerrail
      "BTrk_Presence"(Item := "BTrk".A0302_EXIT."B"["BTRK_A0302_MANIP_DEPOSITO_A0303_BASSO"])
      "BTrk_Absence"(Item := "BTrk".A0303.Preparation."B")
      Contact( #CIn.Manipolatori.Testa.Sollevatore.Rest )
      Contact( #CIn.Manipolatori.Coda.Sollevatore.Rest )
      Contact( #CIn.Manipolatori.Testa.Sollevatore.Standstill )
      Contact( #CIn.Manipolatori.Coda.Sollevatore.Standstill )
      Coil( #Ctrl.TRK.BTrk.CheckOut_GoodQlty_DOWN_To_Sgancia )
   END_RUNG
   RUNG wire#powerrail
      Contact( #Ctrl.TRK.BTrk.CheckOut_GoodQlty_DOWN_To_Sgancia )
      Contact( #CIn.Manipolatori.Testa.Magnete.Rest )
      Contact( #CIn.Manipolatori.Coda.Magnete.Rest )
      I_Contact( #CIn.CarroPareggTesta.Sens.PresenzaMat )
      I_Contact( #CIn.CarroPareggCoda.Sens.PresenzaMat )
      Move(in := "BTrk".A0302_EXIT."B"["BTRK_A0302_MANIP_DEPOSITO_A0303_BASSO"], out1 => "BTrk".A0303.Preparation."B")
      Move(in := "BTrk".Empty, out1 => "BTrk".A0302_EXIT."B"["BTRK_A0302_MANIP_DEPOSITO_A0303_BASSO"])
   END_RUNG
   // the same network as SCL:
   "BTrk_Presence"(Item := "BTrk".A0302_EXIT."B"["BTRK_A0302_MANIP_DEPOSITO_A0303_BASSO"], ENO => #_w1);
   "BTrk_Absence"(EN := #_w1, Item := "BTrk".A0303.Preparation."B", ENO => #_w2);
   #Ctrl.TRK.BTrk.CheckOut_GoodQlty_DOWN_To_Sgancia := #_w2 AND #CIn.Manipolatori.Testa.Sollevatore.Rest AND #CIn.Manipolatori.Coda.Sollevatore.Rest AND #CIn.Manipolatori.Testa.Sollevatore.Standstill AND #CIn.Manipolatori.Coda.Sollevatore.Standstill;
   IF #Ctrl.TRK.BTrk.CheckOut_GoodQlty_DOWN_To_Sgancia AND #CIn.Manipolatori.Testa.Magnete.Rest AND #CIn.Manipolatori.Coda.Magnete.Rest AND NOT #CIn.CarroPareggTesta.Sens.PresenzaMat AND NOT #CIn.CarroPareggCoda.Sens.PresenzaMat THEN
       "BTrk".A0303.Preparation."B" := "BTrk".A0302_EXIT."B"["BTRK_A0302_MANIP_DEPOSITO_A0303_BASSO"];
       "BTrk".A0302_EXIT."B"["BTRK_A0302_MANIP_DEPOSITO_A0303_BASSO"] := "BTrk".Empty;
   END_IF;
END_REGION

REGION Network 113: <+>
END_REGION

REGION Network 114: [Ax] Manipolatore - Control - Pos. PRELIEVO su carri pareggiatori
   RUNG wire#powerrail
      "BTrk_Absence"(Item := "BTrk".A0302_EXIT."B"["BTRK_A0302_MANIP_DEPOSITO_A0303_ALTO"])
      "BTrk_Absence"(Item := "BTrk".A0302_EXIT."B"["BTRK_A0302_MANIP_DEPOSITO_A0303_BASSO"])
      "BTrk_Absence"(Item := "BTrk".A0302_EXIT."B"["BTRK_A0302_MANIP_DEPOSITO_USCITA_ALTO"])
      "BTrk_Absence"(Item := "BTrk".A0302_EXIT."B"["BTRK_A0302_MANIP_DEPOSITO_USCITA_BASSO"])
      I_Contact( #CIn.Manipolatori.InPos_Prelievo )
      I_Contact( #CIn.CarroPareggCoda.Sens.PresenzaMat )
      I_Contact( #CIn.CarroPareggTesta.Sens.PresenzaMat )
      Coil( #Ctrl.TRK.BTrk.Manipolatori_Return_ToPrelievo )
   END_RUNG
   // the same network as SCL:
   "BTrk_Absence"(Item := "BTrk".A0302_EXIT."B"["BTRK_A0302_MANIP_DEPOSITO_A0303_ALTO"], ENO => #_w1);
   "BTrk_Absence"(EN := #_w1,
                  Item := "BTrk".A0302_EXIT."B"["BTRK_A0302_MANIP_DEPOSITO_A0303_BASSO"],
                  ENO => #_w2);
   "BTrk_Absence"(EN := #_w2,
                  Item := "BTrk".A0302_EXIT."B"["BTRK_A0302_MANIP_DEPOSITO_USCITA_ALTO"],
                  ENO => #_w3);
   "BTrk_Absence"(EN := #_w3,
                  Item := "BTrk".A0302_EXIT."B"["BTRK_A0302_MANIP_DEPOSITO_USCITA_BASSO"],
                  ENO => #_w4);
   #Ctrl.TRK.BTrk.Manipolatori_Return_ToPrelievo := #_w4 AND NOT #CIn.Manipolatori.InPos_Prelievo AND NOT #CIn.CarroPareggCoda.Sens.PresenzaMat AND NOT #CIn.CarroPareggTesta.Sens.PresenzaMat;
END_REGION

REGION Network 115: <+>
END_REGION

REGION Network 116: Manipolatori - Controllo del pezzo sui Magneti - Allarme grave se perdo i sensori presenza
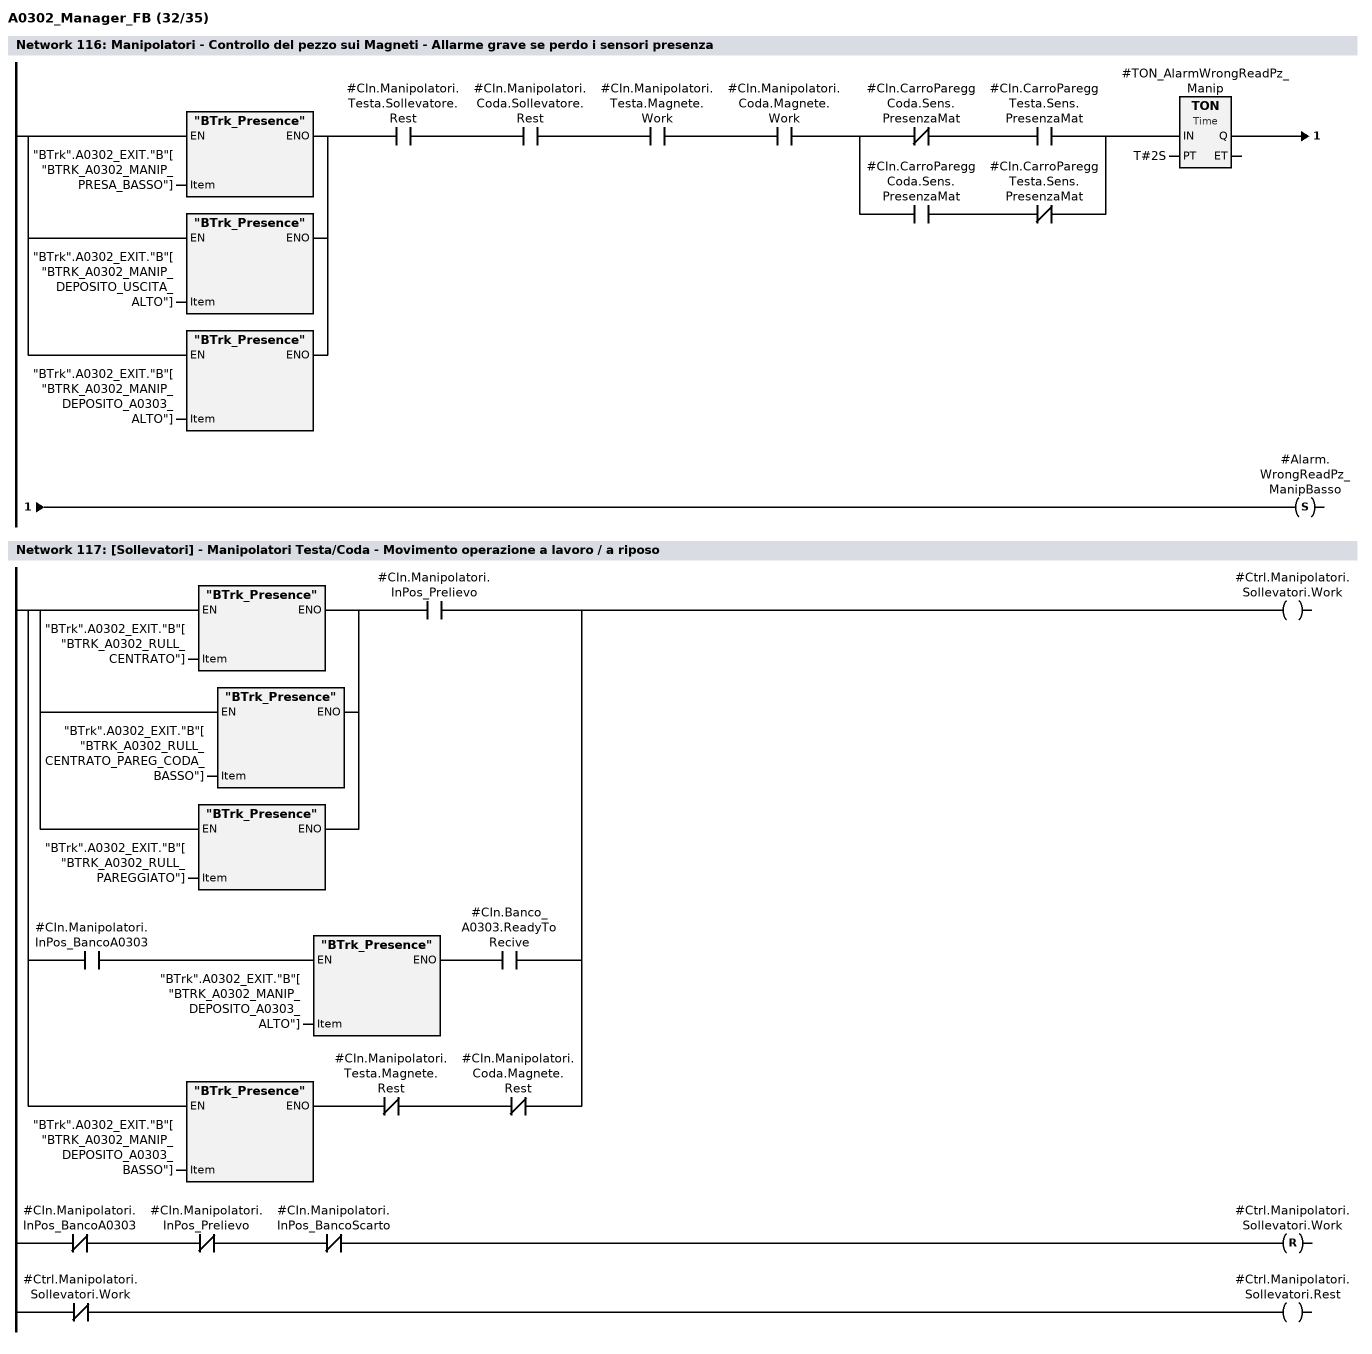
   RUNG wire#powerrail
      "BTrk_Presence"(Item := "BTrk".A0302_EXIT."B"["BTRK_A0302_MANIP_PRESA_BASSO"])
      wire#w1
      Contact( #CIn.Manipolatori.Testa.Sollevatore.Rest )
      Contact( #CIn.Manipolatori.Coda.Sollevatore.Rest )
      Contact( #CIn.Manipolatori.Testa.Magnete.Work )
      Contact( #CIn.Manipolatori.Coda.Magnete.Work )
      wire#w2
      I_Contact( #CIn.CarroPareggCoda.Sens.PresenzaMat )
      Contact( #CIn.CarroPareggTesta.Sens.PresenzaMat )
      wire#w3
      { S7_Templates := "time_type := Time" } #TON_AlarmWrongReadPz_Manip.TON(pt := T#2S, et =>)
      S_Coil( #Alarm.WrongReadPz_ManipBasso )
   END_RUNG
   RUNG wire#powerrail
      "BTrk_Presence"(Item := "BTrk".A0302_EXIT."B"["BTRK_A0302_MANIP_DEPOSITO_USCITA_ALTO"])
   END_RUNG wire#w1
   RUNG wire#powerrail
      "BTrk_Presence"(Item := "BTrk".A0302_EXIT."B"["BTRK_A0302_MANIP_DEPOSITO_A0303_ALTO"])
   END_RUNG wire#w1
   RUNG wire#w2
      Contact( #CIn.CarroPareggCoda.Sens.PresenzaMat )
      I_Contact( #CIn.CarroPareggTesta.Sens.PresenzaMat )
   END_RUNG wire#w3
   // the same network as SCL:
   "BTrk_Presence"(Item := "BTrk".A0302_EXIT."B"["BTRK_A0302_MANIP_PRESA_BASSO"], ENO => #_w1);
   "BTrk_Presence"(Item := "BTrk".A0302_EXIT."B"["BTRK_A0302_MANIP_DEPOSITO_USCITA_ALTO"], ENO => #_w2);
   "BTrk_Presence"(Item := "BTrk".A0302_EXIT."B"["BTRK_A0302_MANIP_DEPOSITO_A0303_ALTO"], ENO => #_w3);
   #TON_AlarmWrongReadPz_Manip.TON(IN := (#_w1 OR #_w2 OR #_w3) AND #CIn.Manipolatori.Testa.Sollevatore.Rest AND #CIn.Manipolatori.Coda.Sollevatore.Rest AND #CIn.Manipolatori.Testa.Magnete.Work AND #CIn.Manipolatori.Coda.Magnete.Work AND ((NOT #CIn.CarroPareggCoda.Sens.PresenzaMat AND #CIn.CarroPareggTesta.Sens.PresenzaMat) OR (#CIn.CarroPareggCoda.Sens.PresenzaMat AND NOT #CIn.CarroPareggTesta.Sens.PresenzaMat)),
                           PT := T#2S);
   IF #TON_AlarmWrongReadPz_Manip.Q THEN #Alarm.WrongReadPz_ManipBasso := TRUE; END_IF;
END_REGION

REGION Network 117: [Sollevatori] - Manipolatori Testa/Coda - Movimento operazione a lavoro / a riposo
   RUNG wire#powerrail
      "BTrk_Presence"(Item := "BTrk".A0302_EXIT."B"["BTRK_A0302_RULL_CENTRATO"])
      wire#w1
      Contact( #CIn.Manipolatori.InPos_Prelievo )
      wire#w2
      Coil( #Ctrl.Manipolatori.Sollevatori.Work )
   END_RUNG
   RUNG wire#powerrail
      "BTrk_Presence"(Item := "BTrk".A0302_EXIT."B"["BTRK_A0302_RULL_CENTRATO_PAREG_CODA_BASSO"])
   END_RUNG wire#w1
   RUNG wire#powerrail
      "BTrk_Presence"(Item := "BTrk".A0302_EXIT."B"["BTRK_A0302_RULL_PAREGGIATO"])
   END_RUNG wire#w1
   RUNG wire#powerrail
      Contact( #CIn.Manipolatori.InPos_BancoA0303 )
      "BTrk_Presence"(Item := "BTrk".A0302_EXIT."B"["BTRK_A0302_MANIP_DEPOSITO_A0303_ALTO"])
      Contact( #CIn.Banco_A0303.ReadyToRecive )
   END_RUNG wire#w2
   RUNG wire#powerrail
      "BTrk_Presence"(Item := "BTrk".A0302_EXIT."B"["BTRK_A0302_MANIP_DEPOSITO_A0303_BASSO"])
      I_Contact( #CIn.Manipolatori.Testa.Magnete.Rest )
      I_Contact( #CIn.Manipolatori.Coda.Magnete.Rest )
   END_RUNG wire#w2
   RUNG wire#powerrail
      I_Contact( #CIn.Manipolatori.InPos_BancoA0303 )
      I_Contact( #CIn.Manipolatori.InPos_Prelievo )
      I_Contact( #CIn.Manipolatori.InPos_BancoScarto )
      R_Coil( #Ctrl.Manipolatori.Sollevatori.Work )
   END_RUNG
   RUNG wire#powerrail
      I_Contact( #Ctrl.Manipolatori.Sollevatori.Work )
      Coil( #Ctrl.Manipolatori.Sollevatori.Rest )
   END_RUNG
   // the same network as SCL:
   "BTrk_Presence"(Item := "BTrk".A0302_EXIT."B"["BTRK_A0302_RULL_CENTRATO"], ENO => #_w1);
   "BTrk_Presence"(Item := "BTrk".A0302_EXIT."B"["BTRK_A0302_RULL_CENTRATO_PAREG_CODA_BASSO"], ENO => #_w2);
   "BTrk_Presence"(Item := "BTrk".A0302_EXIT."B"["BTRK_A0302_RULL_PAREGGIATO"], ENO => #_w3);
   "BTrk_Presence"(EN := #CIn.Manipolatori.InPos_BancoA0303,
                   Item := "BTrk".A0302_EXIT."B"["BTRK_A0302_MANIP_DEPOSITO_A0303_ALTO"],
                   ENO => #_w4);
   "BTrk_Presence"(Item := "BTrk".A0302_EXIT."B"["BTRK_A0302_MANIP_DEPOSITO_A0303_BASSO"], ENO => #_w5);
   #Ctrl.Manipolatori.Sollevatori.Work := ((#_w1 OR #_w2 OR #_w3) AND #CIn.Manipolatori.InPos_Prelievo) OR (#_w4 AND #CIn.Banco_A0303.ReadyToRecive) OR (#_w5 AND NOT #CIn.Manipolatori.Testa.Magnete.Rest AND NOT #CIn.Manipolatori.Coda.Magnete.Rest);
   IF NOT #CIn.Manipolatori.InPos_BancoA0303 AND NOT #CIn.Manipolatori.InPos_Prelievo AND NOT #CIn.Manipolatori.InPos_BancoScarto THEN
       #Ctrl.Manipolatori.Sollevatori.Work := FALSE;
   END_IF;
   #Ctrl.Manipolatori.Sollevatori.Rest := NOT #Ctrl.Manipolatori.Sollevatori.Work;
END_REGION

REGION Network 118: [Magneti] - Manipolatori Testa/Coda - Movimento operazione a lavoro / a riposo
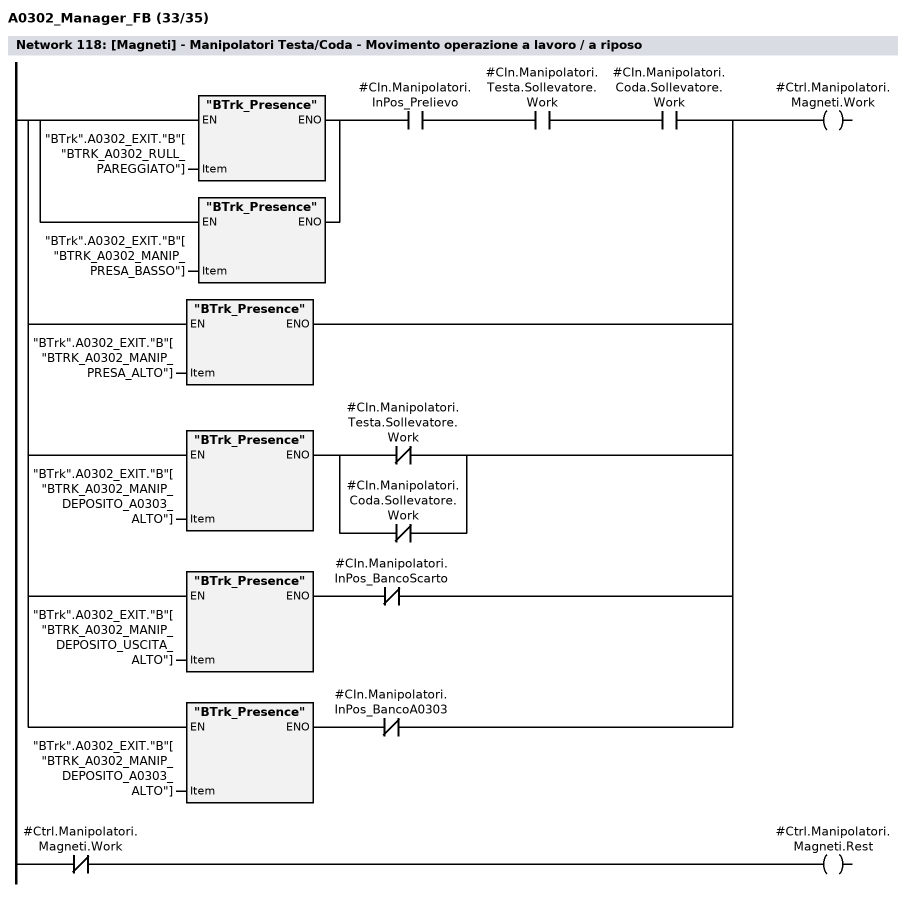
   RUNG wire#powerrail
      "BTrk_Presence"(Item := "BTrk".A0302_EXIT."B"["BTRK_A0302_RULL_PAREGGIATO"])
      wire#w1
      Contact( #CIn.Manipolatori.InPos_Prelievo )
      Contact( #CIn.Manipolatori.Testa.Sollevatore.Work )
      Contact( #CIn.Manipolatori.Coda.Sollevatore.Work )
      wire#w2
      Coil( #Ctrl.Manipolatori.Magneti.Work )
   END_RUNG
   RUNG wire#powerrail
      "BTrk_Presence"(Item := "BTrk".A0302_EXIT."B"["BTRK_A0302_MANIP_PRESA_BASSO"])
   END_RUNG wire#w1
   RUNG wire#powerrail
      "BTrk_Presence"(Item := "BTrk".A0302_EXIT."B"["BTRK_A0302_MANIP_PRESA_ALTO"])
   END_RUNG wire#w2
   RUNG wire#powerrail
      "BTrk_Presence"(Item := "BTrk".A0302_EXIT."B"["BTRK_A0302_MANIP_DEPOSITO_A0303_ALTO"])
      wire#w3
      I_Contact( #CIn.Manipolatori.Testa.Sollevatore.Work )
   END_RUNG wire#w2
   RUNG wire#w3
      I_Contact( #CIn.Manipolatori.Coda.Sollevatore.Work )
   END_RUNG wire#w2
   RUNG wire#powerrail
      "BTrk_Presence"(Item := "BTrk".A0302_EXIT."B"["BTRK_A0302_MANIP_DEPOSITO_USCITA_ALTO"])
      I_Contact( #CIn.Manipolatori.InPos_BancoScarto )
   END_RUNG wire#w2
   RUNG wire#powerrail
      "BTrk_Presence"(Item := "BTrk".A0302_EXIT."B"["BTRK_A0302_MANIP_DEPOSITO_A0303_ALTO"])
      I_Contact( #CIn.Manipolatori.InPos_BancoA0303 )
   END_RUNG wire#w2
   RUNG wire#powerrail
      I_Contact( #Ctrl.Manipolatori.Magneti.Work )
      Coil( #Ctrl.Manipolatori.Magneti.Rest )
   END_RUNG
   // the same network as SCL:
   "BTrk_Presence"(Item := "BTrk".A0302_EXIT."B"["BTRK_A0302_RULL_PAREGGIATO"], ENO => #_w1);
   "BTrk_Presence"(Item := "BTrk".A0302_EXIT."B"["BTRK_A0302_MANIP_PRESA_BASSO"], ENO => #_w2);
   "BTrk_Presence"(Item := "BTrk".A0302_EXIT."B"["BTRK_A0302_MANIP_PRESA_ALTO"], ENO => #_w3);
   "BTrk_Presence"(Item := "BTrk".A0302_EXIT."B"["BTRK_A0302_MANIP_DEPOSITO_A0303_ALTO"], ENO => #_w4);
   "BTrk_Presence"(Item := "BTrk".A0302_EXIT."B"["BTRK_A0302_MANIP_DEPOSITO_USCITA_ALTO"], ENO => #_w5);
   "BTrk_Presence"(Item := "BTrk".A0302_EXIT."B"["BTRK_A0302_MANIP_DEPOSITO_A0303_ALTO"], ENO => #_w6);
   #Ctrl.Manipolatori.Magneti.Work := ((#_w1 OR #_w2) AND #CIn.Manipolatori.InPos_Prelievo AND #CIn.Manipolatori.Testa.Sollevatore.Work AND #CIn.Manipolatori.Coda.Sollevatore.Work) OR #_w3 OR (#_w4 AND (NOT #CIn.Manipolatori.Testa.Sollevatore.Work OR NOT #CIn.Manipolatori.Coda.Sollevatore.Work)) OR (#_w5 AND NOT #CIn.Manipolatori.InPos_BancoScarto) OR (#_w6 AND NOT #CIn.Manipolatori.InPos_BancoA0303);
   #Ctrl.Manipolatori.Magneti.Rest := NOT #Ctrl.Manipolatori.Magneti.Work;
END_REGION

REGION Network 119: <+>
END_REGION

REGION Network 120: [Sollevatori + Magneti + Ax] - Manipolatori Testa/Coda - COut Manager
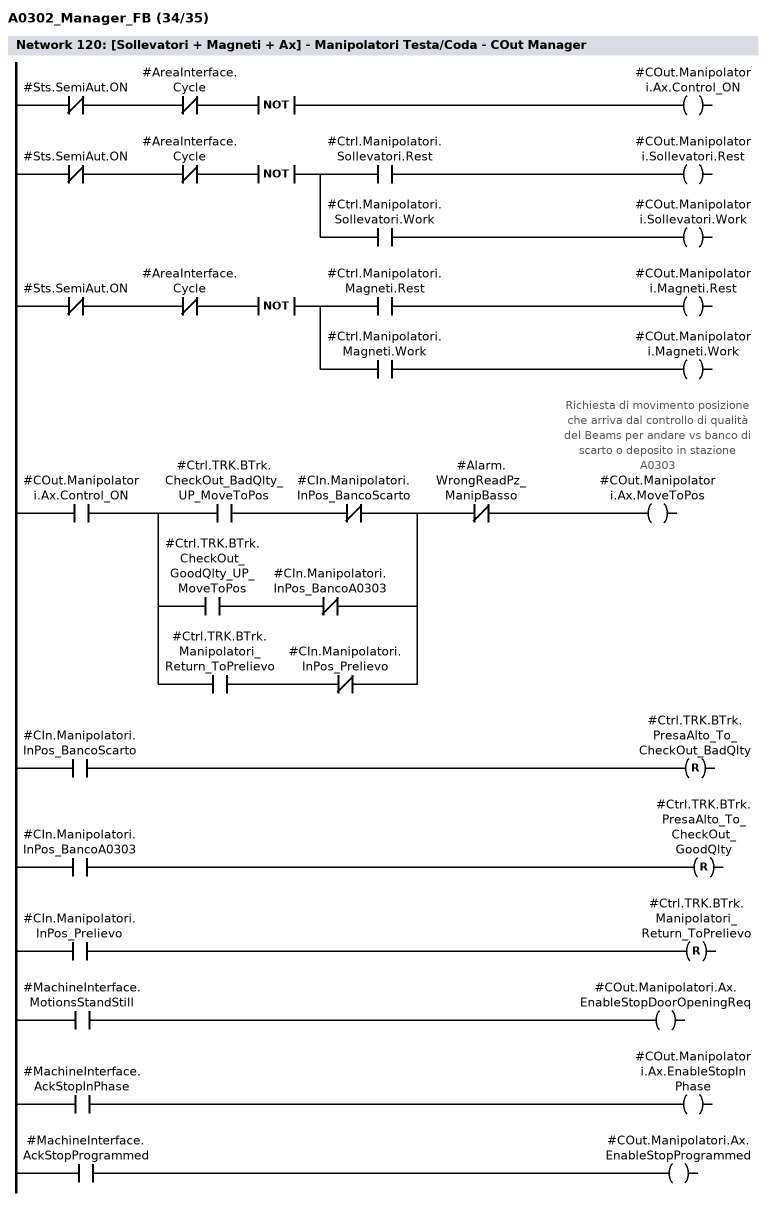
   RUNG wire#powerrail
      I_Contact( #Sts.SemiAut.ON )
      I_Contact( #AreaInterface.Cycle )
      Not()
      Coil( #COut.Manipolatori.Ax.Control_ON )
   END_RUNG
   RUNG wire#powerrail
      I_Contact( #Sts.SemiAut.ON )
      I_Contact( #AreaInterface.Cycle )
      Not()
      wire#w1
      Contact( #Ctrl.Manipolatori.Sollevatori.Rest )
      Coil( #COut.Manipolatori.Sollevatori.Rest )
   END_RUNG
   RUNG wire#w1
      Contact( #Ctrl.Manipolatori.Sollevatori.Work )
      Coil( #COut.Manipolatori.Sollevatori.Work )
   END_RUNG
   RUNG wire#powerrail
      I_Contact( #Sts.SemiAut.ON )
      I_Contact( #AreaInterface.Cycle )
      Not()
      wire#w2
      Contact( #Ctrl.Manipolatori.Magneti.Rest )
      Coil( #COut.Manipolatori.Magneti.Rest )
   END_RUNG
   RUNG wire#w2
      Contact( #Ctrl.Manipolatori.Magneti.Work )
      Coil( #COut.Manipolatori.Magneti.Work )
   END_RUNG
   RUNG wire#powerrail
      Contact( #COut.Manipolatori.Ax.Control_ON )
      wire#w3
      Contact( #Ctrl.TRK.BTrk.CheckOut_BadQlty_UP_MoveToPos )
      I_Contact( #CIn.Manipolatori.InPos_BancoScarto )
      wire#w4
      I_Contact( #Alarm.WrongReadPz_ManipBasso )
      Coil( #COut.Manipolatori.Ax.MoveToPos )   // Richiesta di movimento posizione che arriva dal controllo di qualità del Beams per andare vs banco di scarto o deposito in stazione A0303
   END_RUNG
   RUNG wire#w3
      Contact( #Ctrl.TRK.BTrk.CheckOut_GoodQlty_UP_MoveToPos )
      I_Contact( #CIn.Manipolatori.InPos_BancoA0303 )
   END_RUNG wire#w4
   RUNG wire#w3
      Contact( #Ctrl.TRK.BTrk.Manipolatori_Return_ToPrelievo )
      I_Contact( #CIn.Manipolatori.InPos_Prelievo )
   END_RUNG wire#w4
   RUNG wire#powerrail
      Contact( #CIn.Manipolatori.InPos_BancoScarto )
      R_Coil( #Ctrl.TRK.BTrk.PresaAlto_To_CheckOut_BadQlty )
   END_RUNG
   RUNG wire#powerrail
      Contact( #CIn.Manipolatori.InPos_BancoA0303 )
      R_Coil( #Ctrl.TRK.BTrk.PresaAlto_To_CheckOut_GoodQlty )
   END_RUNG
   RUNG wire#powerrail
      Contact( #CIn.Manipolatori.InPos_Prelievo )
      R_Coil( #Ctrl.TRK.BTrk.Manipolatori_Return_ToPrelievo )
   END_RUNG
   RUNG wire#powerrail
      Contact( #MachineInterface.MotionsStandStill )
      Coil( #COut.Manipolatori.Ax.EnableStopDoorOpeningReq )
   END_RUNG
   RUNG wire#powerrail
      Contact( #MachineInterface.AckStopInPhase )
      Coil( #COut.Manipolatori.Ax.EnableStopInPhase )
   END_RUNG
   RUNG wire#powerrail
      Contact( #MachineInterface.AckStopProgrammed )
      Coil( #COut.Manipolatori.Ax.EnableStopProgrammed )
   END_RUNG
   // the same network as SCL:
   #COut.Manipolatori.Ax.Control_ON := NOT (NOT #Sts.SemiAut.ON AND NOT #AreaInterface.Cycle);
   #_w1 := NOT (NOT #Sts.SemiAut.ON AND NOT #AreaInterface.Cycle);
   #COut.Manipolatori.Sollevatori.Rest := #_w1 AND #Ctrl.Manipolatori.Sollevatori.Rest;
   #COut.Manipolatori.Sollevatori.Work := #_w1 AND #Ctrl.Manipolatori.Sollevatori.Work;
   #_w2 := NOT (NOT #Sts.SemiAut.ON AND NOT #AreaInterface.Cycle);
   #COut.Manipolatori.Magneti.Rest := #_w2 AND #Ctrl.Manipolatori.Magneti.Rest;
   #COut.Manipolatori.Magneti.Work := #_w2 AND #Ctrl.Manipolatori.Magneti.Work;
   #COut.Manipolatori.Ax.MoveToPos := #COut.Manipolatori.Ax.Control_ON AND ((#Ctrl.TRK.BTrk.CheckOut_BadQlty_UP_MoveToPos AND NOT #CIn.Manipolatori.InPos_BancoScarto) OR (#Ctrl.TRK.BTrk.CheckOut_GoodQlty_UP_MoveToPos AND NOT #CIn.Manipolatori.InPos_BancoA0303) OR (#Ctrl.TRK.BTrk.Manipolatori_Return_ToPrelievo AND NOT #CIn.Manipolatori.InPos_Prelievo)) AND NOT #Alarm.WrongReadPz_ManipBasso;   // Richiesta di movimento posizione che arriva dal controllo di qualità del Beams per andare vs banco di scarto o deposito in stazione A0303
   IF #CIn.Manipolatori.InPos_BancoScarto THEN #Ctrl.TRK.BTrk.PresaAlto_To_CheckOut_BadQlty := FALSE; END_IF;
   IF #CIn.Manipolatori.InPos_BancoA0303 THEN #Ctrl.TRK.BTrk.PresaAlto_To_CheckOut_GoodQlty := FALSE; END_IF;
   IF #CIn.Manipolatori.InPos_Prelievo THEN #Ctrl.TRK.BTrk.Manipolatori_Return_ToPrelievo := FALSE; END_IF;
   #COut.Manipolatori.Ax.EnableStopDoorOpeningReq := #MachineInterface.MotionsStandStill;
   #COut.Manipolatori.Ax.EnableStopInPhase := #MachineInterface.AckStopInPhase;
   #COut.Manipolatori.Ax.EnableStopProgrammed := #MachineInterface.AckStopProgrammed;
END_REGION

